REGION Network 50: Step[401] : JOB[4] Condition
   RUNG wire#powerrail
      { S7_Templates := "SrcType := DInt" } EQ_Contact(in1 := "Unit1.Em4.ControlNodes".sideTapeAttachment.sequence.status.currentStep, in2 := #JOB_4_STEP_1)
      Contact( "Unit1.Em4.ControlNodes".sideTapeAttachment.sequence.status.seqActive )
      wire#w1
      Coil( "Unit1.Em4.ControlNodes".sideTapeAttachment."step".action1[401] )
   END_RUNG
   RUNG wire#w1
      Coil( "Unit1.Em4.ControlNodes".sideTapeAttachment."step".transition1[401] )
   END_RUNG
   RUNG wire#w1
      Contact( "Unit1.Em4.ControlNodes".sideTapeAttachment."step".transition1[401] )
      { S7_Templates := "time_type := Time" } #statTonTime[401].TON(pt := T#100ms, et =>)
      wire#w2
      I_Contact( #unitStatus.specialFunctions."sideTapeLeft1 Unuse" )
      I_Contact( #unitStatus.specialFunctions."sideTapeRight1 Unuse" )
      wire#w3
      Contact( "Unit1.Em4.ControlNodes".sideTapeAttachment.homeCheck.waitPosTapeAllGet )
      wire#w4
      Move(in := #JOB_4_STEP_10, out1 => "Unit1.Em4.ControlNodes".sideTapeAttachment.sequence.status.nextStep)
   END_RUNG
   RUNG wire#w3
      Contact( "Unit1.Em4.ControlNodes".sideTapeAttachment.homeCheck.putPosTapeAllGet )
   END_RUNG wire#w4
   RUNG wire#w2
      Contact( #unitStatus.specialFunctions."sideTapeLeft1 Unuse" )
      Contact( "Unit1.Em4.ControlNodes".sideTapeAttachment.homeCheck.waitPosTapeRightGet )
   END_RUNG wire#w4
   RUNG wire#w2
      Contact( #unitStatus.specialFunctions."sideTapeRight1 Unuse" )
      Contact( "Unit1.Em4.ControlNodes".sideTapeAttachment.homeCheck.waitPosTapeLeftGet )
   END_RUNG wire#w4
   RUNG wire#w2
      Contact( #unitStatus.specialFunctions."sideTapeLeft1 Unuse" )
      Contact( #unitStatus.specialFunctions."sideTapeRight1 Unuse" )
      Move(in := #JOB_4_STEP_90, out1 => "Unit1.Em4.ControlNodes".sideTapeAttachment.sequence.status.nextStep)
   END_RUNG
   // the same network as SCL:
   "Unit1.Em4.ControlNodes".sideTapeAttachment."step".action1[401] := ("Unit1.Em4.ControlNodes".sideTapeAttachment.sequence.status.currentStep = #JOB_4_STEP_1) AND "Unit1.Em4.ControlNodes".sideTapeAttachment.sequence.status.seqActive;
   "Unit1.Em4.ControlNodes".sideTapeAttachment."step".transition1[401] := ("Unit1.Em4.ControlNodes".sideTapeAttachment.sequence.status.currentStep = #JOB_4_STEP_1) AND "Unit1.Em4.ControlNodes".sideTapeAttachment.sequence.status.seqActive;
   #statTonTime[401].TON(IN := ("Unit1.Em4.ControlNodes".sideTapeAttachment.sequence.status.currentStep = #JOB_4_STEP_1) AND "Unit1.Em4.ControlNodes".sideTapeAttachment.sequence.status.seqActive AND "Unit1.Em4.ControlNodes".sideTapeAttachment."step".transition1[401],
                         PT := T#100ms);
   IF #statTonTime[401].Q AND ((NOT #unitStatus.specialFunctions."sideTapeLeft1 Unuse" AND NOT #unitStatus.specialFunctions."sideTapeRight1 Unuse" AND ("Unit1.Em4.ControlNodes".sideTapeAttachment.homeCheck.waitPosTapeAllGet OR "Unit1.Em4.ControlNodes".sideTapeAttachment.homeCheck.putPosTapeAllGet)) OR (#unitStatus.specialFunctions."sideTapeLeft1 Unuse" AND "Unit1.Em4.ControlNodes".sideTapeAttachment.homeCheck.waitPosTapeRightGet) OR (#unitStatus.specialFunctions."sideTapeRight1 Unuse" AND "Unit1.Em4.ControlNodes".sideTapeAttachment.homeCheck.waitPosTapeLeftGet)) THEN
       "Unit1.Em4.ControlNodes".sideTapeAttachment.sequence.status.nextStep := #JOB_4_STEP_10;
   END_IF;
   IF #statTonTime[401].Q AND #unitStatus.specialFunctions."sideTapeLeft1 Unuse" AND #unitStatus.specialFunctions."sideTapeRight1 Unuse" THEN
       "Unit1.Em4.ControlNodes".sideTapeAttachment.sequence.status.nextStep := #JOB_4_STEP_90;
   END_IF;
END_REGION

REGION Network 51: Step[410] : Side Tape Attachment X-Axis Tape-1 Put Pos
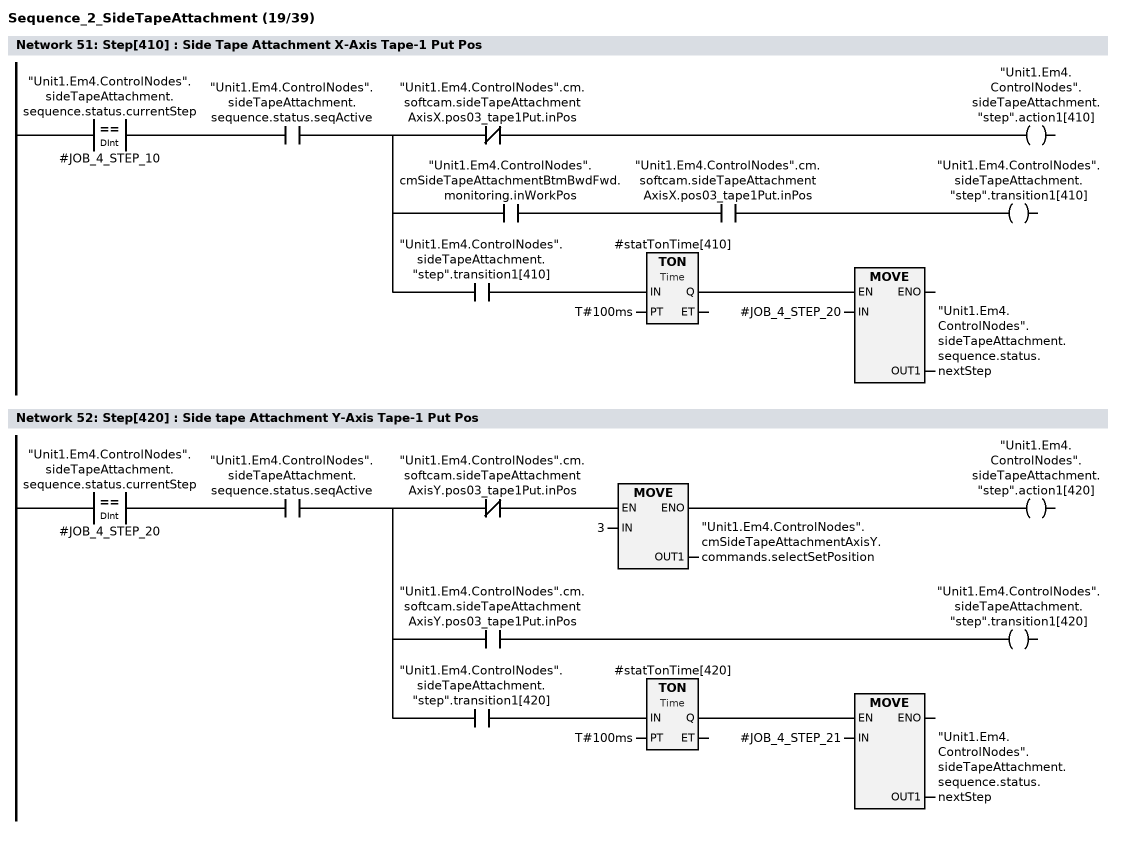
   RUNG wire#powerrail
      { S7_Templates := "SrcType := DInt" } EQ_Contact(in1 := "Unit1.Em4.ControlNodes".sideTapeAttachment.sequence.status.currentStep, in2 := #JOB_4_STEP_10)
      Contact( "Unit1.Em4.ControlNodes".sideTapeAttachment.sequence.status.seqActive )
      wire#w1
      I_Contact( "Unit1.Em4.ControlNodes".cm.softcam.sideTapeAttachmentAxisX.pos03_tape1Put.inPos )
      Coil( "Unit1.Em4.ControlNodes".sideTapeAttachment."step".action1[410] )
   END_RUNG
   RUNG wire#w1
      Contact( "Unit1.Em4.ControlNodes".cmSideTapeAttachmentBtmBwdFwd.monitoring.inWorkPos )
      Contact( "Unit1.Em4.ControlNodes".cm.softcam.sideTapeAttachmentAxisX.pos03_tape1Put.inPos )
      Coil( "Unit1.Em4.ControlNodes".sideTapeAttachment."step".transition1[410] )
   END_RUNG
   RUNG wire#w1
      Contact( "Unit1.Em4.ControlNodes".sideTapeAttachment."step".transition1[410] )
      { S7_Templates := "time_type := Time" } #statTonTime[410].TON(pt := T#100ms, et =>)
      Move(in := #JOB_4_STEP_20, out1 => "Unit1.Em4.ControlNodes".sideTapeAttachment.sequence.status.nextStep)
   END_RUNG
   // the same network as SCL:
   #_w1 := ("Unit1.Em4.ControlNodes".sideTapeAttachment.sequence.status.currentStep = #JOB_4_STEP_10) AND "Unit1.Em4.ControlNodes".sideTapeAttachment.sequence.status.seqActive;
   "Unit1.Em4.ControlNodes".sideTapeAttachment."step".action1[410] := #_w1 AND NOT "Unit1.Em4.ControlNodes".cm.softcam.sideTapeAttachmentAxisX.pos03_tape1Put.inPos;
   "Unit1.Em4.ControlNodes".sideTapeAttachment."step".transition1[410] := #_w1 AND "Unit1.Em4.ControlNodes".cmSideTapeAttachmentBtmBwdFwd.monitoring.inWorkPos AND "Unit1.Em4.ControlNodes".cm.softcam.sideTapeAttachmentAxisX.pos03_tape1Put.inPos;
   #statTonTime[410].TON(IN := #_w1 AND "Unit1.Em4.ControlNodes".sideTapeAttachment."step".transition1[410],
                         PT := T#100ms);
   IF #statTonTime[410].Q THEN
       "Unit1.Em4.ControlNodes".sideTapeAttachment.sequence.status.nextStep := #JOB_4_STEP_20;
   END_IF;
END_REGION

REGION Network 52: Step[420] : Side tape Attachment Y-Axis Tape-1 Put Pos
   RUNG wire#powerrail
      { S7_Templates := "SrcType := DInt" } EQ_Contact(in1 := "Unit1.Em4.ControlNodes".sideTapeAttachment.sequence.status.currentStep, in2 := #JOB_4_STEP_20)
      Contact( "Unit1.Em4.ControlNodes".sideTapeAttachment.sequence.status.seqActive )
      wire#w1
      I_Contact( "Unit1.Em4.ControlNodes".cm.softcam.sideTapeAttachmentAxisY.pos03_tape1Put.inPos )
      Move(in := 3, out1 => "Unit1.Em4.ControlNodes".cmSideTapeAttachmentAxisY.commands.selectSetPosition)
      Coil( "Unit1.Em4.ControlNodes".sideTapeAttachment."step".action1[420] )
   END_RUNG
   RUNG wire#w1
      Contact( "Unit1.Em4.ControlNodes".cm.softcam.sideTapeAttachmentAxisY.pos03_tape1Put.inPos )
      Coil( "Unit1.Em4.ControlNodes".sideTapeAttachment."step".transition1[420] )
   END_RUNG
   RUNG wire#w1
      Contact( "Unit1.Em4.ControlNodes".sideTapeAttachment."step".transition1[420] )
      { S7_Templates := "time_type := Time" } #statTonTime[420].TON(pt := T#100ms, et =>)
      Move(in := #JOB_4_STEP_21, out1 => "Unit1.Em4.ControlNodes".sideTapeAttachment.sequence.status.nextStep)
   END_RUNG
   // the same network as SCL:
   #_w1 := ("Unit1.Em4.ControlNodes".sideTapeAttachment.sequence.status.currentStep = #JOB_4_STEP_20) AND "Unit1.Em4.ControlNodes".sideTapeAttachment.sequence.status.seqActive;
   #_w2 := #_w1 AND NOT "Unit1.Em4.ControlNodes".cm.softcam.sideTapeAttachmentAxisY.pos03_tape1Put.inPos;
   IF #_w2 THEN "Unit1.Em4.ControlNodes".cmSideTapeAttachmentAxisY.commands.selectSetPosition := 3; END_IF;
   "Unit1.Em4.ControlNodes".sideTapeAttachment."step".action1[420] := #_w2;
   "Unit1.Em4.ControlNodes".sideTapeAttachment."step".transition1[420] := #_w1 AND "Unit1.Em4.ControlNodes".cm.softcam.sideTapeAttachmentAxisY.pos03_tape1Put.inPos;
   #statTonTime[420].TON(IN := #_w1 AND "Unit1.Em4.ControlNodes".sideTapeAttachment."step".transition1[420],
                         PT := T#100ms);
   IF #statTonTime[420].Q THEN
       "Unit1.Em4.ControlNodes".sideTapeAttachment.sequence.status.nextStep := #JOB_4_STEP_21;
   END_IF;
END_REGION

REGION Network 53: Step[421] : Side Tape Attachment Left, Right Forward, Vaccum Off
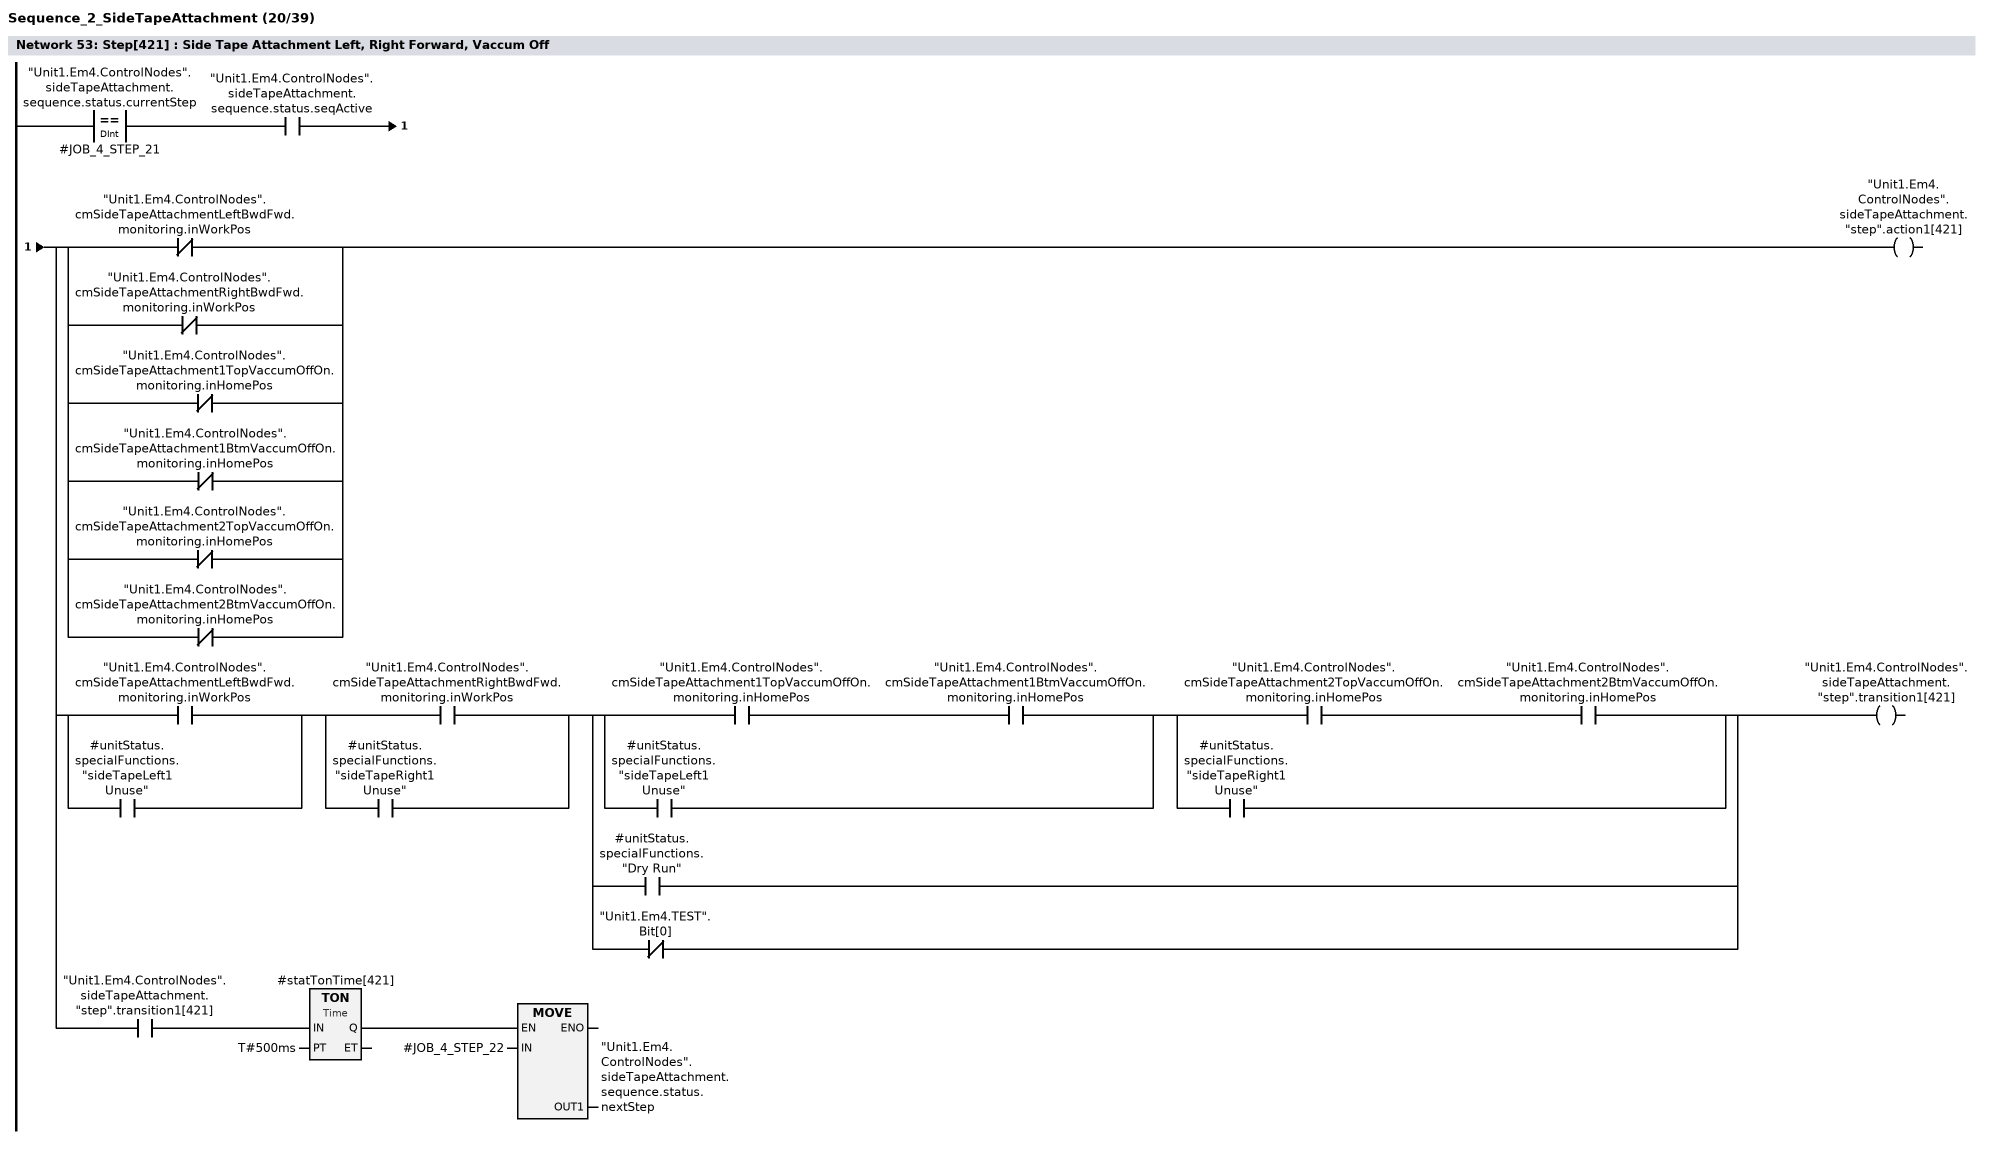
   RUNG wire#powerrail
      { S7_Templates := "SrcType := DInt" } EQ_Contact(in1 := "Unit1.Em4.ControlNodes".sideTapeAttachment.sequence.status.currentStep, in2 := #JOB_4_STEP_21)
      Contact( "Unit1.Em4.ControlNodes".sideTapeAttachment.sequence.status.seqActive )
      wire#w1
      I_Contact( "Unit1.Em4.ControlNodes".cmSideTapeAttachmentLeftBwdFwd.monitoring.inWorkPos )
      wire#w2
      Coil( "Unit1.Em4.ControlNodes".sideTapeAttachment."step".action1[421] )
   END_RUNG
   RUNG wire#w1
      I_Contact( "Unit1.Em4.ControlNodes".cmSideTapeAttachmentRightBwdFwd.monitoring.inWorkPos )
   END_RUNG wire#w2
   RUNG wire#w1
      I_Contact( "Unit1.Em4.ControlNodes".cmSideTapeAttachment1TopVaccumOffOn.monitoring.inHomePos )
   END_RUNG wire#w2
   RUNG wire#w1
      I_Contact( "Unit1.Em4.ControlNodes".cmSideTapeAttachment1BtmVaccumOffOn.monitoring.inHomePos )
   END_RUNG wire#w2
   RUNG wire#w1
      I_Contact( "Unit1.Em4.ControlNodes".cmSideTapeAttachment2TopVaccumOffOn.monitoring.inHomePos )
   END_RUNG wire#w2
   RUNG wire#w1
      I_Contact( "Unit1.Em4.ControlNodes".cmSideTapeAttachment2BtmVaccumOffOn.monitoring.inHomePos )
   END_RUNG wire#w2
   RUNG wire#w1
      Contact( "Unit1.Em4.ControlNodes".cmSideTapeAttachmentLeftBwdFwd.monitoring.inWorkPos )
      wire#w3
      Contact( "Unit1.Em4.ControlNodes".cmSideTapeAttachmentRightBwdFwd.monitoring.inWorkPos )
      wire#w4
      Contact( "Unit1.Em4.ControlNodes".cmSideTapeAttachment1TopVaccumOffOn.monitoring.inHomePos )
      Contact( "Unit1.Em4.ControlNodes".cmSideTapeAttachment1BtmVaccumOffOn.monitoring.inHomePos )
      wire#w5
      Contact( "Unit1.Em4.ControlNodes".cmSideTapeAttachment2TopVaccumOffOn.monitoring.inHomePos )
      Contact( "Unit1.Em4.ControlNodes".cmSideTapeAttachment2BtmVaccumOffOn.monitoring.inHomePos )
      wire#w6
      Coil( "Unit1.Em4.ControlNodes".sideTapeAttachment."step".transition1[421] )
   END_RUNG
   RUNG wire#w1
      Contact( #unitStatus.specialFunctions."sideTapeLeft1 Unuse" )
   END_RUNG wire#w3
   RUNG wire#w3
      Contact( #unitStatus.specialFunctions."sideTapeRight1 Unuse" )
   END_RUNG wire#w4
   RUNG wire#w4
      Contact( #unitStatus.specialFunctions."sideTapeLeft1 Unuse" )
   END_RUNG wire#w5
   RUNG wire#w5
      Contact( #unitStatus.specialFunctions."sideTapeRight1 Unuse" )
   END_RUNG wire#w6
   RUNG wire#w4
      Contact( #unitStatus.specialFunctions."Dry Run" )
   END_RUNG wire#w6
   RUNG wire#w4
      I_Contact( "Unit1.Em4.TEST".Bit[0] )
   END_RUNG wire#w6
   RUNG wire#w1
      Contact( "Unit1.Em4.ControlNodes".sideTapeAttachment."step".transition1[421] )
      { S7_Templates := "time_type := Time" } #statTonTime[421].TON(pt := T#500ms, et =>)
      Move(in := #JOB_4_STEP_22, out1 => "Unit1.Em4.ControlNodes".sideTapeAttachment.sequence.status.nextStep)
   END_RUNG
   // the same network as SCL:
   #_w1 := ("Unit1.Em4.ControlNodes".sideTapeAttachment.sequence.status.currentStep = #JOB_4_STEP_21) AND "Unit1.Em4.ControlNodes".sideTapeAttachment.sequence.status.seqActive;
   "Unit1.Em4.ControlNodes".sideTapeAttachment."step".action1[421] := #_w1 AND (NOT "Unit1.Em4.ControlNodes".cmSideTapeAttachmentLeftBwdFwd.monitoring.inWorkPos OR NOT "Unit1.Em4.ControlNodes".cmSideTapeAttachmentRightBwdFwd.monitoring.inWorkPos OR NOT "Unit1.Em4.ControlNodes".cmSideTapeAttachment1TopVaccumOffOn.monitoring.inHomePos OR NOT "Unit1.Em4.ControlNodes".cmSideTapeAttachment1BtmVaccumOffOn.monitoring.inHomePos OR NOT "Unit1.Em4.ControlNodes".cmSideTapeAttachment2TopVaccumOffOn.monitoring.inHomePos OR NOT "Unit1.Em4.ControlNodes".cmSideTapeAttachment2BtmVaccumOffOn.monitoring.inHomePos);
   "Unit1.Em4.ControlNodes".sideTapeAttachment."step".transition1[421] := #_w1 AND ("Unit1.Em4.ControlNodes".cmSideTapeAttachmentLeftBwdFwd.monitoring.inWorkPos OR #unitStatus.specialFunctions."sideTapeLeft1 Unuse") AND ("Unit1.Em4.ControlNodes".cmSideTapeAttachmentRightBwdFwd.monitoring.inWorkPos OR #unitStatus.specialFunctions."sideTapeRight1 Unuse") AND (((("Unit1.Em4.ControlNodes".cmSideTapeAttachment1TopVaccumOffOn.monitoring.inHomePos AND "Unit1.Em4.ControlNodes".cmSideTapeAttachment1BtmVaccumOffOn.monitoring.inHomePos) OR #unitStatus.specialFunctions."sideTapeLeft1 Unuse") AND (("Unit1.Em4.ControlNodes".cmSideTapeAttachment2TopVaccumOffOn.monitoring.inHomePos AND "Unit1.Em4.ControlNodes".cmSideTapeAttachment2BtmVaccumOffOn.monitoring.inHomePos) OR #unitStatus.specialFunctions."sideTapeRight1 Unuse")) OR #unitStatus.specialFunctions."Dry Run" OR NOT "Unit1.Em4.TEST".Bit[0]);
   #statTonTime[421].TON(IN := #_w1 AND "Unit1.Em4.ControlNodes".sideTapeAttachment."step".transition1[421],
                         PT := T#500ms);
   IF #statTonTime[421].Q THEN
       "Unit1.Em4.ControlNodes".sideTapeAttachment.sequence.status.nextStep := #JOB_4_STEP_22;
   END_IF;
END_REGION

REGION Network 54: Step[422] : Spare
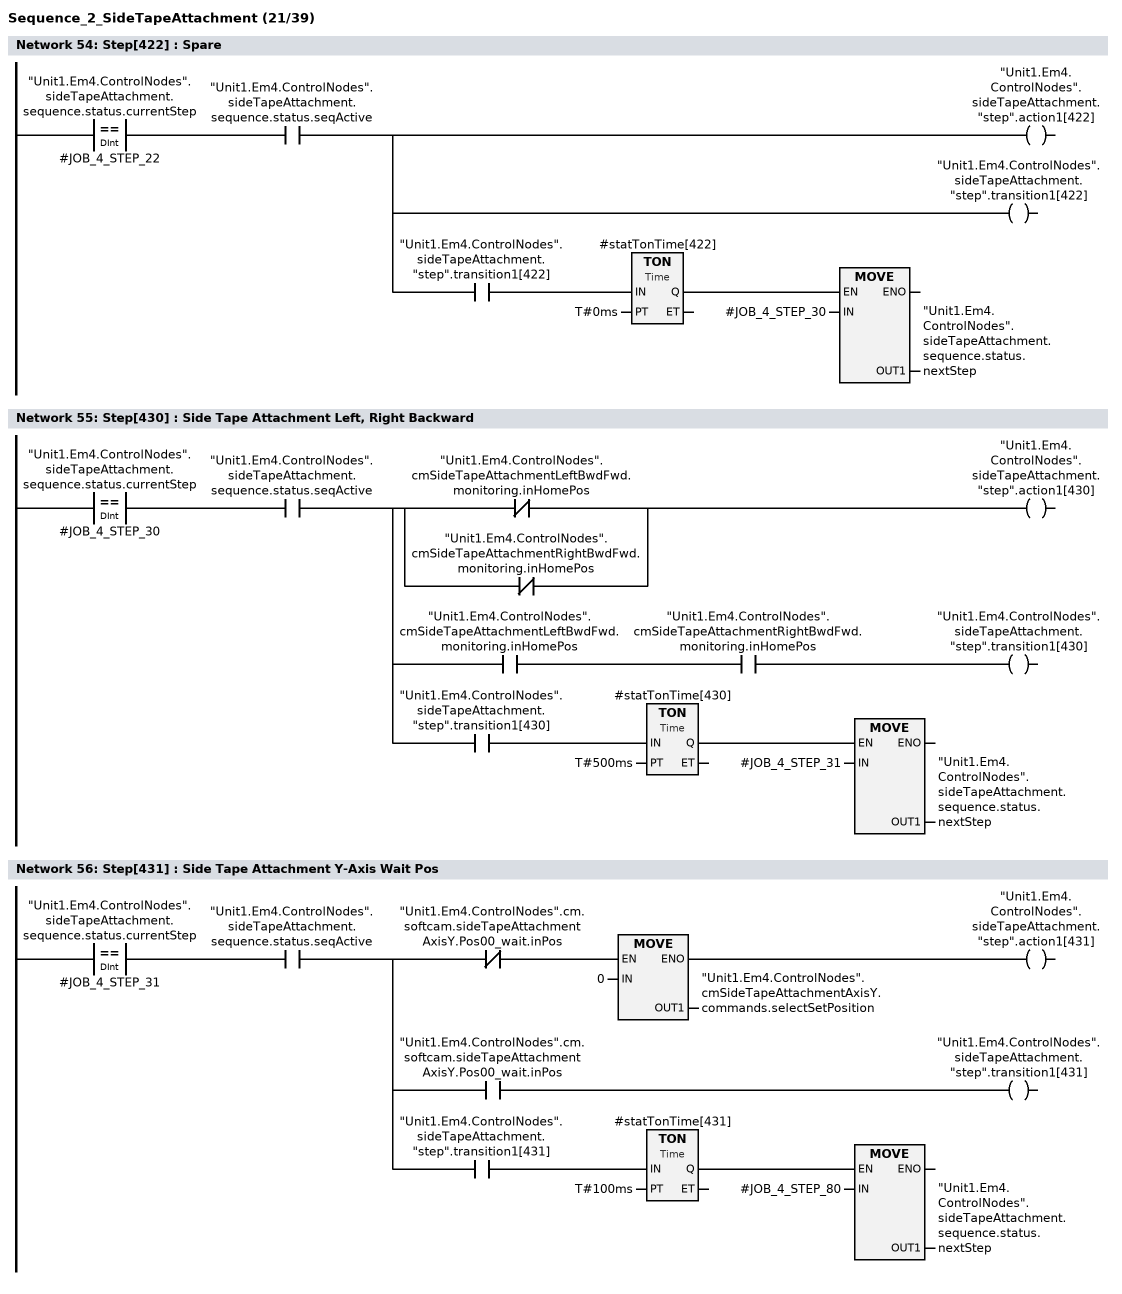
   RUNG wire#powerrail
      { S7_Templates := "SrcType := DInt" } EQ_Contact(in1 := "Unit1.Em4.ControlNodes".sideTapeAttachment.sequence.status.currentStep, in2 := #JOB_4_STEP_22)
      Contact( "Unit1.Em4.ControlNodes".sideTapeAttachment.sequence.status.seqActive )
      wire#w1
      Coil( "Unit1.Em4.ControlNodes".sideTapeAttachment."step".action1[422] )
   END_RUNG
   RUNG wire#w1
      Coil( "Unit1.Em4.ControlNodes".sideTapeAttachment."step".transition1[422] )
   END_RUNG
   RUNG wire#w1
      Contact( "Unit1.Em4.ControlNodes".sideTapeAttachment."step".transition1[422] )
      { S7_Templates := "time_type := Time" } #statTonTime[422].TON(pt := T#0ms, et =>)
      Move(in := #JOB_4_STEP_30, out1 => "Unit1.Em4.ControlNodes".sideTapeAttachment.sequence.status.nextStep)
   END_RUNG
   // the same network as SCL:
   "Unit1.Em4.ControlNodes".sideTapeAttachment."step".action1[422] := ("Unit1.Em4.ControlNodes".sideTapeAttachment.sequence.status.currentStep = #JOB_4_STEP_22) AND "Unit1.Em4.ControlNodes".sideTapeAttachment.sequence.status.seqActive;
   "Unit1.Em4.ControlNodes".sideTapeAttachment."step".transition1[422] := ("Unit1.Em4.ControlNodes".sideTapeAttachment.sequence.status.currentStep = #JOB_4_STEP_22) AND "Unit1.Em4.ControlNodes".sideTapeAttachment.sequence.status.seqActive;
   #statTonTime[422].TON(IN := ("Unit1.Em4.ControlNodes".sideTapeAttachment.sequence.status.currentStep = #JOB_4_STEP_22) AND "Unit1.Em4.ControlNodes".sideTapeAttachment.sequence.status.seqActive AND "Unit1.Em4.ControlNodes".sideTapeAttachment."step".transition1[422],
                         PT := T#0ms);
   IF #statTonTime[422].Q THEN
       "Unit1.Em4.ControlNodes".sideTapeAttachment.sequence.status.nextStep := #JOB_4_STEP_30;
   END_IF;
END_REGION

REGION Network 55: Step[430] : Side Tape Attachment Left, Right Backward
   RUNG wire#powerrail
      { S7_Templates := "SrcType := DInt" } EQ_Contact(in1 := "Unit1.Em4.ControlNodes".sideTapeAttachment.sequence.status.currentStep, in2 := #JOB_4_STEP_30)
      Contact( "Unit1.Em4.ControlNodes".sideTapeAttachment.sequence.status.seqActive )
      wire#w1
      I_Contact( "Unit1.Em4.ControlNodes".cmSideTapeAttachmentLeftBwdFwd.monitoring.inHomePos )
      wire#w2
      Coil( "Unit1.Em4.ControlNodes".sideTapeAttachment."step".action1[430] )
   END_RUNG
   RUNG wire#w1
      I_Contact( "Unit1.Em4.ControlNodes".cmSideTapeAttachmentRightBwdFwd.monitoring.inHomePos )
   END_RUNG wire#w2
   RUNG wire#w1
      Contact( "Unit1.Em4.ControlNodes".cmSideTapeAttachmentLeftBwdFwd.monitoring.inHomePos )
      Contact( "Unit1.Em4.ControlNodes".cmSideTapeAttachmentRightBwdFwd.monitoring.inHomePos )
      Coil( "Unit1.Em4.ControlNodes".sideTapeAttachment."step".transition1[430] )
   END_RUNG
   RUNG wire#w1
      Contact( "Unit1.Em4.ControlNodes".sideTapeAttachment."step".transition1[430] )
      { S7_Templates := "time_type := Time" } #statTonTime[430].TON(pt := T#500ms, et =>)
      Move(in := #JOB_4_STEP_31, out1 => "Unit1.Em4.ControlNodes".sideTapeAttachment.sequence.status.nextStep)
   END_RUNG
   // the same network as SCL:
   #_w1 := ("Unit1.Em4.ControlNodes".sideTapeAttachment.sequence.status.currentStep = #JOB_4_STEP_30) AND "Unit1.Em4.ControlNodes".sideTapeAttachment.sequence.status.seqActive;
   "Unit1.Em4.ControlNodes".sideTapeAttachment."step".action1[430] := #_w1 AND (NOT "Unit1.Em4.ControlNodes".cmSideTapeAttachmentLeftBwdFwd.monitoring.inHomePos OR NOT "Unit1.Em4.ControlNodes".cmSideTapeAttachmentRightBwdFwd.monitoring.inHomePos);
   "Unit1.Em4.ControlNodes".sideTapeAttachment."step".transition1[430] := #_w1 AND "Unit1.Em4.ControlNodes".cmSideTapeAttachmentLeftBwdFwd.monitoring.inHomePos AND "Unit1.Em4.ControlNodes".cmSideTapeAttachmentRightBwdFwd.monitoring.inHomePos;
   #statTonTime[430].TON(IN := #_w1 AND "Unit1.Em4.ControlNodes".sideTapeAttachment."step".transition1[430],
                         PT := T#500ms);
   IF #statTonTime[430].Q THEN
       "Unit1.Em4.ControlNodes".sideTapeAttachment.sequence.status.nextStep := #JOB_4_STEP_31;
   END_IF;
END_REGION

REGION Network 56: Step[431] : Side Tape Attachment Y-Axis Wait Pos
   RUNG wire#powerrail
      { S7_Templates := "SrcType := DInt" } EQ_Contact(in1 := "Unit1.Em4.ControlNodes".sideTapeAttachment.sequence.status.currentStep, in2 := #JOB_4_STEP_31)
      Contact( "Unit1.Em4.ControlNodes".sideTapeAttachment.sequence.status.seqActive )
      wire#w1
      I_Contact( "Unit1.Em4.ControlNodes".cm.softcam.sideTapeAttachmentAxisY.Pos00_wait.inPos )
      Move(in := 0, out1 => "Unit1.Em4.ControlNodes".cmSideTapeAttachmentAxisY.commands.selectSetPosition)
      Coil( "Unit1.Em4.ControlNodes".sideTapeAttachment."step".action1[431] )
   END_RUNG
   RUNG wire#w1
      Contact( "Unit1.Em4.ControlNodes".cm.softcam.sideTapeAttachmentAxisY.Pos00_wait.inPos )
      Coil( "Unit1.Em4.ControlNodes".sideTapeAttachment."step".transition1[431] )
   END_RUNG
   RUNG wire#w1
      Contact( "Unit1.Em4.ControlNodes".sideTapeAttachment."step".transition1[431] )
      { S7_Templates := "time_type := Time" } #statTonTime[431].TON(pt := T#100ms, et =>)
      Move(in := #JOB_4_STEP_80, out1 => "Unit1.Em4.ControlNodes".sideTapeAttachment.sequence.status.nextStep)
   END_RUNG
   // the same network as SCL:
   #_w1 := ("Unit1.Em4.ControlNodes".sideTapeAttachment.sequence.status.currentStep = #JOB_4_STEP_31) AND "Unit1.Em4.ControlNodes".sideTapeAttachment.sequence.status.seqActive;
   #_w2 := #_w1 AND NOT "Unit1.Em4.ControlNodes".cm.softcam.sideTapeAttachmentAxisY.Pos00_wait.inPos;
   IF #_w2 THEN "Unit1.Em4.ControlNodes".cmSideTapeAttachmentAxisY.commands.selectSetPosition := 0; END_IF;
   "Unit1.Em4.ControlNodes".sideTapeAttachment."step".action1[431] := #_w2;
   "Unit1.Em4.ControlNodes".sideTapeAttachment."step".transition1[431] := #_w1 AND "Unit1.Em4.ControlNodes".cm.softcam.sideTapeAttachmentAxisY.Pos00_wait.inPos;
   #statTonTime[431].TON(IN := #_w1 AND "Unit1.Em4.ControlNodes".sideTapeAttachment."step".transition1[431],
                         PT := T#100ms);
   IF #statTonTime[431].Q THEN
       "Unit1.Em4.ControlNodes".sideTapeAttachment.sequence.status.nextStep := #JOB_4_STEP_80;
   END_IF;
END_REGION

REGION Network 57: Step[480] : Side Tape Attachment X-Axis Wait Pos
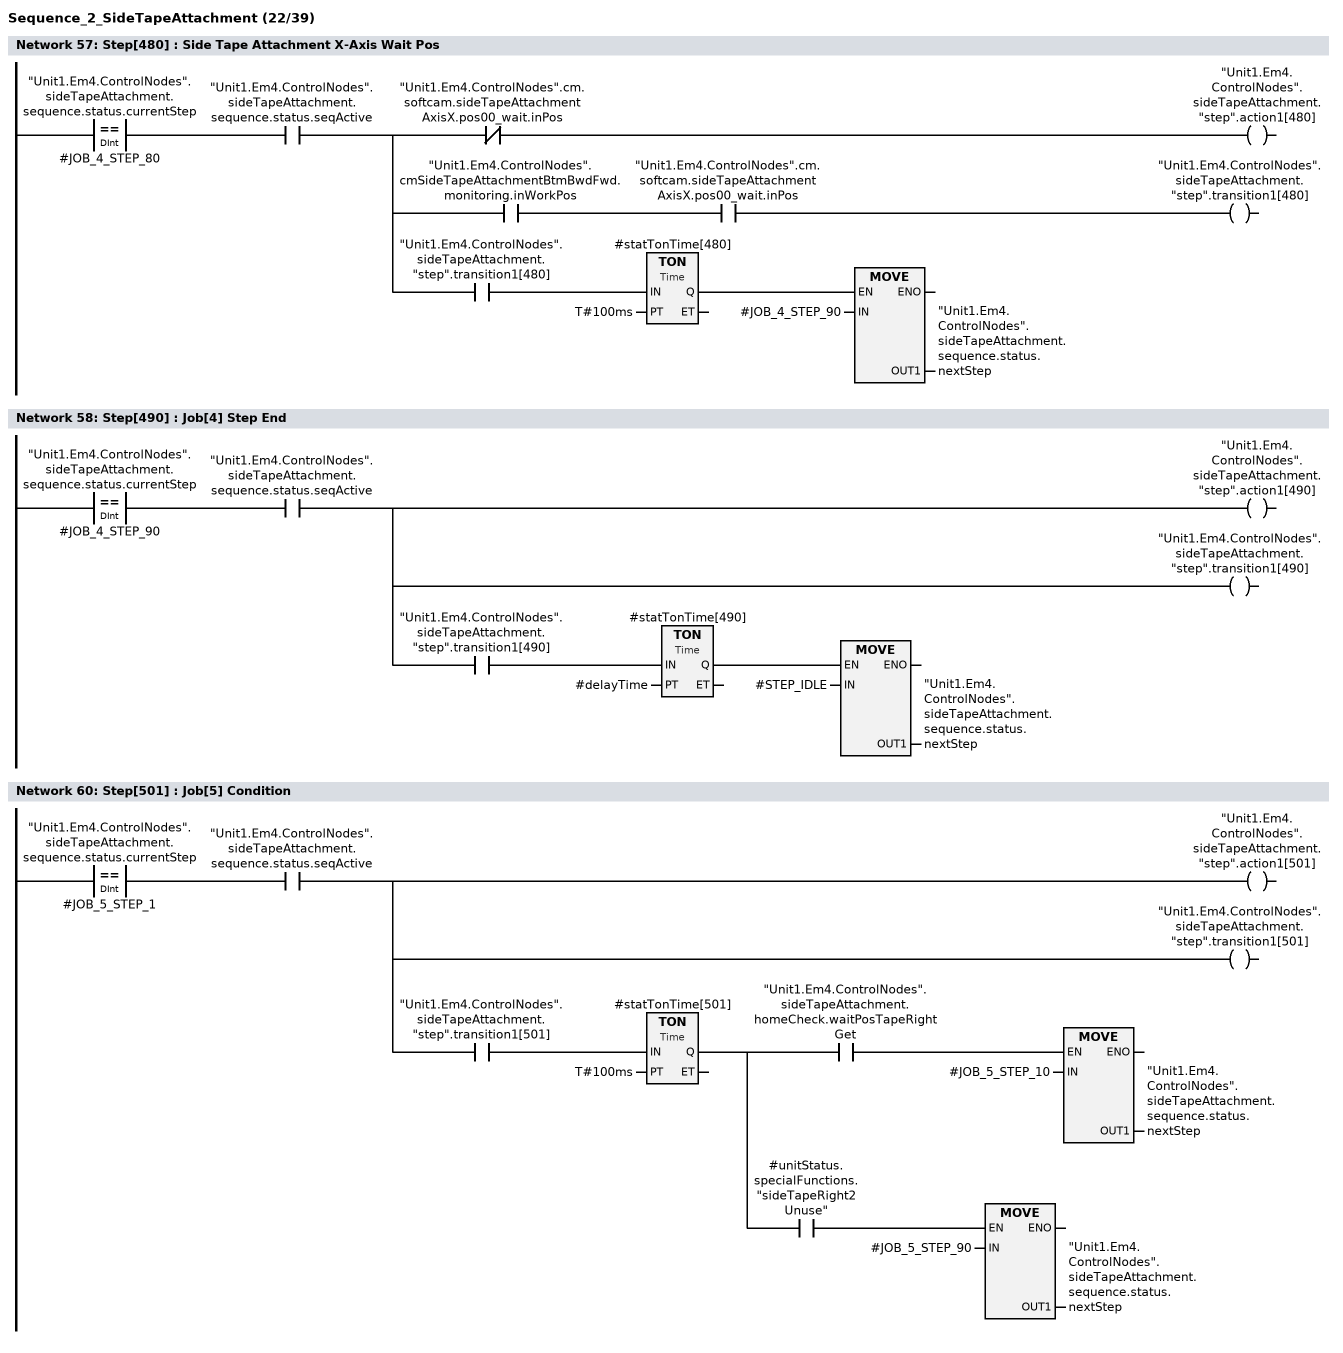
   RUNG wire#powerrail
      { S7_Templates := "SrcType := DInt" } EQ_Contact(in1 := "Unit1.Em4.ControlNodes".sideTapeAttachment.sequence.status.currentStep, in2 := #JOB_4_STEP_80)
      Contact( "Unit1.Em4.ControlNodes".sideTapeAttachment.sequence.status.seqActive )
      wire#w1
      I_Contact( "Unit1.Em4.ControlNodes".cm.softcam.sideTapeAttachmentAxisX.pos00_wait.inPos )
      Coil( "Unit1.Em4.ControlNodes".sideTapeAttachment."step".action1[480] )
   END_RUNG
   RUNG wire#w1
      Contact( "Unit1.Em4.ControlNodes".cmSideTapeAttachmentBtmBwdFwd.monitoring.inWorkPos )
      Contact( "Unit1.Em4.ControlNodes".cm.softcam.sideTapeAttachmentAxisX.pos00_wait.inPos )
      Coil( "Unit1.Em4.ControlNodes".sideTapeAttachment."step".transition1[480] )
   END_RUNG
   RUNG wire#w1
      Contact( "Unit1.Em4.ControlNodes".sideTapeAttachment."step".transition1[480] )
      { S7_Templates := "time_type := Time" } #statTonTime[480].TON(pt := T#100ms, et =>)
      Move(in := #JOB_4_STEP_90, out1 => "Unit1.Em4.ControlNodes".sideTapeAttachment.sequence.status.nextStep)
   END_RUNG
   // the same network as SCL:
   #_w1 := ("Unit1.Em4.ControlNodes".sideTapeAttachment.sequence.status.currentStep = #JOB_4_STEP_80) AND "Unit1.Em4.ControlNodes".sideTapeAttachment.sequence.status.seqActive;
   "Unit1.Em4.ControlNodes".sideTapeAttachment."step".action1[480] := #_w1 AND NOT "Unit1.Em4.ControlNodes".cm.softcam.sideTapeAttachmentAxisX.pos00_wait.inPos;
   "Unit1.Em4.ControlNodes".sideTapeAttachment."step".transition1[480] := #_w1 AND "Unit1.Em4.ControlNodes".cmSideTapeAttachmentBtmBwdFwd.monitoring.inWorkPos AND "Unit1.Em4.ControlNodes".cm.softcam.sideTapeAttachmentAxisX.pos00_wait.inPos;
   #statTonTime[480].TON(IN := #_w1 AND "Unit1.Em4.ControlNodes".sideTapeAttachment."step".transition1[480],
                         PT := T#100ms);
   IF #statTonTime[480].Q THEN
       "Unit1.Em4.ControlNodes".sideTapeAttachment.sequence.status.nextStep := #JOB_4_STEP_90;
   END_IF;
END_REGION

REGION Network 58: Step[490] : Job[4] Step End
   RUNG wire#powerrail
      { S7_Templates := "SrcType := DInt" } EQ_Contact(in1 := "Unit1.Em4.ControlNodes".sideTapeAttachment.sequence.status.currentStep, in2 := #JOB_4_STEP_90)
      Contact( "Unit1.Em4.ControlNodes".sideTapeAttachment.sequence.status.seqActive )
      wire#w1
      Coil( "Unit1.Em4.ControlNodes".sideTapeAttachment."step".action1[490] )
   END_RUNG
   RUNG wire#w1
      Coil( "Unit1.Em4.ControlNodes".sideTapeAttachment."step".transition1[490] )
   END_RUNG
   RUNG wire#w1
      Contact( "Unit1.Em4.ControlNodes".sideTapeAttachment."step".transition1[490] )
      { S7_Templates := "time_type := Time" } #statTonTime[490].TON(pt := #delayTime, et =>)
      Move(in := #STEP_IDLE, out1 => "Unit1.Em4.ControlNodes".sideTapeAttachment.sequence.status.nextStep)
   END_RUNG
   // the same network as SCL:
   "Unit1.Em4.ControlNodes".sideTapeAttachment."step".action1[490] := ("Unit1.Em4.ControlNodes".sideTapeAttachment.sequence.status.currentStep = #JOB_4_STEP_90) AND "Unit1.Em4.ControlNodes".sideTapeAttachment.sequence.status.seqActive;
   "Unit1.Em4.ControlNodes".sideTapeAttachment."step".transition1[490] := ("Unit1.Em4.ControlNodes".sideTapeAttachment.sequence.status.currentStep = #JOB_4_STEP_90) AND "Unit1.Em4.ControlNodes".sideTapeAttachment.sequence.status.seqActive;
   #statTonTime[490].TON(IN := ("Unit1.Em4.ControlNodes".sideTapeAttachment.sequence.status.currentStep = #JOB_4_STEP_90) AND "Unit1.Em4.ControlNodes".sideTapeAttachment.sequence.status.seqActive AND "Unit1.Em4.ControlNodes".sideTapeAttachment."step".transition1[490],
                         PT := #delayTime);
   IF #statTonTime[490].Q THEN
       "Unit1.Em4.ControlNodes".sideTapeAttachment.sequence.status.nextStep := #STEP_IDLE;
   END_IF;
END_REGION

REGION Network 59: *************** JOB[5] SIDE TAPE PUT-2=AUTO *************************
END_REGION

REGION Network 60: Step[501] : Job[5] Condition
   RUNG wire#powerrail
      { S7_Templates := "SrcType := DInt" } EQ_Contact(in1 := "Unit1.Em4.ControlNodes".sideTapeAttachment.sequence.status.currentStep, in2 := #JOB_5_STEP_1)
      Contact( "Unit1.Em4.ControlNodes".sideTapeAttachment.sequence.status.seqActive )
      wire#w1
      Coil( "Unit1.Em4.ControlNodes".sideTapeAttachment."step".action1[501] )
   END_RUNG
   RUNG wire#w1
      Coil( "Unit1.Em4.ControlNodes".sideTapeAttachment."step".transition1[501] )
   END_RUNG
   RUNG wire#w1
      Contact( "Unit1.Em4.ControlNodes".sideTapeAttachment."step".transition1[501] )
      { S7_Templates := "time_type := Time" } #statTonTime[501].TON(pt := T#100ms, et =>)
      wire#w2
      Contact( "Unit1.Em4.ControlNodes".sideTapeAttachment.homeCheck.waitPosTapeRightGet )
      Move(in := #JOB_5_STEP_10, out1 => "Unit1.Em4.ControlNodes".sideTapeAttachment.sequence.status.nextStep)
   END_RUNG
   RUNG wire#w2
      Contact( #unitStatus.specialFunctions."sideTapeRight2 Unuse" )
      Move(in := #JOB_5_STEP_90, out1 => "Unit1.Em4.ControlNodes".sideTapeAttachment.sequence.status.nextStep)
   END_RUNG
   // the same network as SCL:
   "Unit1.Em4.ControlNodes".sideTapeAttachment."step".action1[501] := ("Unit1.Em4.ControlNodes".sideTapeAttachment.sequence.status.currentStep = #JOB_5_STEP_1) AND "Unit1.Em4.ControlNodes".sideTapeAttachment.sequence.status.seqActive;
   "Unit1.Em4.ControlNodes".sideTapeAttachment."step".transition1[501] := ("Unit1.Em4.ControlNodes".sideTapeAttachment.sequence.status.currentStep = #JOB_5_STEP_1) AND "Unit1.Em4.ControlNodes".sideTapeAttachment.sequence.status.seqActive;
   #statTonTime[501].TON(IN := ("Unit1.Em4.ControlNodes".sideTapeAttachment.sequence.status.currentStep = #JOB_5_STEP_1) AND "Unit1.Em4.ControlNodes".sideTapeAttachment.sequence.status.seqActive AND "Unit1.Em4.ControlNodes".sideTapeAttachment."step".transition1[501],
                         PT := T#100ms);
   IF #statTonTime[501].Q AND "Unit1.Em4.ControlNodes".sideTapeAttachment.homeCheck.waitPosTapeRightGet THEN
       "Unit1.Em4.ControlNodes".sideTapeAttachment.sequence.status.nextStep := #JOB_5_STEP_10;
   END_IF;
   IF #statTonTime[501].Q AND #unitStatus.specialFunctions."sideTapeRight2 Unuse" THEN
       "Unit1.Em4.ControlNodes".sideTapeAttachment.sequence.status.nextStep := #JOB_5_STEP_90;
   END_IF;
END_REGION

REGION Network 61: Step[510] : Side Tape Attachment X-Axis Tape-2 Put Pos
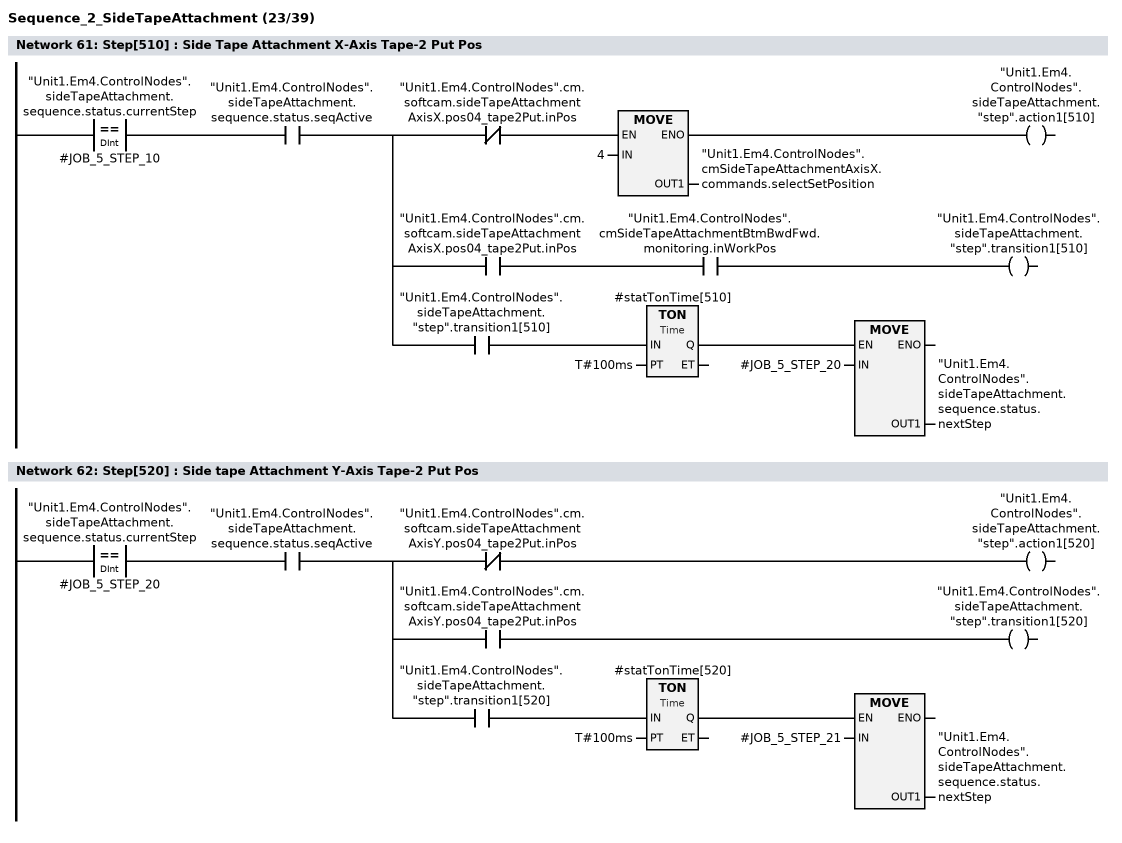
   RUNG wire#powerrail
      { S7_Templates := "SrcType := DInt" } EQ_Contact(in1 := "Unit1.Em4.ControlNodes".sideTapeAttachment.sequence.status.currentStep, in2 := #JOB_5_STEP_10)
      Contact( "Unit1.Em4.ControlNodes".sideTapeAttachment.sequence.status.seqActive )
      wire#w1
      I_Contact( "Unit1.Em4.ControlNodes".cm.softcam.sideTapeAttachmentAxisX.pos04_tape2Put.inPos )
      Move(in := 4, out1 => "Unit1.Em4.ControlNodes".cmSideTapeAttachmentAxisX.commands.selectSetPosition)
      Coil( "Unit1.Em4.ControlNodes".sideTapeAttachment."step".action1[510] )
   END_RUNG
   RUNG wire#w1
      Contact( "Unit1.Em4.ControlNodes".cm.softcam.sideTapeAttachmentAxisX.pos04_tape2Put.inPos )
      Contact( "Unit1.Em4.ControlNodes".cmSideTapeAttachmentBtmBwdFwd.monitoring.inWorkPos )
      Coil( "Unit1.Em4.ControlNodes".sideTapeAttachment."step".transition1[510] )
   END_RUNG
   RUNG wire#w1
      Contact( "Unit1.Em4.ControlNodes".sideTapeAttachment."step".transition1[510] )
      { S7_Templates := "time_type := Time" } #statTonTime[510].TON(pt := T#100ms, et =>)
      Move(in := #JOB_5_STEP_20, out1 => "Unit1.Em4.ControlNodes".sideTapeAttachment.sequence.status.nextStep)
   END_RUNG
   // the same network as SCL:
   #_w1 := ("Unit1.Em4.ControlNodes".sideTapeAttachment.sequence.status.currentStep = #JOB_5_STEP_10) AND "Unit1.Em4.ControlNodes".sideTapeAttachment.sequence.status.seqActive;
   #_w2 := #_w1 AND NOT "Unit1.Em4.ControlNodes".cm.softcam.sideTapeAttachmentAxisX.pos04_tape2Put.inPos;
   IF #_w2 THEN "Unit1.Em4.ControlNodes".cmSideTapeAttachmentAxisX.commands.selectSetPosition := 4; END_IF;
   "Unit1.Em4.ControlNodes".sideTapeAttachment."step".action1[510] := #_w2;
   "Unit1.Em4.ControlNodes".sideTapeAttachment."step".transition1[510] := #_w1 AND "Unit1.Em4.ControlNodes".cm.softcam.sideTapeAttachmentAxisX.pos04_tape2Put.inPos AND "Unit1.Em4.ControlNodes".cmSideTapeAttachmentBtmBwdFwd.monitoring.inWorkPos;
   #statTonTime[510].TON(IN := #_w1 AND "Unit1.Em4.ControlNodes".sideTapeAttachment."step".transition1[510],
                         PT := T#100ms);
   IF #statTonTime[510].Q THEN
       "Unit1.Em4.ControlNodes".sideTapeAttachment.sequence.status.nextStep := #JOB_5_STEP_20;
   END_IF;
END_REGION

REGION Network 62: Step[520] : Side tape Attachment Y-Axis Tape-2 Put Pos
   RUNG wire#powerrail
      { S7_Templates := "SrcType := DInt" } EQ_Contact(in1 := "Unit1.Em4.ControlNodes".sideTapeAttachment.sequence.status.currentStep, in2 := #JOB_5_STEP_20)
      Contact( "Unit1.Em4.ControlNodes".sideTapeAttachment.sequence.status.seqActive )
      wire#w1
      I_Contact( "Unit1.Em4.ControlNodes".cm.softcam.sideTapeAttachmentAxisY.pos04_tape2Put.inPos )
      Coil( "Unit1.Em4.ControlNodes".sideTapeAttachment."step".action1[520] )
   END_RUNG
   RUNG wire#w1
      Contact( "Unit1.Em4.ControlNodes".cm.softcam.sideTapeAttachmentAxisY.pos04_tape2Put.inPos )
      Coil( "Unit1.Em4.ControlNodes".sideTapeAttachment."step".transition1[520] )
   END_RUNG
   RUNG wire#w1
      Contact( "Unit1.Em4.ControlNodes".sideTapeAttachment."step".transition1[520] )
      { S7_Templates := "time_type := Time" } #statTonTime[520].TON(pt := T#100ms, et =>)
      Move(in := #JOB_5_STEP_21, out1 => "Unit1.Em4.ControlNodes".sideTapeAttachment.sequence.status.nextStep)
   END_RUNG
   // the same network as SCL:
   #_w1 := ("Unit1.Em4.ControlNodes".sideTapeAttachment.sequence.status.currentStep = #JOB_5_STEP_20) AND "Unit1.Em4.ControlNodes".sideTapeAttachment.sequence.status.seqActive;
   "Unit1.Em4.ControlNodes".sideTapeAttachment."step".action1[520] := #_w1 AND NOT "Unit1.Em4.ControlNodes".cm.softcam.sideTapeAttachmentAxisY.pos04_tape2Put.inPos;
   "Unit1.Em4.ControlNodes".sideTapeAttachment."step".transition1[520] := #_w1 AND "Unit1.Em4.ControlNodes".cm.softcam.sideTapeAttachmentAxisY.pos04_tape2Put.inPos;
   #statTonTime[520].TON(IN := #_w1 AND "Unit1.Em4.ControlNodes".sideTapeAttachment."step".transition1[520],
                         PT := T#100ms);
   IF #statTonTime[520].Q THEN
       "Unit1.Em4.ControlNodes".sideTapeAttachment.sequence.status.nextStep := #JOB_5_STEP_21;
   END_IF;
END_REGION

REGION Network 63: Step[521] : Side Tape Attachment Right Forward, Vaccum Off
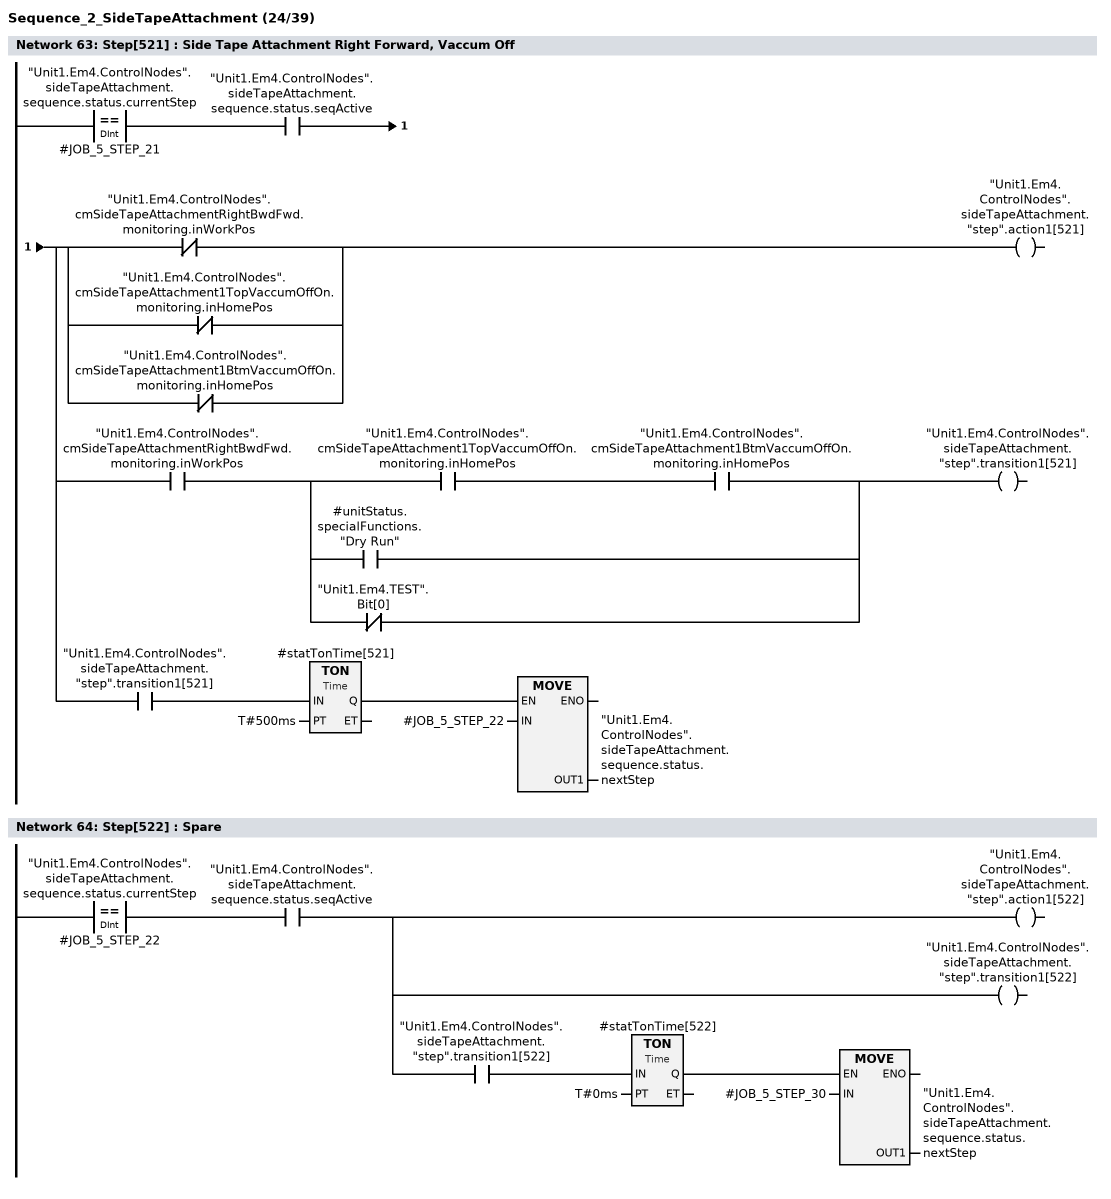
   RUNG wire#powerrail
      { S7_Templates := "SrcType := DInt" } EQ_Contact(in1 := "Unit1.Em4.ControlNodes".sideTapeAttachment.sequence.status.currentStep, in2 := #JOB_5_STEP_21)
      Contact( "Unit1.Em4.ControlNodes".sideTapeAttachment.sequence.status.seqActive )
      wire#w1
      I_Contact( "Unit1.Em4.ControlNodes".cmSideTapeAttachmentRightBwdFwd.monitoring.inWorkPos )
      wire#w2
      Coil( "Unit1.Em4.ControlNodes".sideTapeAttachment."step".action1[521] )
   END_RUNG
   RUNG wire#w1
      I_Contact( "Unit1.Em4.ControlNodes".cmSideTapeAttachment1TopVaccumOffOn.monitoring.inHomePos )
   END_RUNG wire#w2
   RUNG wire#w1
      I_Contact( "Unit1.Em4.ControlNodes".cmSideTapeAttachment1BtmVaccumOffOn.monitoring.inHomePos )
   END_RUNG wire#w2
   RUNG wire#w1
      Contact( "Unit1.Em4.ControlNodes".cmSideTapeAttachmentRightBwdFwd.monitoring.inWorkPos )
      wire#w3
      Contact( "Unit1.Em4.ControlNodes".cmSideTapeAttachment1TopVaccumOffOn.monitoring.inHomePos )
      Contact( "Unit1.Em4.ControlNodes".cmSideTapeAttachment1BtmVaccumOffOn.monitoring.inHomePos )
      wire#w4
      Coil( "Unit1.Em4.ControlNodes".sideTapeAttachment."step".transition1[521] )
   END_RUNG
   RUNG wire#w3
      Contact( #unitStatus.specialFunctions."Dry Run" )
   END_RUNG wire#w4
   RUNG wire#w3
      I_Contact( "Unit1.Em4.TEST".Bit[0] )
   END_RUNG wire#w4
   RUNG wire#w1
      Contact( "Unit1.Em4.ControlNodes".sideTapeAttachment."step".transition1[521] )
      { S7_Templates := "time_type := Time" } #statTonTime[521].TON(pt := T#500ms, et =>)
      Move(in := #JOB_5_STEP_22, out1 => "Unit1.Em4.ControlNodes".sideTapeAttachment.sequence.status.nextStep)
   END_RUNG
   // the same network as SCL:
   #_w1 := ("Unit1.Em4.ControlNodes".sideTapeAttachment.sequence.status.currentStep = #JOB_5_STEP_21) AND "Unit1.Em4.ControlNodes".sideTapeAttachment.sequence.status.seqActive;
   "Unit1.Em4.ControlNodes".sideTapeAttachment."step".action1[521] := #_w1 AND (NOT "Unit1.Em4.ControlNodes".cmSideTapeAttachmentRightBwdFwd.monitoring.inWorkPos OR NOT "Unit1.Em4.ControlNodes".cmSideTapeAttachment1TopVaccumOffOn.monitoring.inHomePos OR NOT "Unit1.Em4.ControlNodes".cmSideTapeAttachment1BtmVaccumOffOn.monitoring.inHomePos);
   "Unit1.Em4.ControlNodes".sideTapeAttachment."step".transition1[521] := #_w1 AND "Unit1.Em4.ControlNodes".cmSideTapeAttachmentRightBwdFwd.monitoring.inWorkPos AND (("Unit1.Em4.ControlNodes".cmSideTapeAttachment1TopVaccumOffOn.monitoring.inHomePos AND "Unit1.Em4.ControlNodes".cmSideTapeAttachment1BtmVaccumOffOn.monitoring.inHomePos) OR #unitStatus.specialFunctions."Dry Run" OR NOT "Unit1.Em4.TEST".Bit[0]);
   #statTonTime[521].TON(IN := #_w1 AND "Unit1.Em4.ControlNodes".sideTapeAttachment."step".transition1[521],
                         PT := T#500ms);
   IF #statTonTime[521].Q THEN
       "Unit1.Em4.ControlNodes".sideTapeAttachment.sequence.status.nextStep := #JOB_5_STEP_22;
   END_IF;
END_REGION

REGION Network 64: Step[522] : Spare
   RUNG wire#powerrail
      { S7_Templates := "SrcType := DInt" } EQ_Contact(in1 := "Unit1.Em4.ControlNodes".sideTapeAttachment.sequence.status.currentStep, in2 := #JOB_5_STEP_22)
      Contact( "Unit1.Em4.ControlNodes".sideTapeAttachment.sequence.status.seqActive )
      wire#w1
      Coil( "Unit1.Em4.ControlNodes".sideTapeAttachment."step".action1[522] )
   END_RUNG
   RUNG wire#w1
      Coil( "Unit1.Em4.ControlNodes".sideTapeAttachment."step".transition1[522] )
   END_RUNG
   RUNG wire#w1
      Contact( "Unit1.Em4.ControlNodes".sideTapeAttachment."step".transition1[522] )
      { S7_Templates := "time_type := Time" } #statTonTime[522].TON(pt := T#0ms, et =>)
      Move(in := #JOB_5_STEP_30, out1 => "Unit1.Em4.ControlNodes".sideTapeAttachment.sequence.status.nextStep)
   END_RUNG
   // the same network as SCL:
   "Unit1.Em4.ControlNodes".sideTapeAttachment."step".action1[522] := ("Unit1.Em4.ControlNodes".sideTapeAttachment.sequence.status.currentStep = #JOB_5_STEP_22) AND "Unit1.Em4.ControlNodes".sideTapeAttachment.sequence.status.seqActive;
   "Unit1.Em4.ControlNodes".sideTapeAttachment."step".transition1[522] := ("Unit1.Em4.ControlNodes".sideTapeAttachment.sequence.status.currentStep = #JOB_5_STEP_22) AND "Unit1.Em4.ControlNodes".sideTapeAttachment.sequence.status.seqActive;
   #statTonTime[522].TON(IN := ("Unit1.Em4.ControlNodes".sideTapeAttachment.sequence.status.currentStep = #JOB_5_STEP_22) AND "Unit1.Em4.ControlNodes".sideTapeAttachment.sequence.status.seqActive AND "Unit1.Em4.ControlNodes".sideTapeAttachment."step".transition1[522],
                         PT := T#0ms);
   IF #statTonTime[522].Q THEN
       "Unit1.Em4.ControlNodes".sideTapeAttachment.sequence.status.nextStep := #JOB_5_STEP_30;
   END_IF;
END_REGION

REGION Network 65: Step[530] : Side Tape Attachment Right Backward
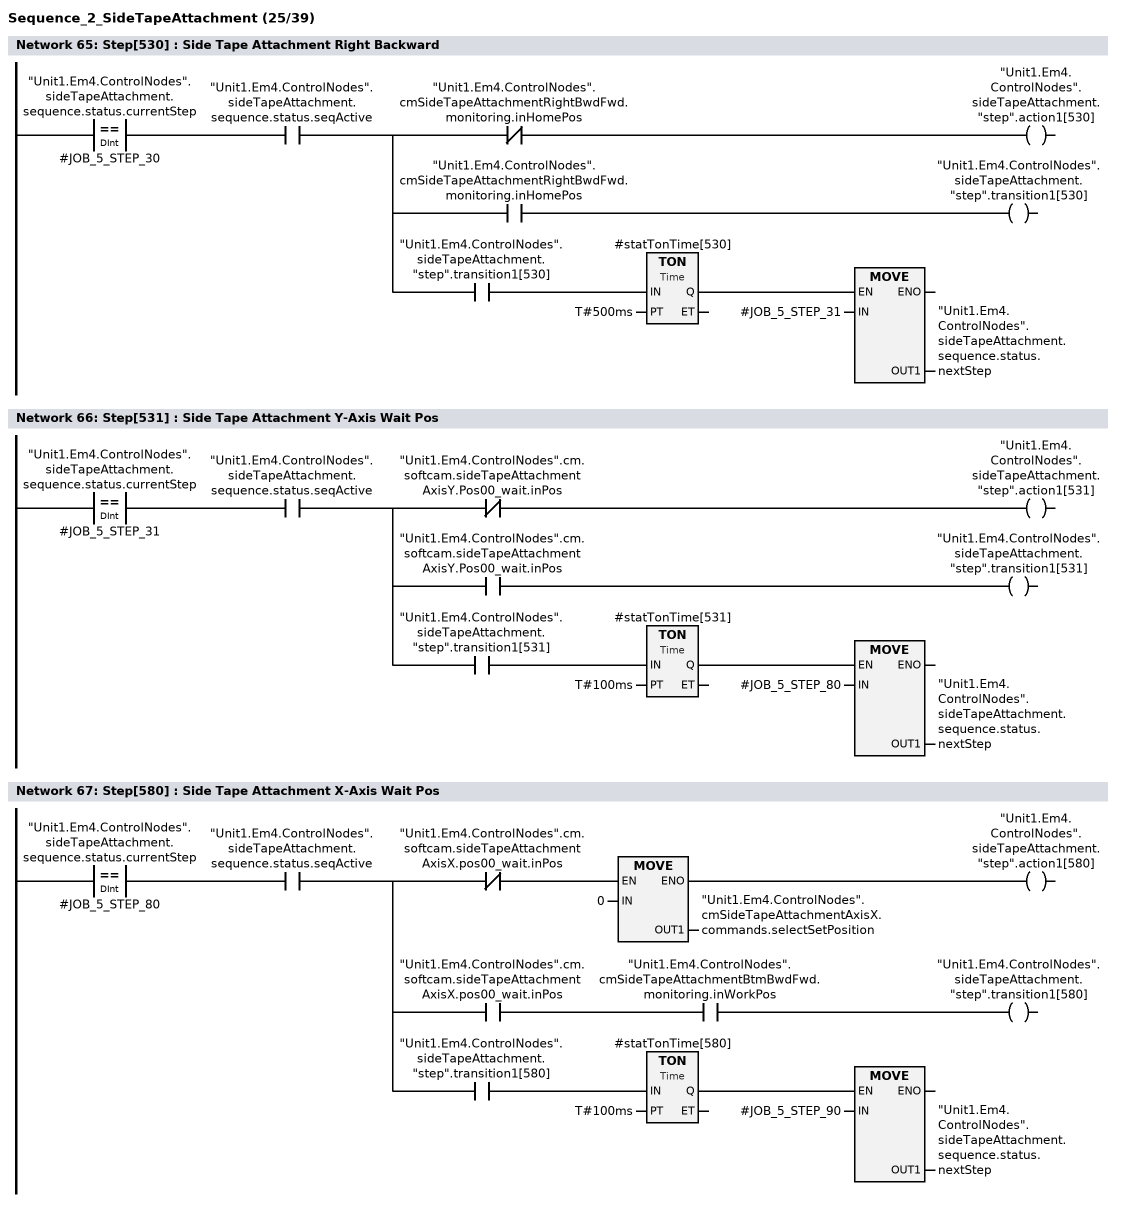
   RUNG wire#powerrail
      { S7_Templates := "SrcType := DInt" } EQ_Contact(in1 := "Unit1.Em4.ControlNodes".sideTapeAttachment.sequence.status.currentStep, in2 := #JOB_5_STEP_30)
      Contact( "Unit1.Em4.ControlNodes".sideTapeAttachment.sequence.status.seqActive )
      wire#w1
      I_Contact( "Unit1.Em4.ControlNodes".cmSideTapeAttachmentRightBwdFwd.monitoring.inHomePos )
      Coil( "Unit1.Em4.ControlNodes".sideTapeAttachment."step".action1[530] )
   END_RUNG
   RUNG wire#w1
      Contact( "Unit1.Em4.ControlNodes".cmSideTapeAttachmentRightBwdFwd.monitoring.inHomePos )
      Coil( "Unit1.Em4.ControlNodes".sideTapeAttachment."step".transition1[530] )
   END_RUNG
   RUNG wire#w1
      Contact( "Unit1.Em4.ControlNodes".sideTapeAttachment."step".transition1[530] )
      { S7_Templates := "time_type := Time" } #statTonTime[530].TON(pt := T#500ms, et =>)
      Move(in := #JOB_5_STEP_31, out1 => "Unit1.Em4.ControlNodes".sideTapeAttachment.sequence.status.nextStep)
   END_RUNG
   // the same network as SCL:
   #_w1 := ("Unit1.Em4.ControlNodes".sideTapeAttachment.sequence.status.currentStep = #JOB_5_STEP_30) AND "Unit1.Em4.ControlNodes".sideTapeAttachment.sequence.status.seqActive;
   "Unit1.Em4.ControlNodes".sideTapeAttachment."step".action1[530] := #_w1 AND NOT "Unit1.Em4.ControlNodes".cmSideTapeAttachmentRightBwdFwd.monitoring.inHomePos;
   "Unit1.Em4.ControlNodes".sideTapeAttachment."step".transition1[530] := #_w1 AND "Unit1.Em4.ControlNodes".cmSideTapeAttachmentRightBwdFwd.monitoring.inHomePos;
   #statTonTime[530].TON(IN := #_w1 AND "Unit1.Em4.ControlNodes".sideTapeAttachment."step".transition1[530],
                         PT := T#500ms);
   IF #statTonTime[530].Q THEN
       "Unit1.Em4.ControlNodes".sideTapeAttachment.sequence.status.nextStep := #JOB_5_STEP_31;
   END_IF;
END_REGION

REGION Network 66: Step[531] : Side Tape Attachment Y-Axis Wait Pos
   RUNG wire#powerrail
      { S7_Templates := "SrcType := DInt" } EQ_Contact(in1 := "Unit1.Em4.ControlNodes".sideTapeAttachment.sequence.status.currentStep, in2 := #JOB_5_STEP_31)
      Contact( "Unit1.Em4.ControlNodes".sideTapeAttachment.sequence.status.seqActive )
      wire#w1
      I_Contact( "Unit1.Em4.ControlNodes".cm.softcam.sideTapeAttachmentAxisY.Pos00_wait.inPos )
      Coil( "Unit1.Em4.ControlNodes".sideTapeAttachment."step".action1[531] )
   END_RUNG
   RUNG wire#w1
      Contact( "Unit1.Em4.ControlNodes".cm.softcam.sideTapeAttachmentAxisY.Pos00_wait.inPos )
      Coil( "Unit1.Em4.ControlNodes".sideTapeAttachment."step".transition1[531] )
   END_RUNG
   RUNG wire#w1
      Contact( "Unit1.Em4.ControlNodes".sideTapeAttachment."step".transition1[531] )
      { S7_Templates := "time_type := Time" } #statTonTime[531].TON(pt := T#100ms, et =>)
      Move(in := #JOB_5_STEP_80, out1 => "Unit1.Em4.ControlNodes".sideTapeAttachment.sequence.status.nextStep)
   END_RUNG
   // the same network as SCL:
   #_w1 := ("Unit1.Em4.ControlNodes".sideTapeAttachment.sequence.status.currentStep = #JOB_5_STEP_31) AND "Unit1.Em4.ControlNodes".sideTapeAttachment.sequence.status.seqActive;
   "Unit1.Em4.ControlNodes".sideTapeAttachment."step".action1[531] := #_w1 AND NOT "Unit1.Em4.ControlNodes".cm.softcam.sideTapeAttachmentAxisY.Pos00_wait.inPos;
   "Unit1.Em4.ControlNodes".sideTapeAttachment."step".transition1[531] := #_w1 AND "Unit1.Em4.ControlNodes".cm.softcam.sideTapeAttachmentAxisY.Pos00_wait.inPos;
   #statTonTime[531].TON(IN := #_w1 AND "Unit1.Em4.ControlNodes".sideTapeAttachment."step".transition1[531],
                         PT := T#100ms);
   IF #statTonTime[531].Q THEN
       "Unit1.Em4.ControlNodes".sideTapeAttachment.sequence.status.nextStep := #JOB_5_STEP_80;
   END_IF;
END_REGION

REGION Network 67: Step[580] : Side Tape Attachment X-Axis Wait Pos
   RUNG wire#powerrail
      { S7_Templates := "SrcType := DInt" } EQ_Contact(in1 := "Unit1.Em4.ControlNodes".sideTapeAttachment.sequence.status.currentStep, in2 := #JOB_5_STEP_80)
      Contact( "Unit1.Em4.ControlNodes".sideTapeAttachment.sequence.status.seqActive )
      wire#w1
      I_Contact( "Unit1.Em4.ControlNodes".cm.softcam.sideTapeAttachmentAxisX.pos00_wait.inPos )
      Move(in := 0, out1 => "Unit1.Em4.ControlNodes".cmSideTapeAttachmentAxisX.commands.selectSetPosition)
      Coil( "Unit1.Em4.ControlNodes".sideTapeAttachment."step".action1[580] )
   END_RUNG
   RUNG wire#w1
      Contact( "Unit1.Em4.ControlNodes".cm.softcam.sideTapeAttachmentAxisX.pos00_wait.inPos )
      Contact( "Unit1.Em4.ControlNodes".cmSideTapeAttachmentBtmBwdFwd.monitoring.inWorkPos )
      Coil( "Unit1.Em4.ControlNodes".sideTapeAttachment."step".transition1[580] )
   END_RUNG
   RUNG wire#w1
      Contact( "Unit1.Em4.ControlNodes".sideTapeAttachment."step".transition1[580] )
      { S7_Templates := "time_type := Time" } #statTonTime[580].TON(pt := T#100ms, et =>)
      Move(in := #JOB_5_STEP_90, out1 => "Unit1.Em4.ControlNodes".sideTapeAttachment.sequence.status.nextStep)
   END_RUNG
   // the same network as SCL:
   #_w1 := ("Unit1.Em4.ControlNodes".sideTapeAttachment.sequence.status.currentStep = #JOB_5_STEP_80) AND "Unit1.Em4.ControlNodes".sideTapeAttachment.sequence.status.seqActive;
   #_w2 := #_w1 AND NOT "Unit1.Em4.ControlNodes".cm.softcam.sideTapeAttachmentAxisX.pos00_wait.inPos;
   IF #_w2 THEN "Unit1.Em4.ControlNodes".cmSideTapeAttachmentAxisX.commands.selectSetPosition := 0; END_IF;
   "Unit1.Em4.ControlNodes".sideTapeAttachment."step".action1[580] := #_w2;
   "Unit1.Em4.ControlNodes".sideTapeAttachment."step".transition1[580] := #_w1 AND "Unit1.Em4.ControlNodes".cm.softcam.sideTapeAttachmentAxisX.pos00_wait.inPos AND "Unit1.Em4.ControlNodes".cmSideTapeAttachmentBtmBwdFwd.monitoring.inWorkPos;
   #statTonTime[580].TON(IN := #_w1 AND "Unit1.Em4.ControlNodes".sideTapeAttachment."step".transition1[580],
                         PT := T#100ms);
   IF #statTonTime[580].Q THEN
       "Unit1.Em4.ControlNodes".sideTapeAttachment.sequence.status.nextStep := #JOB_5_STEP_90;
   END_IF;
END_REGION

REGION Network 68: Step[590] : Job[5] Step End
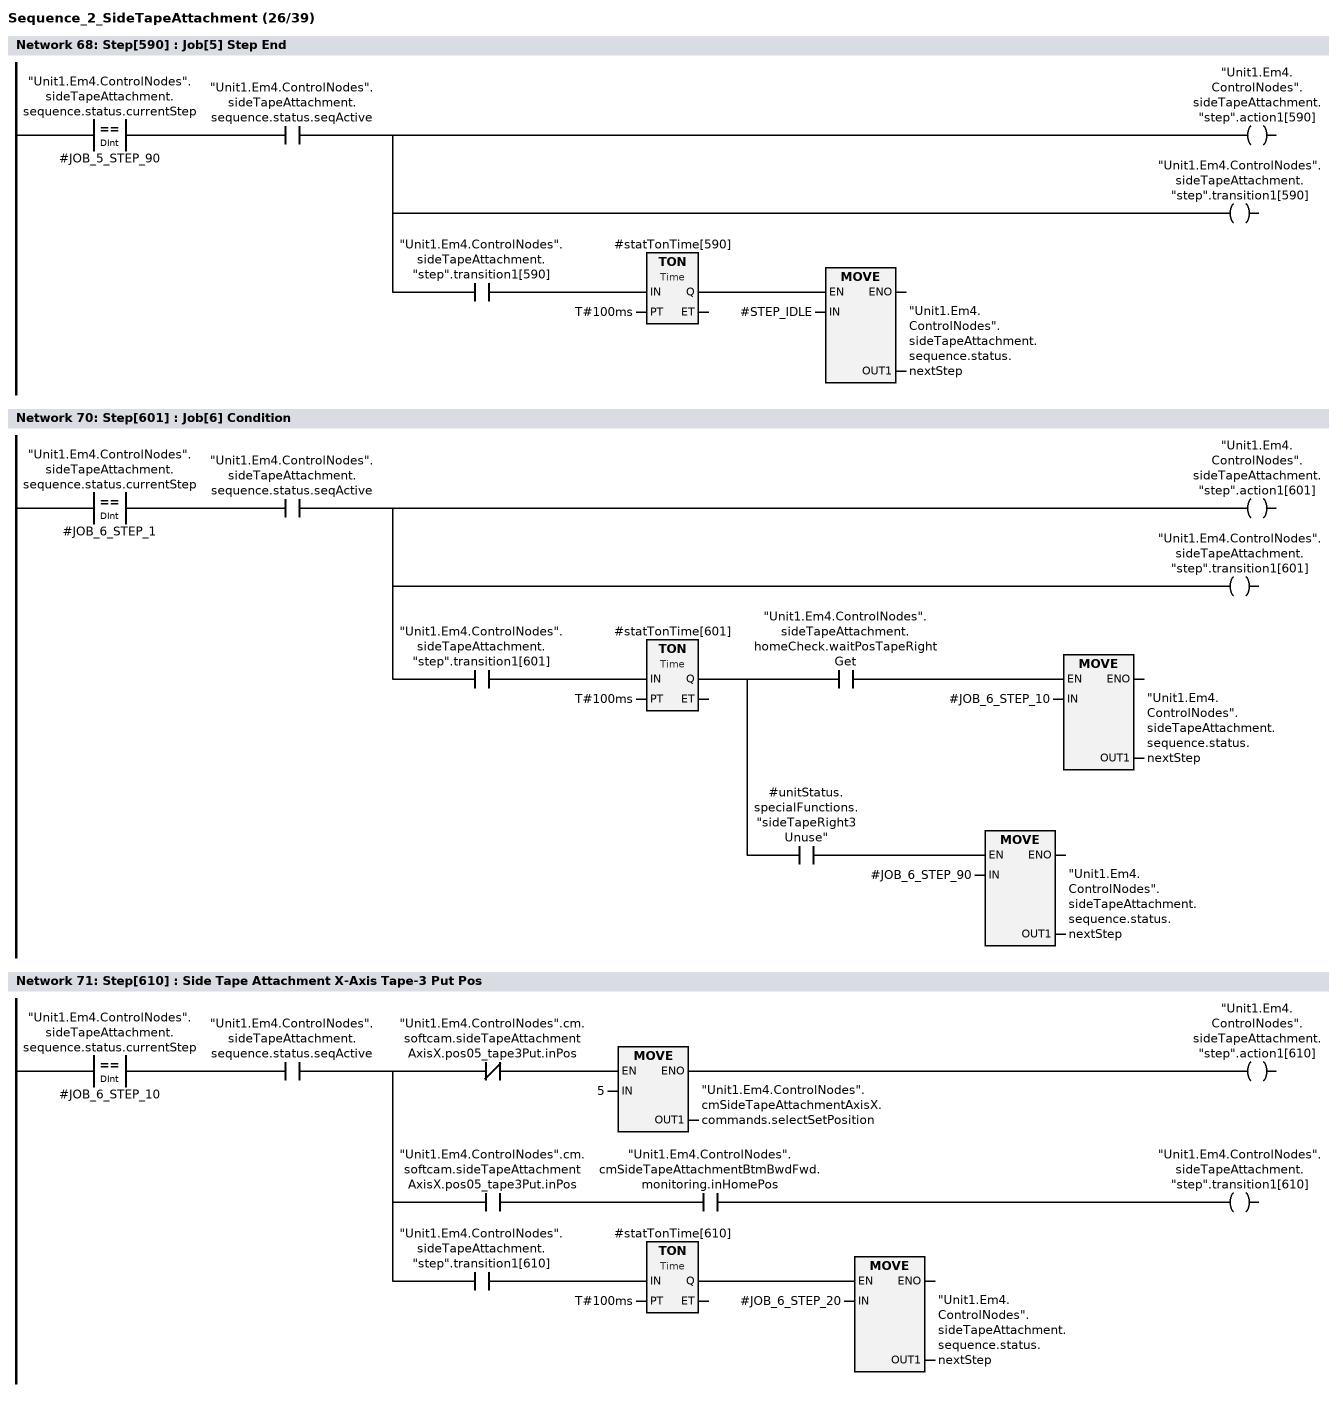
   RUNG wire#powerrail
      { S7_Templates := "SrcType := DInt" } EQ_Contact(in1 := "Unit1.Em4.ControlNodes".sideTapeAttachment.sequence.status.currentStep, in2 := #JOB_5_STEP_90)
      Contact( "Unit1.Em4.ControlNodes".sideTapeAttachment.sequence.status.seqActive )
      wire#w1
      Coil( "Unit1.Em4.ControlNodes".sideTapeAttachment."step".action1[590] )
   END_RUNG
   RUNG wire#w1
      Coil( "Unit1.Em4.ControlNodes".sideTapeAttachment."step".transition1[590] )
   END_RUNG
   RUNG wire#w1
      Contact( "Unit1.Em4.ControlNodes".sideTapeAttachment."step".transition1[590] )
      { S7_Templates := "time_type := Time" } #statTonTime[590].TON(pt := T#100ms, et =>)
      Move(in := #STEP_IDLE, out1 => "Unit1.Em4.ControlNodes".sideTapeAttachment.sequence.status.nextStep)
   END_RUNG
   // the same network as SCL:
   "Unit1.Em4.ControlNodes".sideTapeAttachment."step".action1[590] := ("Unit1.Em4.ControlNodes".sideTapeAttachment.sequence.status.currentStep = #JOB_5_STEP_90) AND "Unit1.Em4.ControlNodes".sideTapeAttachment.sequence.status.seqActive;
   "Unit1.Em4.ControlNodes".sideTapeAttachment."step".transition1[590] := ("Unit1.Em4.ControlNodes".sideTapeAttachment.sequence.status.currentStep = #JOB_5_STEP_90) AND "Unit1.Em4.ControlNodes".sideTapeAttachment.sequence.status.seqActive;
   #statTonTime[590].TON(IN := ("Unit1.Em4.ControlNodes".sideTapeAttachment.sequence.status.currentStep = #JOB_5_STEP_90) AND "Unit1.Em4.ControlNodes".sideTapeAttachment.sequence.status.seqActive AND "Unit1.Em4.ControlNodes".sideTapeAttachment."step".transition1[590],
                         PT := T#100ms);
   IF #statTonTime[590].Q THEN
       "Unit1.Em4.ControlNodes".sideTapeAttachment.sequence.status.nextStep := #STEP_IDLE;
   END_IF;
END_REGION

REGION Network 69: *************** JOB[6] SIDE TAPE PUT-3=AUTO *************************
END_REGION

REGION Network 70: Step[601] : Job[6] Condition
   RUNG wire#powerrail
      { S7_Templates := "SrcType := DInt" } EQ_Contact(in1 := "Unit1.Em4.ControlNodes".sideTapeAttachment.sequence.status.currentStep, in2 := #JOB_6_STEP_1)
      Contact( "Unit1.Em4.ControlNodes".sideTapeAttachment.sequence.status.seqActive )
      wire#w1
      Coil( "Unit1.Em4.ControlNodes".sideTapeAttachment."step".action1[601] )
   END_RUNG
   RUNG wire#w1
      Coil( "Unit1.Em4.ControlNodes".sideTapeAttachment."step".transition1[601] )
   END_RUNG
   RUNG wire#w1
      Contact( "Unit1.Em4.ControlNodes".sideTapeAttachment."step".transition1[601] )
      { S7_Templates := "time_type := Time" } #statTonTime[601].TON(pt := T#100ms, et =>)
      wire#w2
      Contact( "Unit1.Em4.ControlNodes".sideTapeAttachment.homeCheck.waitPosTapeRightGet )
      Move(in := #JOB_6_STEP_10, out1 => "Unit1.Em4.ControlNodes".sideTapeAttachment.sequence.status.nextStep)
   END_RUNG
   RUNG wire#w2
      Contact( #unitStatus.specialFunctions."sideTapeRight3 Unuse" )
      Move(in := #JOB_6_STEP_90, out1 => "Unit1.Em4.ControlNodes".sideTapeAttachment.sequence.status.nextStep)
   END_RUNG
   // the same network as SCL:
   "Unit1.Em4.ControlNodes".sideTapeAttachment."step".action1[601] := ("Unit1.Em4.ControlNodes".sideTapeAttachment.sequence.status.currentStep = #JOB_6_STEP_1) AND "Unit1.Em4.ControlNodes".sideTapeAttachment.sequence.status.seqActive;
   "Unit1.Em4.ControlNodes".sideTapeAttachment."step".transition1[601] := ("Unit1.Em4.ControlNodes".sideTapeAttachment.sequence.status.currentStep = #JOB_6_STEP_1) AND "Unit1.Em4.ControlNodes".sideTapeAttachment.sequence.status.seqActive;
   #statTonTime[601].TON(IN := ("Unit1.Em4.ControlNodes".sideTapeAttachment.sequence.status.currentStep = #JOB_6_STEP_1) AND "Unit1.Em4.ControlNodes".sideTapeAttachment.sequence.status.seqActive AND "Unit1.Em4.ControlNodes".sideTapeAttachment."step".transition1[601],
                         PT := T#100ms);
   IF #statTonTime[601].Q AND "Unit1.Em4.ControlNodes".sideTapeAttachment.homeCheck.waitPosTapeRightGet THEN
       "Unit1.Em4.ControlNodes".sideTapeAttachment.sequence.status.nextStep := #JOB_6_STEP_10;
   END_IF;
   IF #statTonTime[601].Q AND #unitStatus.specialFunctions."sideTapeRight3 Unuse" THEN
       "Unit1.Em4.ControlNodes".sideTapeAttachment.sequence.status.nextStep := #JOB_6_STEP_90;
   END_IF;
END_REGION

REGION Network 71: Step[610] : Side Tape Attachment X-Axis Tape-3 Put Pos
   RUNG wire#powerrail
      { S7_Templates := "SrcType := DInt" } EQ_Contact(in1 := "Unit1.Em4.ControlNodes".sideTapeAttachment.sequence.status.currentStep, in2 := #JOB_6_STEP_10)
      Contact( "Unit1.Em4.ControlNodes".sideTapeAttachment.sequence.status.seqActive )
      wire#w1
      I_Contact( "Unit1.Em4.ControlNodes".cm.softcam.sideTapeAttachmentAxisX.pos05_tape3Put.inPos )
      Move(in := 5, out1 => "Unit1.Em4.ControlNodes".cmSideTapeAttachmentAxisX.commands.selectSetPosition)
      Coil( "Unit1.Em4.ControlNodes".sideTapeAttachment."step".action1[610] )
   END_RUNG
   RUNG wire#w1
      Contact( "Unit1.Em4.ControlNodes".cm.softcam.sideTapeAttachmentAxisX.pos05_tape3Put.inPos )
      Contact( "Unit1.Em4.ControlNodes".cmSideTapeAttachmentBtmBwdFwd.monitoring.inHomePos )
      Coil( "Unit1.Em4.ControlNodes".sideTapeAttachment."step".transition1[610] )
   END_RUNG
   RUNG wire#w1
      Contact( "Unit1.Em4.ControlNodes".sideTapeAttachment."step".transition1[610] )
      { S7_Templates := "time_type := Time" } #statTonTime[610].TON(pt := T#100ms, et =>)
      Move(in := #JOB_6_STEP_20, out1 => "Unit1.Em4.ControlNodes".sideTapeAttachment.sequence.status.nextStep)
   END_RUNG
   // the same network as SCL:
   #_w1 := ("Unit1.Em4.ControlNodes".sideTapeAttachment.sequence.status.currentStep = #JOB_6_STEP_10) AND "Unit1.Em4.ControlNodes".sideTapeAttachment.sequence.status.seqActive;
   #_w2 := #_w1 AND NOT "Unit1.Em4.ControlNodes".cm.softcam.sideTapeAttachmentAxisX.pos05_tape3Put.inPos;
   IF #_w2 THEN "Unit1.Em4.ControlNodes".cmSideTapeAttachmentAxisX.commands.selectSetPosition := 5; END_IF;
   "Unit1.Em4.ControlNodes".sideTapeAttachment."step".action1[610] := #_w2;
   "Unit1.Em4.ControlNodes".sideTapeAttachment."step".transition1[610] := #_w1 AND "Unit1.Em4.ControlNodes".cm.softcam.sideTapeAttachmentAxisX.pos05_tape3Put.inPos AND "Unit1.Em4.ControlNodes".cmSideTapeAttachmentBtmBwdFwd.monitoring.inHomePos;
   #statTonTime[610].TON(IN := #_w1 AND "Unit1.Em4.ControlNodes".sideTapeAttachment."step".transition1[610],
                         PT := T#100ms);
   IF #statTonTime[610].Q THEN
       "Unit1.Em4.ControlNodes".sideTapeAttachment.sequence.status.nextStep := #JOB_6_STEP_20;
   END_IF;
END_REGION

REGION Network 72: Step[620] : Side tape Attachment Y-Axis Tape-3 Put Pos
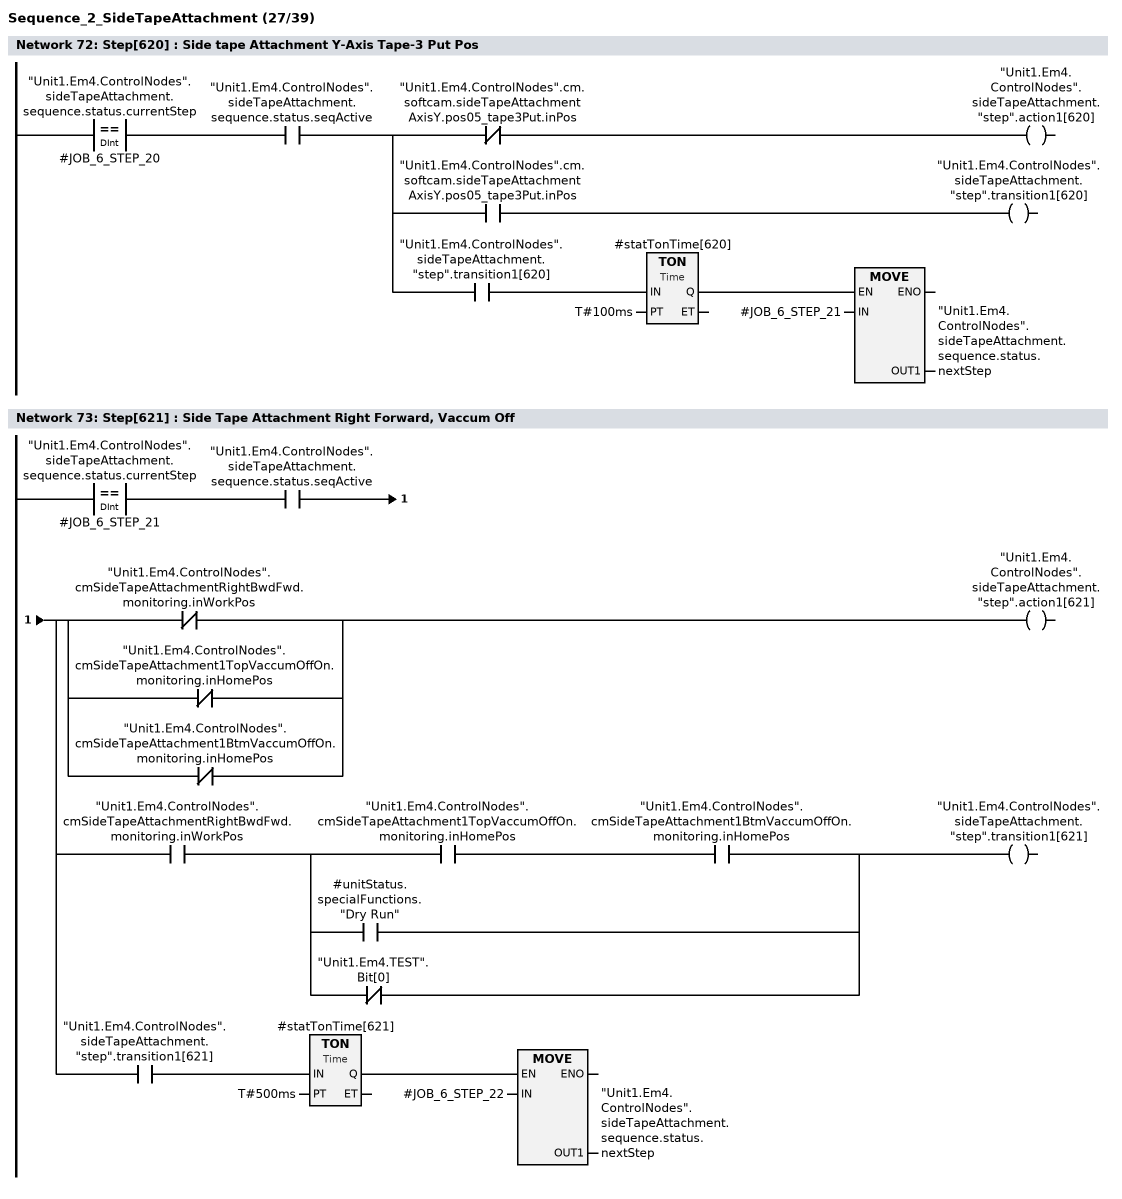
   RUNG wire#powerrail
      { S7_Templates := "SrcType := DInt" } EQ_Contact(in1 := "Unit1.Em4.ControlNodes".sideTapeAttachment.sequence.status.currentStep, in2 := #JOB_6_STEP_20)
      Contact( "Unit1.Em4.ControlNodes".sideTapeAttachment.sequence.status.seqActive )
      wire#w1
      I_Contact( "Unit1.Em4.ControlNodes".cm.softcam.sideTapeAttachmentAxisY.pos05_tape3Put.inPos )
      Coil( "Unit1.Em4.ControlNodes".sideTapeAttachment."step".action1[620] )
   END_RUNG
   RUNG wire#w1
      Contact( "Unit1.Em4.ControlNodes".cm.softcam.sideTapeAttachmentAxisY.pos05_tape3Put.inPos )
      Coil( "Unit1.Em4.ControlNodes".sideTapeAttachment."step".transition1[620] )
   END_RUNG
   RUNG wire#w1
      Contact( "Unit1.Em4.ControlNodes".sideTapeAttachment."step".transition1[620] )
      { S7_Templates := "time_type := Time" } #statTonTime[620].TON(pt := T#100ms, et =>)
      Move(in := #JOB_6_STEP_21, out1 => "Unit1.Em4.ControlNodes".sideTapeAttachment.sequence.status.nextStep)
   END_RUNG
   // the same network as SCL:
   #_w1 := ("Unit1.Em4.ControlNodes".sideTapeAttachment.sequence.status.currentStep = #JOB_6_STEP_20) AND "Unit1.Em4.ControlNodes".sideTapeAttachment.sequence.status.seqActive;
   "Unit1.Em4.ControlNodes".sideTapeAttachment."step".action1[620] := #_w1 AND NOT "Unit1.Em4.ControlNodes".cm.softcam.sideTapeAttachmentAxisY.pos05_tape3Put.inPos;
   "Unit1.Em4.ControlNodes".sideTapeAttachment."step".transition1[620] := #_w1 AND "Unit1.Em4.ControlNodes".cm.softcam.sideTapeAttachmentAxisY.pos05_tape3Put.inPos;
   #statTonTime[620].TON(IN := #_w1 AND "Unit1.Em4.ControlNodes".sideTapeAttachment."step".transition1[620],
                         PT := T#100ms);
   IF #statTonTime[620].Q THEN
       "Unit1.Em4.ControlNodes".sideTapeAttachment.sequence.status.nextStep := #JOB_6_STEP_21;
   END_IF;
END_REGION

REGION Network 73: Step[621] : Side Tape Attachment Right Forward, Vaccum Off
   RUNG wire#powerrail
      { S7_Templates := "SrcType := DInt" } EQ_Contact(in1 := "Unit1.Em4.ControlNodes".sideTapeAttachment.sequence.status.currentStep, in2 := #JOB_6_STEP_21)
      Contact( "Unit1.Em4.ControlNodes".sideTapeAttachment.sequence.status.seqActive )
      wire#w1
      I_Contact( "Unit1.Em4.ControlNodes".cmSideTapeAttachmentRightBwdFwd.monitoring.inWorkPos )
      wire#w2
      Coil( "Unit1.Em4.ControlNodes".sideTapeAttachment."step".action1[621] )
   END_RUNG
   RUNG wire#w1
      I_Contact( "Unit1.Em4.ControlNodes".cmSideTapeAttachment1TopVaccumOffOn.monitoring.inHomePos )
   END_RUNG wire#w2
   RUNG wire#w1
      I_Contact( "Unit1.Em4.ControlNodes".cmSideTapeAttachment1BtmVaccumOffOn.monitoring.inHomePos )
   END_RUNG wire#w2
   RUNG wire#w1
      Contact( "Unit1.Em4.ControlNodes".cmSideTapeAttachmentRightBwdFwd.monitoring.inWorkPos )
      wire#w3
      Contact( "Unit1.Em4.ControlNodes".cmSideTapeAttachment1TopVaccumOffOn.monitoring.inHomePos )
      Contact( "Unit1.Em4.ControlNodes".cmSideTapeAttachment1BtmVaccumOffOn.monitoring.inHomePos )
      wire#w4
      Coil( "Unit1.Em4.ControlNodes".sideTapeAttachment."step".transition1[621] )
   END_RUNG
   RUNG wire#w3
      Contact( #unitStatus.specialFunctions."Dry Run" )
   END_RUNG wire#w4
   RUNG wire#w3
      I_Contact( "Unit1.Em4.TEST".Bit[0] )
   END_RUNG wire#w4
   RUNG wire#w1
      Contact( "Unit1.Em4.ControlNodes".sideTapeAttachment."step".transition1[621] )
      { S7_Templates := "time_type := Time" } #statTonTime[621].TON(pt := T#500ms, et =>)
      Move(in := #JOB_6_STEP_22, out1 => "Unit1.Em4.ControlNodes".sideTapeAttachment.sequence.status.nextStep)
   END_RUNG
   // the same network as SCL:
   #_w1 := ("Unit1.Em4.ControlNodes".sideTapeAttachment.sequence.status.currentStep = #JOB_6_STEP_21) AND "Unit1.Em4.ControlNodes".sideTapeAttachment.sequence.status.seqActive;
   "Unit1.Em4.ControlNodes".sideTapeAttachment."step".action1[621] := #_w1 AND (NOT "Unit1.Em4.ControlNodes".cmSideTapeAttachmentRightBwdFwd.monitoring.inWorkPos OR NOT "Unit1.Em4.ControlNodes".cmSideTapeAttachment1TopVaccumOffOn.monitoring.inHomePos OR NOT "Unit1.Em4.ControlNodes".cmSideTapeAttachment1BtmVaccumOffOn.monitoring.inHomePos);
   "Unit1.Em4.ControlNodes".sideTapeAttachment."step".transition1[621] := #_w1 AND "Unit1.Em4.ControlNodes".cmSideTapeAttachmentRightBwdFwd.monitoring.inWorkPos AND (("Unit1.Em4.ControlNodes".cmSideTapeAttachment1TopVaccumOffOn.monitoring.inHomePos AND "Unit1.Em4.ControlNodes".cmSideTapeAttachment1BtmVaccumOffOn.monitoring.inHomePos) OR #unitStatus.specialFunctions."Dry Run" OR NOT "Unit1.Em4.TEST".Bit[0]);
   #statTonTime[621].TON(IN := #_w1 AND "Unit1.Em4.ControlNodes".sideTapeAttachment."step".transition1[621],
                         PT := T#500ms);
   IF #statTonTime[621].Q THEN
       "Unit1.Em4.ControlNodes".sideTapeAttachment.sequence.status.nextStep := #JOB_6_STEP_22;
   END_IF;
END_REGION

REGION Network 74: Step[622] : Spare
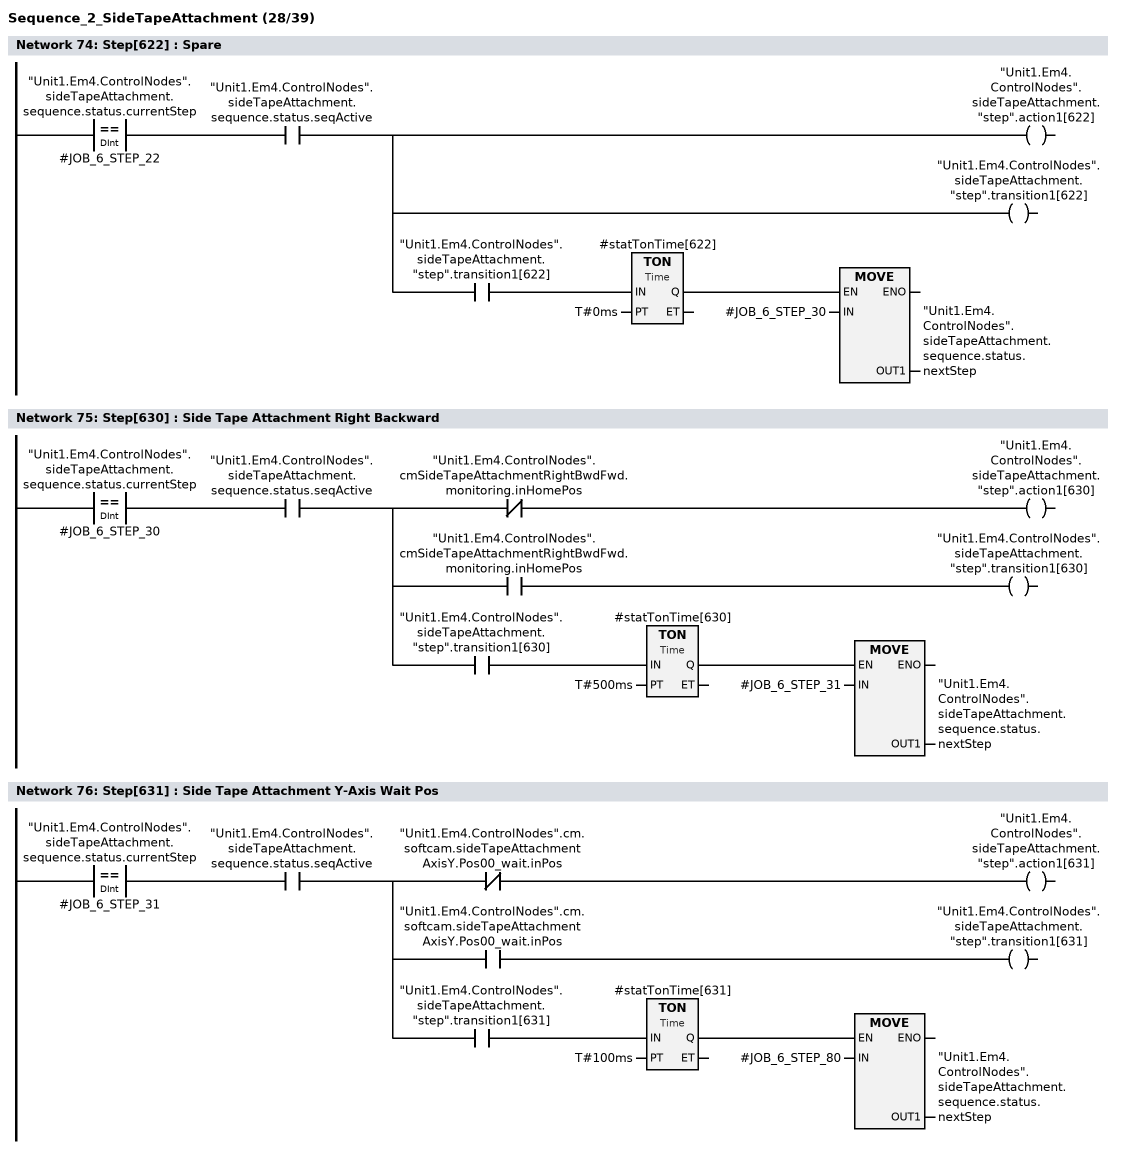
   RUNG wire#powerrail
      { S7_Templates := "SrcType := DInt" } EQ_Contact(in1 := "Unit1.Em4.ControlNodes".sideTapeAttachment.sequence.status.currentStep, in2 := #JOB_6_STEP_22)
      Contact( "Unit1.Em4.ControlNodes".sideTapeAttachment.sequence.status.seqActive )
      wire#w1
      Coil( "Unit1.Em4.ControlNodes".sideTapeAttachment."step".action1[622] )
   END_RUNG
   RUNG wire#w1
      Coil( "Unit1.Em4.ControlNodes".sideTapeAttachment."step".transition1[622] )
   END_RUNG
   RUNG wire#w1
      Contact( "Unit1.Em4.ControlNodes".sideTapeAttachment."step".transition1[622] )
      { S7_Templates := "time_type := Time" } #statTonTime[622].TON(pt := T#0ms, et =>)
      Move(in := #JOB_6_STEP_30, out1 => "Unit1.Em4.ControlNodes".sideTapeAttachment.sequence.status.nextStep)
   END_RUNG
   // the same network as SCL:
   "Unit1.Em4.ControlNodes".sideTapeAttachment."step".action1[622] := ("Unit1.Em4.ControlNodes".sideTapeAttachment.sequence.status.currentStep = #JOB_6_STEP_22) AND "Unit1.Em4.ControlNodes".sideTapeAttachment.sequence.status.seqActive;
   "Unit1.Em4.ControlNodes".sideTapeAttachment."step".transition1[622] := ("Unit1.Em4.ControlNodes".sideTapeAttachment.sequence.status.currentStep = #JOB_6_STEP_22) AND "Unit1.Em4.ControlNodes".sideTapeAttachment.sequence.status.seqActive;
   #statTonTime[622].TON(IN := ("Unit1.Em4.ControlNodes".sideTapeAttachment.sequence.status.currentStep = #JOB_6_STEP_22) AND "Unit1.Em4.ControlNodes".sideTapeAttachment.sequence.status.seqActive AND "Unit1.Em4.ControlNodes".sideTapeAttachment."step".transition1[622],
                         PT := T#0ms);
   IF #statTonTime[622].Q THEN
       "Unit1.Em4.ControlNodes".sideTapeAttachment.sequence.status.nextStep := #JOB_6_STEP_30;
   END_IF;
END_REGION

REGION Network 75: Step[630] : Side Tape Attachment Right Backward
   RUNG wire#powerrail
      { S7_Templates := "SrcType := DInt" } EQ_Contact(in1 := "Unit1.Em4.ControlNodes".sideTapeAttachment.sequence.status.currentStep, in2 := #JOB_6_STEP_30)
      Contact( "Unit1.Em4.ControlNodes".sideTapeAttachment.sequence.status.seqActive )
      wire#w1
      I_Contact( "Unit1.Em4.ControlNodes".cmSideTapeAttachmentRightBwdFwd.monitoring.inHomePos )
      Coil( "Unit1.Em4.ControlNodes".sideTapeAttachment."step".action1[630] )
   END_RUNG
   RUNG wire#w1
      Contact( "Unit1.Em4.ControlNodes".cmSideTapeAttachmentRightBwdFwd.monitoring.inHomePos )
      Coil( "Unit1.Em4.ControlNodes".sideTapeAttachment."step".transition1[630] )
   END_RUNG
   RUNG wire#w1
      Contact( "Unit1.Em4.ControlNodes".sideTapeAttachment."step".transition1[630] )
      { S7_Templates := "time_type := Time" } #statTonTime[630].TON(pt := T#500ms, et =>)
      Move(in := #JOB_6_STEP_31, out1 => "Unit1.Em4.ControlNodes".sideTapeAttachment.sequence.status.nextStep)
   END_RUNG
   // the same network as SCL:
   #_w1 := ("Unit1.Em4.ControlNodes".sideTapeAttachment.sequence.status.currentStep = #JOB_6_STEP_30) AND "Unit1.Em4.ControlNodes".sideTapeAttachment.sequence.status.seqActive;
   "Unit1.Em4.ControlNodes".sideTapeAttachment."step".action1[630] := #_w1 AND NOT "Unit1.Em4.ControlNodes".cmSideTapeAttachmentRightBwdFwd.monitoring.inHomePos;
   "Unit1.Em4.ControlNodes".sideTapeAttachment."step".transition1[630] := #_w1 AND "Unit1.Em4.ControlNodes".cmSideTapeAttachmentRightBwdFwd.monitoring.inHomePos;
   #statTonTime[630].TON(IN := #_w1 AND "Unit1.Em4.ControlNodes".sideTapeAttachment."step".transition1[630],
                         PT := T#500ms);
   IF #statTonTime[630].Q THEN
       "Unit1.Em4.ControlNodes".sideTapeAttachment.sequence.status.nextStep := #JOB_6_STEP_31;
   END_IF;
END_REGION

REGION Network 76: Step[631] : Side Tape Attachment Y-Axis Wait Pos
   RUNG wire#powerrail
      { S7_Templates := "SrcType := DInt" } EQ_Contact(in1 := "Unit1.Em4.ControlNodes".sideTapeAttachment.sequence.status.currentStep, in2 := #JOB_6_STEP_31)
      Contact( "Unit1.Em4.ControlNodes".sideTapeAttachment.sequence.status.seqActive )
      wire#w1
      I_Contact( "Unit1.Em4.ControlNodes".cm.softcam.sideTapeAttachmentAxisY.Pos00_wait.inPos )
      Coil( "Unit1.Em4.ControlNodes".sideTapeAttachment."step".action1[631] )
   END_RUNG
   RUNG wire#w1
      Contact( "Unit1.Em4.ControlNodes".cm.softcam.sideTapeAttachmentAxisY.Pos00_wait.inPos )
      Coil( "Unit1.Em4.ControlNodes".sideTapeAttachment."step".transition1[631] )
   END_RUNG
   RUNG wire#w1
      Contact( "Unit1.Em4.ControlNodes".sideTapeAttachment."step".transition1[631] )
      { S7_Templates := "time_type := Time" } #statTonTime[631].TON(pt := T#100ms, et =>)
      Move(in := #JOB_6_STEP_80, out1 => "Unit1.Em4.ControlNodes".sideTapeAttachment.sequence.status.nextStep)
   END_RUNG
   // the same network as SCL:
   #_w1 := ("Unit1.Em4.ControlNodes".sideTapeAttachment.sequence.status.currentStep = #JOB_6_STEP_31) AND "Unit1.Em4.ControlNodes".sideTapeAttachment.sequence.status.seqActive;
   "Unit1.Em4.ControlNodes".sideTapeAttachment."step".action1[631] := #_w1 AND NOT "Unit1.Em4.ControlNodes".cm.softcam.sideTapeAttachmentAxisY.Pos00_wait.inPos;
   "Unit1.Em4.ControlNodes".sideTapeAttachment."step".transition1[631] := #_w1 AND "Unit1.Em4.ControlNodes".cm.softcam.sideTapeAttachmentAxisY.Pos00_wait.inPos;
   #statTonTime[631].TON(IN := #_w1 AND "Unit1.Em4.ControlNodes".sideTapeAttachment."step".transition1[631],
                         PT := T#100ms);
   IF #statTonTime[631].Q THEN
       "Unit1.Em4.ControlNodes".sideTapeAttachment.sequence.status.nextStep := #JOB_6_STEP_80;
   END_IF;
END_REGION

REGION Network 77: Step[680] : Side Tape Attachment X-Axis Wait Pos
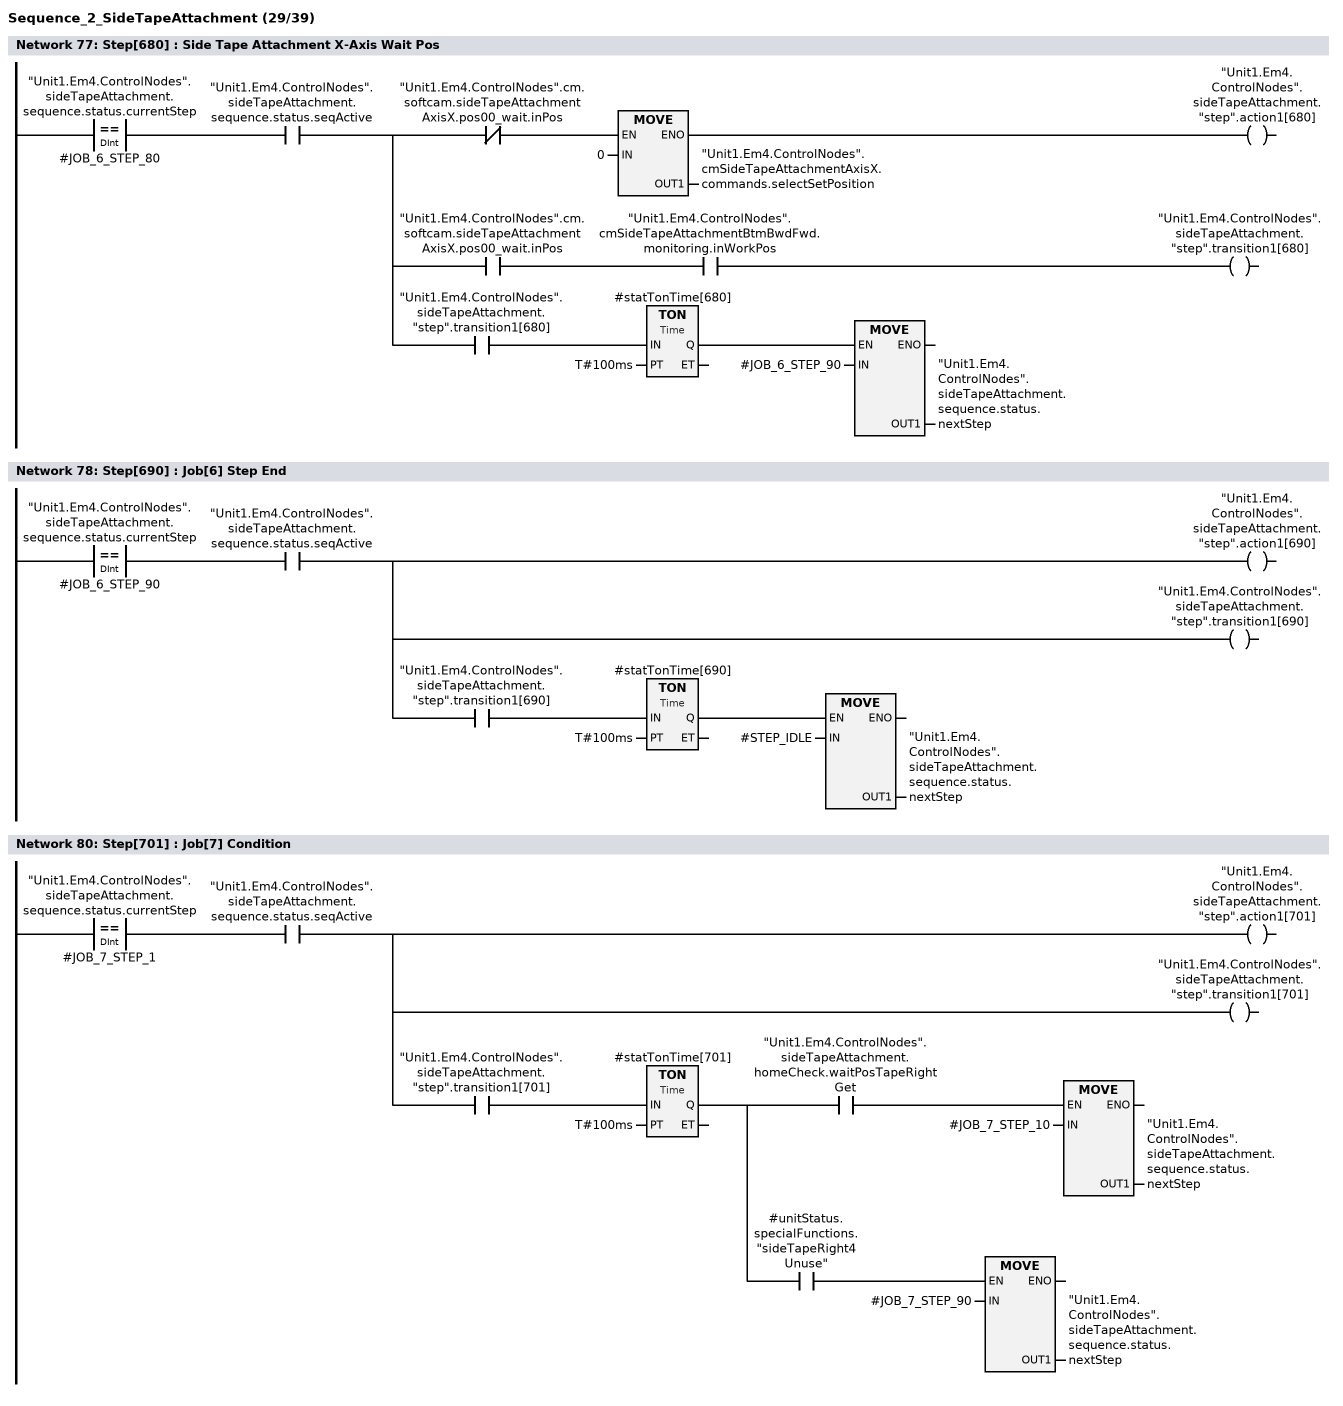
   RUNG wire#powerrail
      { S7_Templates := "SrcType := DInt" } EQ_Contact(in1 := "Unit1.Em4.ControlNodes".sideTapeAttachment.sequence.status.currentStep, in2 := #JOB_6_STEP_80)
      Contact( "Unit1.Em4.ControlNodes".sideTapeAttachment.sequence.status.seqActive )
      wire#w1
      I_Contact( "Unit1.Em4.ControlNodes".cm.softcam.sideTapeAttachmentAxisX.pos00_wait.inPos )
      Move(in := 0, out1 => "Unit1.Em4.ControlNodes".cmSideTapeAttachmentAxisX.commands.selectSetPosition)
      Coil( "Unit1.Em4.ControlNodes".sideTapeAttachment."step".action1[680] )
   END_RUNG
   RUNG wire#w1
      Contact( "Unit1.Em4.ControlNodes".cm.softcam.sideTapeAttachmentAxisX.pos00_wait.inPos )
      Contact( "Unit1.Em4.ControlNodes".cmSideTapeAttachmentBtmBwdFwd.monitoring.inWorkPos )
      Coil( "Unit1.Em4.ControlNodes".sideTapeAttachment."step".transition1[680] )
   END_RUNG
   RUNG wire#w1
      Contact( "Unit1.Em4.ControlNodes".sideTapeAttachment."step".transition1[680] )
      { S7_Templates := "time_type := Time" } #statTonTime[680].TON(pt := T#100ms, et =>)
      Move(in := #JOB_6_STEP_90, out1 => "Unit1.Em4.ControlNodes".sideTapeAttachment.sequence.status.nextStep)
   END_RUNG
   // the same network as SCL:
   #_w1 := ("Unit1.Em4.ControlNodes".sideTapeAttachment.sequence.status.currentStep = #JOB_6_STEP_80) AND "Unit1.Em4.ControlNodes".sideTapeAttachment.sequence.status.seqActive;
   #_w2 := #_w1 AND NOT "Unit1.Em4.ControlNodes".cm.softcam.sideTapeAttachmentAxisX.pos00_wait.inPos;
   IF #_w2 THEN "Unit1.Em4.ControlNodes".cmSideTapeAttachmentAxisX.commands.selectSetPosition := 0; END_IF;
   "Unit1.Em4.ControlNodes".sideTapeAttachment."step".action1[680] := #_w2;
   "Unit1.Em4.ControlNodes".sideTapeAttachment."step".transition1[680] := #_w1 AND "Unit1.Em4.ControlNodes".cm.softcam.sideTapeAttachmentAxisX.pos00_wait.inPos AND "Unit1.Em4.ControlNodes".cmSideTapeAttachmentBtmBwdFwd.monitoring.inWorkPos;
   #statTonTime[680].TON(IN := #_w1 AND "Unit1.Em4.ControlNodes".sideTapeAttachment."step".transition1[680],
                         PT := T#100ms);
   IF #statTonTime[680].Q THEN
       "Unit1.Em4.ControlNodes".sideTapeAttachment.sequence.status.nextStep := #JOB_6_STEP_90;
   END_IF;
END_REGION

REGION Network 78: Step[690] : Job[6] Step End
   RUNG wire#powerrail
      { S7_Templates := "SrcType := DInt" } EQ_Contact(in1 := "Unit1.Em4.ControlNodes".sideTapeAttachment.sequence.status.currentStep, in2 := #JOB_6_STEP_90)
      Contact( "Unit1.Em4.ControlNodes".sideTapeAttachment.sequence.status.seqActive )
      wire#w1
      Coil( "Unit1.Em4.ControlNodes".sideTapeAttachment."step".action1[690] )
   END_RUNG
   RUNG wire#w1
      Coil( "Unit1.Em4.ControlNodes".sideTapeAttachment."step".transition1[690] )
   END_RUNG
   RUNG wire#w1
      Contact( "Unit1.Em4.ControlNodes".sideTapeAttachment."step".transition1[690] )
      { S7_Templates := "time_type := Time" } #statTonTime[690].TON(pt := T#100ms, et =>)
      Move(in := #STEP_IDLE, out1 => "Unit1.Em4.ControlNodes".sideTapeAttachment.sequence.status.nextStep)
   END_RUNG
   // the same network as SCL:
   "Unit1.Em4.ControlNodes".sideTapeAttachment."step".action1[690] := ("Unit1.Em4.ControlNodes".sideTapeAttachment.sequence.status.currentStep = #JOB_6_STEP_90) AND "Unit1.Em4.ControlNodes".sideTapeAttachment.sequence.status.seqActive;
   "Unit1.Em4.ControlNodes".sideTapeAttachment."step".transition1[690] := ("Unit1.Em4.ControlNodes".sideTapeAttachment.sequence.status.currentStep = #JOB_6_STEP_90) AND "Unit1.Em4.ControlNodes".sideTapeAttachment.sequence.status.seqActive;
   #statTonTime[690].TON(IN := ("Unit1.Em4.ControlNodes".sideTapeAttachment.sequence.status.currentStep = #JOB_6_STEP_90) AND "Unit1.Em4.ControlNodes".sideTapeAttachment.sequence.status.seqActive AND "Unit1.Em4.ControlNodes".sideTapeAttachment."step".transition1[690],
                         PT := T#100ms);
   IF #statTonTime[690].Q THEN
       "Unit1.Em4.ControlNodes".sideTapeAttachment.sequence.status.nextStep := #STEP_IDLE;
   END_IF;
END_REGION

REGION Network 79: *************** JOB[7] SIDE TAPE PUT-4=AUTO *************************
END_REGION

REGION Network 80: Step[701] : Job[7] Condition
   RUNG wire#powerrail
      { S7_Templates := "SrcType := DInt" } EQ_Contact(in1 := "Unit1.Em4.ControlNodes".sideTapeAttachment.sequence.status.currentStep, in2 := #JOB_7_STEP_1)
      Contact( "Unit1.Em4.ControlNodes".sideTapeAttachment.sequence.status.seqActive )
      wire#w1
      Coil( "Unit1.Em4.ControlNodes".sideTapeAttachment."step".action1[701] )
   END_RUNG
   RUNG wire#w1
      Coil( "Unit1.Em4.ControlNodes".sideTapeAttachment."step".transition1[701] )
   END_RUNG
   RUNG wire#w1
      Contact( "Unit1.Em4.ControlNodes".sideTapeAttachment."step".transition1[701] )
      { S7_Templates := "time_type := Time" } #statTonTime[701].TON(pt := T#100ms, et =>)
      wire#w2
      Contact( "Unit1.Em4.ControlNodes".sideTapeAttachment.homeCheck.waitPosTapeRightGet )
      Move(in := #JOB_7_STEP_10, out1 => "Unit1.Em4.ControlNodes".sideTapeAttachment.sequence.status.nextStep)
   END_RUNG
   RUNG wire#w2
      Contact( #unitStatus.specialFunctions."sideTapeRight4 Unuse" )
      Move(in := #JOB_7_STEP_90, out1 => "Unit1.Em4.ControlNodes".sideTapeAttachment.sequence.status.nextStep)
   END_RUNG
   // the same network as SCL:
   "Unit1.Em4.ControlNodes".sideTapeAttachment."step".action1[701] := ("Unit1.Em4.ControlNodes".sideTapeAttachment.sequence.status.currentStep = #JOB_7_STEP_1) AND "Unit1.Em4.ControlNodes".sideTapeAttachment.sequence.status.seqActive;
   "Unit1.Em4.ControlNodes".sideTapeAttachment."step".transition1[701] := ("Unit1.Em4.ControlNodes".sideTapeAttachment.sequence.status.currentStep = #JOB_7_STEP_1) AND "Unit1.Em4.ControlNodes".sideTapeAttachment.sequence.status.seqActive;
   #statTonTime[701].TON(IN := ("Unit1.Em4.ControlNodes".sideTapeAttachment.sequence.status.currentStep = #JOB_7_STEP_1) AND "Unit1.Em4.ControlNodes".sideTapeAttachment.sequence.status.seqActive AND "Unit1.Em4.ControlNodes".sideTapeAttachment."step".transition1[701],
                         PT := T#100ms);
   IF #statTonTime[701].Q AND "Unit1.Em4.ControlNodes".sideTapeAttachment.homeCheck.waitPosTapeRightGet THEN
       "Unit1.Em4.ControlNodes".sideTapeAttachment.sequence.status.nextStep := #JOB_7_STEP_10;
   END_IF;
   IF #statTonTime[701].Q AND #unitStatus.specialFunctions."sideTapeRight4 Unuse" THEN
       "Unit1.Em4.ControlNodes".sideTapeAttachment.sequence.status.nextStep := #JOB_7_STEP_90;
   END_IF;
END_REGION

REGION Network 81: Step[710] : Side Tape Attachment X-Axis Tape-4 Put Pos
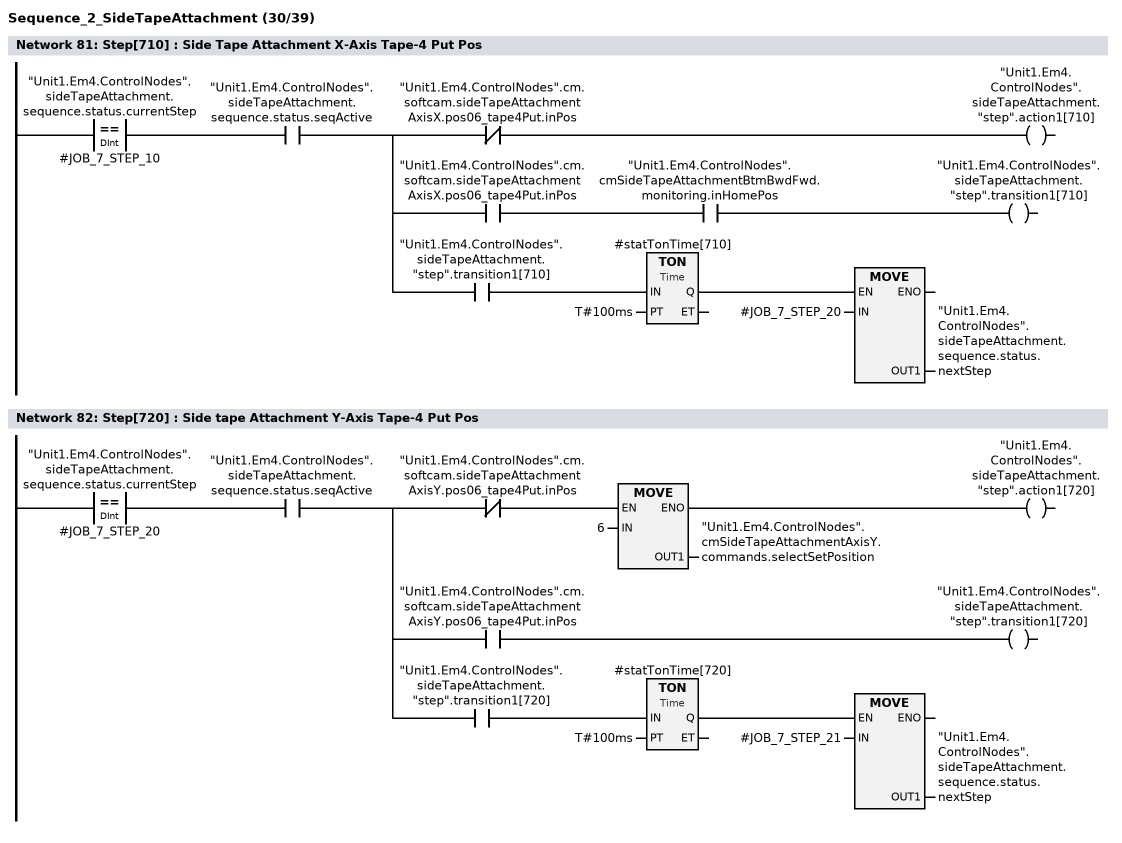
   RUNG wire#powerrail
      { S7_Templates := "SrcType := DInt" } EQ_Contact(in1 := "Unit1.Em4.ControlNodes".sideTapeAttachment.sequence.status.currentStep, in2 := #JOB_7_STEP_10)
      Contact( "Unit1.Em4.ControlNodes".sideTapeAttachment.sequence.status.seqActive )
      wire#w1
      I_Contact( "Unit1.Em4.ControlNodes".cm.softcam.sideTapeAttachmentAxisX.pos06_tape4Put.inPos )
      Coil( "Unit1.Em4.ControlNodes".sideTapeAttachment."step".action1[710] )
   END_RUNG
   RUNG wire#w1
      Contact( "Unit1.Em4.ControlNodes".cm.softcam.sideTapeAttachmentAxisX.pos06_tape4Put.inPos )
      Contact( "Unit1.Em4.ControlNodes".cmSideTapeAttachmentBtmBwdFwd.monitoring.inHomePos )
      Coil( "Unit1.Em4.ControlNodes".sideTapeAttachment."step".transition1[710] )
   END_RUNG
   RUNG wire#w1
      Contact( "Unit1.Em4.ControlNodes".sideTapeAttachment."step".transition1[710] )
      { S7_Templates := "time_type := Time" } #statTonTime[710].TON(pt := T#100ms, et =>)
      Move(in := #JOB_7_STEP_20, out1 => "Unit1.Em4.ControlNodes".sideTapeAttachment.sequence.status.nextStep)
   END_RUNG
   // the same network as SCL:
   #_w1 := ("Unit1.Em4.ControlNodes".sideTapeAttachment.sequence.status.currentStep = #JOB_7_STEP_10) AND "Unit1.Em4.ControlNodes".sideTapeAttachment.sequence.status.seqActive;
   "Unit1.Em4.ControlNodes".sideTapeAttachment."step".action1[710] := #_w1 AND NOT "Unit1.Em4.ControlNodes".cm.softcam.sideTapeAttachmentAxisX.pos06_tape4Put.inPos;
   "Unit1.Em4.ControlNodes".sideTapeAttachment."step".transition1[710] := #_w1 AND "Unit1.Em4.ControlNodes".cm.softcam.sideTapeAttachmentAxisX.pos06_tape4Put.inPos AND "Unit1.Em4.ControlNodes".cmSideTapeAttachmentBtmBwdFwd.monitoring.inHomePos;
   #statTonTime[710].TON(IN := #_w1 AND "Unit1.Em4.ControlNodes".sideTapeAttachment."step".transition1[710],
                         PT := T#100ms);
   IF #statTonTime[710].Q THEN
       "Unit1.Em4.ControlNodes".sideTapeAttachment.sequence.status.nextStep := #JOB_7_STEP_20;
   END_IF;
END_REGION

REGION Network 82: Step[720] : Side tape Attachment Y-Axis Tape-4 Put Pos
   RUNG wire#powerrail
      { S7_Templates := "SrcType := DInt" } EQ_Contact(in1 := "Unit1.Em4.ControlNodes".sideTapeAttachment.sequence.status.currentStep, in2 := #JOB_7_STEP_20)
      Contact( "Unit1.Em4.ControlNodes".sideTapeAttachment.sequence.status.seqActive )
      wire#w1
      I_Contact( "Unit1.Em4.ControlNodes".cm.softcam.sideTapeAttachmentAxisY.pos06_tape4Put.inPos )
      Move(in := 6, out1 => "Unit1.Em4.ControlNodes".cmSideTapeAttachmentAxisY.commands.selectSetPosition)
      Coil( "Unit1.Em4.ControlNodes".sideTapeAttachment."step".action1[720] )
   END_RUNG
   RUNG wire#w1
      Contact( "Unit1.Em4.ControlNodes".cm.softcam.sideTapeAttachmentAxisY.pos06_tape4Put.inPos )
      Coil( "Unit1.Em4.ControlNodes".sideTapeAttachment."step".transition1[720] )
   END_RUNG
   RUNG wire#w1
      Contact( "Unit1.Em4.ControlNodes".sideTapeAttachment."step".transition1[720] )
      { S7_Templates := "time_type := Time" } #statTonTime[720].TON(pt := T#100ms, et =>)
      Move(in := #JOB_7_STEP_21, out1 => "Unit1.Em4.ControlNodes".sideTapeAttachment.sequence.status.nextStep)
   END_RUNG
   // the same network as SCL:
   #_w1 := ("Unit1.Em4.ControlNodes".sideTapeAttachment.sequence.status.currentStep = #JOB_7_STEP_20) AND "Unit1.Em4.ControlNodes".sideTapeAttachment.sequence.status.seqActive;
   #_w2 := #_w1 AND NOT "Unit1.Em4.ControlNodes".cm.softcam.sideTapeAttachmentAxisY.pos06_tape4Put.inPos;
   IF #_w2 THEN "Unit1.Em4.ControlNodes".cmSideTapeAttachmentAxisY.commands.selectSetPosition := 6; END_IF;
   "Unit1.Em4.ControlNodes".sideTapeAttachment."step".action1[720] := #_w2;
   "Unit1.Em4.ControlNodes".sideTapeAttachment."step".transition1[720] := #_w1 AND "Unit1.Em4.ControlNodes".cm.softcam.sideTapeAttachmentAxisY.pos06_tape4Put.inPos;
   #statTonTime[720].TON(IN := #_w1 AND "Unit1.Em4.ControlNodes".sideTapeAttachment."step".transition1[720],
                         PT := T#100ms);
   IF #statTonTime[720].Q THEN
       "Unit1.Em4.ControlNodes".sideTapeAttachment.sequence.status.nextStep := #JOB_7_STEP_21;
   END_IF;
END_REGION

REGION Network 83: Step[721] : Side Tape Attachment Right Forward, Vaccum Off
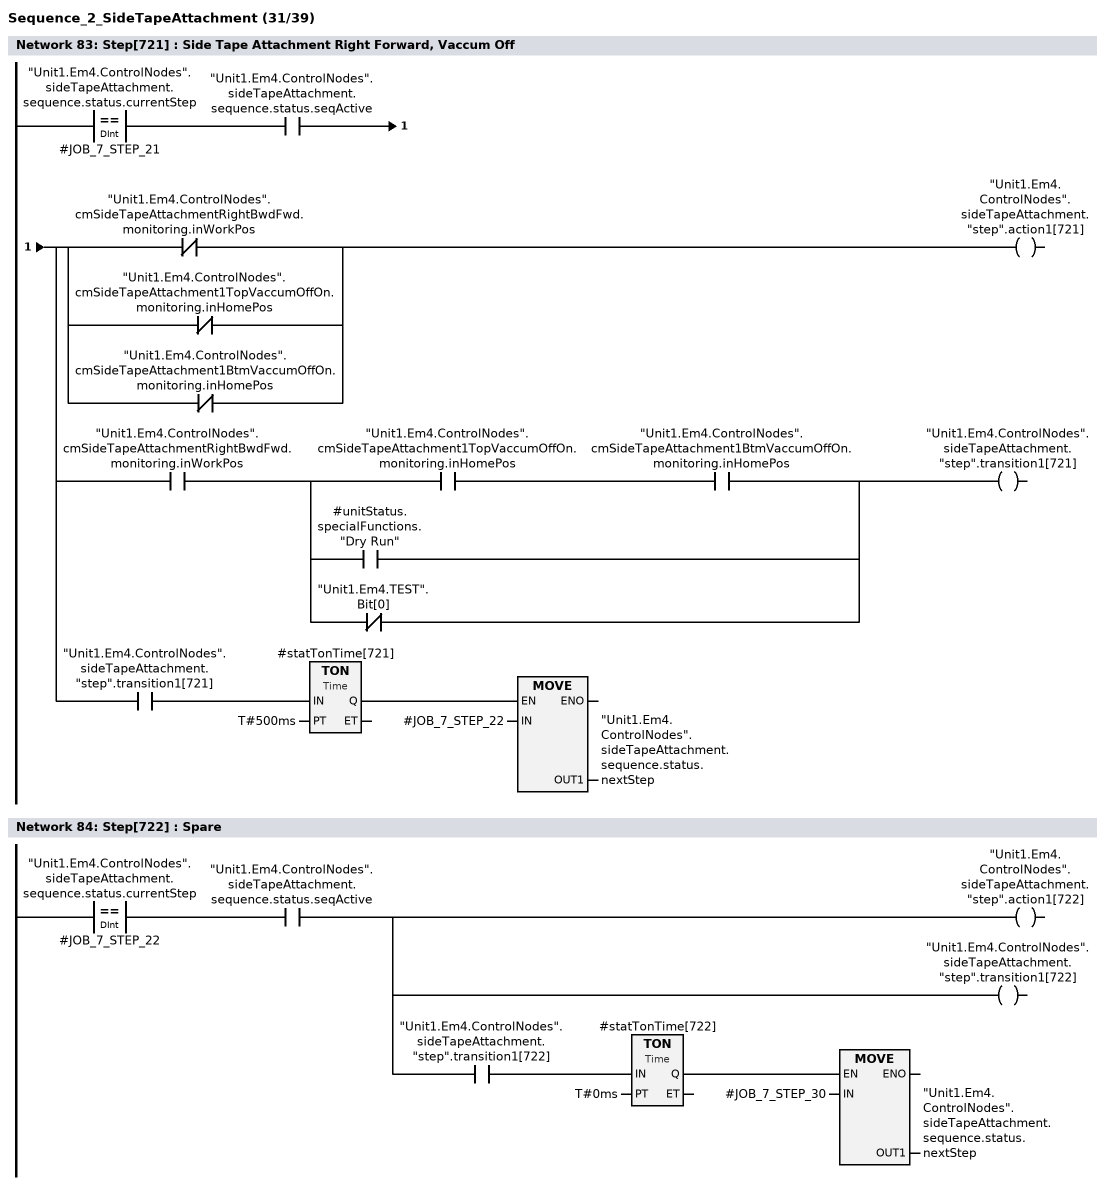
   RUNG wire#powerrail
      { S7_Templates := "SrcType := DInt" } EQ_Contact(in1 := "Unit1.Em4.ControlNodes".sideTapeAttachment.sequence.status.currentStep, in2 := #JOB_7_STEP_21)
      Contact( "Unit1.Em4.ControlNodes".sideTapeAttachment.sequence.status.seqActive )
      wire#w1
      I_Contact( "Unit1.Em4.ControlNodes".cmSideTapeAttachmentRightBwdFwd.monitoring.inWorkPos )
      wire#w2
      Coil( "Unit1.Em4.ControlNodes".sideTapeAttachment."step".action1[721] )
   END_RUNG
   RUNG wire#w1
      I_Contact( "Unit1.Em4.ControlNodes".cmSideTapeAttachment1TopVaccumOffOn.monitoring.inHomePos )
   END_RUNG wire#w2
   RUNG wire#w1
      I_Contact( "Unit1.Em4.ControlNodes".cmSideTapeAttachment1BtmVaccumOffOn.monitoring.inHomePos )
   END_RUNG wire#w2
   RUNG wire#w1
      Contact( "Unit1.Em4.ControlNodes".cmSideTapeAttachmentRightBwdFwd.monitoring.inWorkPos )
      wire#w3
      Contact( "Unit1.Em4.ControlNodes".cmSideTapeAttachment1TopVaccumOffOn.monitoring.inHomePos )
      Contact( "Unit1.Em4.ControlNodes".cmSideTapeAttachment1BtmVaccumOffOn.monitoring.inHomePos )
      wire#w4
      Coil( "Unit1.Em4.ControlNodes".sideTapeAttachment."step".transition1[721] )
   END_RUNG
   RUNG wire#w3
      Contact( #unitStatus.specialFunctions."Dry Run" )
   END_RUNG wire#w4
   RUNG wire#w3
      I_Contact( "Unit1.Em4.TEST".Bit[0] )
   END_RUNG wire#w4
   RUNG wire#w1
      Contact( "Unit1.Em4.ControlNodes".sideTapeAttachment."step".transition1[721] )
      { S7_Templates := "time_type := Time" } #statTonTime[721].TON(pt := T#500ms, et =>)
      Move(in := #JOB_7_STEP_22, out1 => "Unit1.Em4.ControlNodes".sideTapeAttachment.sequence.status.nextStep)
   END_RUNG
   // the same network as SCL:
   #_w1 := ("Unit1.Em4.ControlNodes".sideTapeAttachment.sequence.status.currentStep = #JOB_7_STEP_21) AND "Unit1.Em4.ControlNodes".sideTapeAttachment.sequence.status.seqActive;
   "Unit1.Em4.ControlNodes".sideTapeAttachment."step".action1[721] := #_w1 AND (NOT "Unit1.Em4.ControlNodes".cmSideTapeAttachmentRightBwdFwd.monitoring.inWorkPos OR NOT "Unit1.Em4.ControlNodes".cmSideTapeAttachment1TopVaccumOffOn.monitoring.inHomePos OR NOT "Unit1.Em4.ControlNodes".cmSideTapeAttachment1BtmVaccumOffOn.monitoring.inHomePos);
   "Unit1.Em4.ControlNodes".sideTapeAttachment."step".transition1[721] := #_w1 AND "Unit1.Em4.ControlNodes".cmSideTapeAttachmentRightBwdFwd.monitoring.inWorkPos AND (("Unit1.Em4.ControlNodes".cmSideTapeAttachment1TopVaccumOffOn.monitoring.inHomePos AND "Unit1.Em4.ControlNodes".cmSideTapeAttachment1BtmVaccumOffOn.monitoring.inHomePos) OR #unitStatus.specialFunctions."Dry Run" OR NOT "Unit1.Em4.TEST".Bit[0]);
   #statTonTime[721].TON(IN := #_w1 AND "Unit1.Em4.ControlNodes".sideTapeAttachment."step".transition1[721],
                         PT := T#500ms);
   IF #statTonTime[721].Q THEN
       "Unit1.Em4.ControlNodes".sideTapeAttachment.sequence.status.nextStep := #JOB_7_STEP_22;
   END_IF;
END_REGION

REGION Network 84: Step[722] : Spare
   RUNG wire#powerrail
      { S7_Templates := "SrcType := DInt" } EQ_Contact(in1 := "Unit1.Em4.ControlNodes".sideTapeAttachment.sequence.status.currentStep, in2 := #JOB_7_STEP_22)
      Contact( "Unit1.Em4.ControlNodes".sideTapeAttachment.sequence.status.seqActive )
      wire#w1
      Coil( "Unit1.Em4.ControlNodes".sideTapeAttachment."step".action1[722] )
   END_RUNG
   RUNG wire#w1
      Coil( "Unit1.Em4.ControlNodes".sideTapeAttachment."step".transition1[722] )
   END_RUNG
   RUNG wire#w1
      Contact( "Unit1.Em4.ControlNodes".sideTapeAttachment."step".transition1[722] )
      { S7_Templates := "time_type := Time" } #statTonTime[722].TON(pt := T#0ms, et =>)
      Move(in := #JOB_7_STEP_30, out1 => "Unit1.Em4.ControlNodes".sideTapeAttachment.sequence.status.nextStep)
   END_RUNG
   // the same network as SCL:
   "Unit1.Em4.ControlNodes".sideTapeAttachment."step".action1[722] := ("Unit1.Em4.ControlNodes".sideTapeAttachment.sequence.status.currentStep = #JOB_7_STEP_22) AND "Unit1.Em4.ControlNodes".sideTapeAttachment.sequence.status.seqActive;
   "Unit1.Em4.ControlNodes".sideTapeAttachment."step".transition1[722] := ("Unit1.Em4.ControlNodes".sideTapeAttachment.sequence.status.currentStep = #JOB_7_STEP_22) AND "Unit1.Em4.ControlNodes".sideTapeAttachment.sequence.status.seqActive;
   #statTonTime[722].TON(IN := ("Unit1.Em4.ControlNodes".sideTapeAttachment.sequence.status.currentStep = #JOB_7_STEP_22) AND "Unit1.Em4.ControlNodes".sideTapeAttachment.sequence.status.seqActive AND "Unit1.Em4.ControlNodes".sideTapeAttachment."step".transition1[722],
                         PT := T#0ms);
   IF #statTonTime[722].Q THEN
       "Unit1.Em4.ControlNodes".sideTapeAttachment.sequence.status.nextStep := #JOB_7_STEP_30;
   END_IF;
END_REGION

REGION Network 85: Step[730] : Side Tape Attachment Right Backward
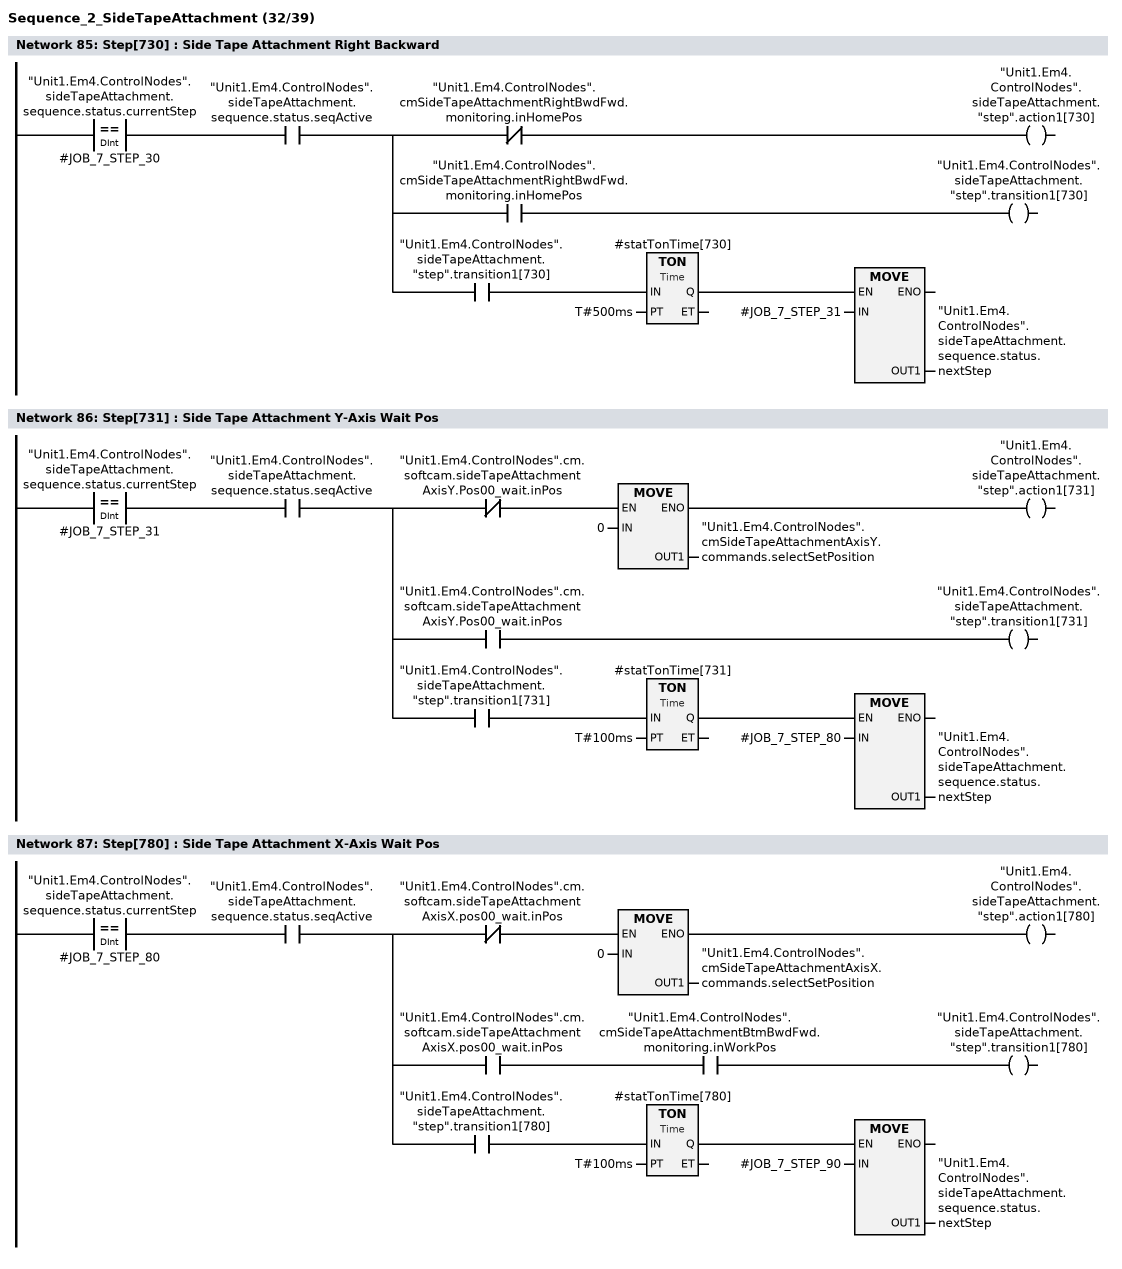
   RUNG wire#powerrail
      { S7_Templates := "SrcType := DInt" } EQ_Contact(in1 := "Unit1.Em4.ControlNodes".sideTapeAttachment.sequence.status.currentStep, in2 := #JOB_7_STEP_30)
      Contact( "Unit1.Em4.ControlNodes".sideTapeAttachment.sequence.status.seqActive )
      wire#w1
      I_Contact( "Unit1.Em4.ControlNodes".cmSideTapeAttachmentRightBwdFwd.monitoring.inHomePos )
      Coil( "Unit1.Em4.ControlNodes".sideTapeAttachment."step".action1[730] )
   END_RUNG
   RUNG wire#w1
      Contact( "Unit1.Em4.ControlNodes".cmSideTapeAttachmentRightBwdFwd.monitoring.inHomePos )
      Coil( "Unit1.Em4.ControlNodes".sideTapeAttachment."step".transition1[730] )
   END_RUNG
   RUNG wire#w1
      Contact( "Unit1.Em4.ControlNodes".sideTapeAttachment."step".transition1[730] )
      { S7_Templates := "time_type := Time" } #statTonTime[730].TON(pt := T#500ms, et =>)
      Move(in := #JOB_7_STEP_31, out1 => "Unit1.Em4.ControlNodes".sideTapeAttachment.sequence.status.nextStep)
   END_RUNG
   // the same network as SCL:
   #_w1 := ("Unit1.Em4.ControlNodes".sideTapeAttachment.sequence.status.currentStep = #JOB_7_STEP_30) AND "Unit1.Em4.ControlNodes".sideTapeAttachment.sequence.status.seqActive;
   "Unit1.Em4.ControlNodes".sideTapeAttachment."step".action1[730] := #_w1 AND NOT "Unit1.Em4.ControlNodes".cmSideTapeAttachmentRightBwdFwd.monitoring.inHomePos;
   "Unit1.Em4.ControlNodes".sideTapeAttachment."step".transition1[730] := #_w1 AND "Unit1.Em4.ControlNodes".cmSideTapeAttachmentRightBwdFwd.monitoring.inHomePos;
   #statTonTime[730].TON(IN := #_w1 AND "Unit1.Em4.ControlNodes".sideTapeAttachment."step".transition1[730],
                         PT := T#500ms);
   IF #statTonTime[730].Q THEN
       "Unit1.Em4.ControlNodes".sideTapeAttachment.sequence.status.nextStep := #JOB_7_STEP_31;
   END_IF;
END_REGION

REGION Network 86: Step[731] : Side Tape Attachment Y-Axis Wait Pos
   RUNG wire#powerrail
      { S7_Templates := "SrcType := DInt" } EQ_Contact(in1 := "Unit1.Em4.ControlNodes".sideTapeAttachment.sequence.status.currentStep, in2 := #JOB_7_STEP_31)
      Contact( "Unit1.Em4.ControlNodes".sideTapeAttachment.sequence.status.seqActive )
      wire#w1
      I_Contact( "Unit1.Em4.ControlNodes".cm.softcam.sideTapeAttachmentAxisY.Pos00_wait.inPos )
      Move(in := 0, out1 => "Unit1.Em4.ControlNodes".cmSideTapeAttachmentAxisY.commands.selectSetPosition)
      Coil( "Unit1.Em4.ControlNodes".sideTapeAttachment."step".action1[731] )
   END_RUNG
   RUNG wire#w1
      Contact( "Unit1.Em4.ControlNodes".cm.softcam.sideTapeAttachmentAxisY.Pos00_wait.inPos )
      Coil( "Unit1.Em4.ControlNodes".sideTapeAttachment."step".transition1[731] )
   END_RUNG
   RUNG wire#w1
      Contact( "Unit1.Em4.ControlNodes".sideTapeAttachment."step".transition1[731] )
      { S7_Templates := "time_type := Time" } #statTonTime[731].TON(pt := T#100ms, et =>)
      Move(in := #JOB_7_STEP_80, out1 => "Unit1.Em4.ControlNodes".sideTapeAttachment.sequence.status.nextStep)
   END_RUNG
   // the same network as SCL:
   #_w1 := ("Unit1.Em4.ControlNodes".sideTapeAttachment.sequence.status.currentStep = #JOB_7_STEP_31) AND "Unit1.Em4.ControlNodes".sideTapeAttachment.sequence.status.seqActive;
   #_w2 := #_w1 AND NOT "Unit1.Em4.ControlNodes".cm.softcam.sideTapeAttachmentAxisY.Pos00_wait.inPos;
   IF #_w2 THEN "Unit1.Em4.ControlNodes".cmSideTapeAttachmentAxisY.commands.selectSetPosition := 0; END_IF;
   "Unit1.Em4.ControlNodes".sideTapeAttachment."step".action1[731] := #_w2;
   "Unit1.Em4.ControlNodes".sideTapeAttachment."step".transition1[731] := #_w1 AND "Unit1.Em4.ControlNodes".cm.softcam.sideTapeAttachmentAxisY.Pos00_wait.inPos;
   #statTonTime[731].TON(IN := #_w1 AND "Unit1.Em4.ControlNodes".sideTapeAttachment."step".transition1[731],
                         PT := T#100ms);
   IF #statTonTime[731].Q THEN
       "Unit1.Em4.ControlNodes".sideTapeAttachment.sequence.status.nextStep := #JOB_7_STEP_80;
   END_IF;
END_REGION

REGION Network 87: Step[780] : Side Tape Attachment X-Axis Wait Pos
   RUNG wire#powerrail
      { S7_Templates := "SrcType := DInt" } EQ_Contact(in1 := "Unit1.Em4.ControlNodes".sideTapeAttachment.sequence.status.currentStep, in2 := #JOB_7_STEP_80)
      Contact( "Unit1.Em4.ControlNodes".sideTapeAttachment.sequence.status.seqActive )
      wire#w1
      I_Contact( "Unit1.Em4.ControlNodes".cm.softcam.sideTapeAttachmentAxisX.pos00_wait.inPos )
      Move(in := 0, out1 => "Unit1.Em4.ControlNodes".cmSideTapeAttachmentAxisX.commands.selectSetPosition)
      Coil( "Unit1.Em4.ControlNodes".sideTapeAttachment."step".action1[780] )
   END_RUNG
   RUNG wire#w1
      Contact( "Unit1.Em4.ControlNodes".cm.softcam.sideTapeAttachmentAxisX.pos00_wait.inPos )
      Contact( "Unit1.Em4.ControlNodes".cmSideTapeAttachmentBtmBwdFwd.monitoring.inWorkPos )
      Coil( "Unit1.Em4.ControlNodes".sideTapeAttachment."step".transition1[780] )
   END_RUNG
   RUNG wire#w1
      Contact( "Unit1.Em4.ControlNodes".sideTapeAttachment."step".transition1[780] )
      { S7_Templates := "time_type := Time" } #statTonTime[780].TON(pt := T#100ms, et =>)
      Move(in := #JOB_7_STEP_90, out1 => "Unit1.Em4.ControlNodes".sideTapeAttachment.sequence.status.nextStep)
   END_RUNG
   // the same network as SCL:
   #_w1 := ("Unit1.Em4.ControlNodes".sideTapeAttachment.sequence.status.currentStep = #JOB_7_STEP_80) AND "Unit1.Em4.ControlNodes".sideTapeAttachment.sequence.status.seqActive;
   #_w2 := #_w1 AND NOT "Unit1.Em4.ControlNodes".cm.softcam.sideTapeAttachmentAxisX.pos00_wait.inPos;
   IF #_w2 THEN "Unit1.Em4.ControlNodes".cmSideTapeAttachmentAxisX.commands.selectSetPosition := 0; END_IF;
   "Unit1.Em4.ControlNodes".sideTapeAttachment."step".action1[780] := #_w2;
   "Unit1.Em4.ControlNodes".sideTapeAttachment."step".transition1[780] := #_w1 AND "Unit1.Em4.ControlNodes".cm.softcam.sideTapeAttachmentAxisX.pos00_wait.inPos AND "Unit1.Em4.ControlNodes".cmSideTapeAttachmentBtmBwdFwd.monitoring.inWorkPos;
   #statTonTime[780].TON(IN := #_w1 AND "Unit1.Em4.ControlNodes".sideTapeAttachment."step".transition1[780],
                         PT := T#100ms);
   IF #statTonTime[780].Q THEN
       "Unit1.Em4.ControlNodes".sideTapeAttachment.sequence.status.nextStep := #JOB_7_STEP_90;
   END_IF;
END_REGION

REGION Network 88: Step[790] : Job[7] Step End
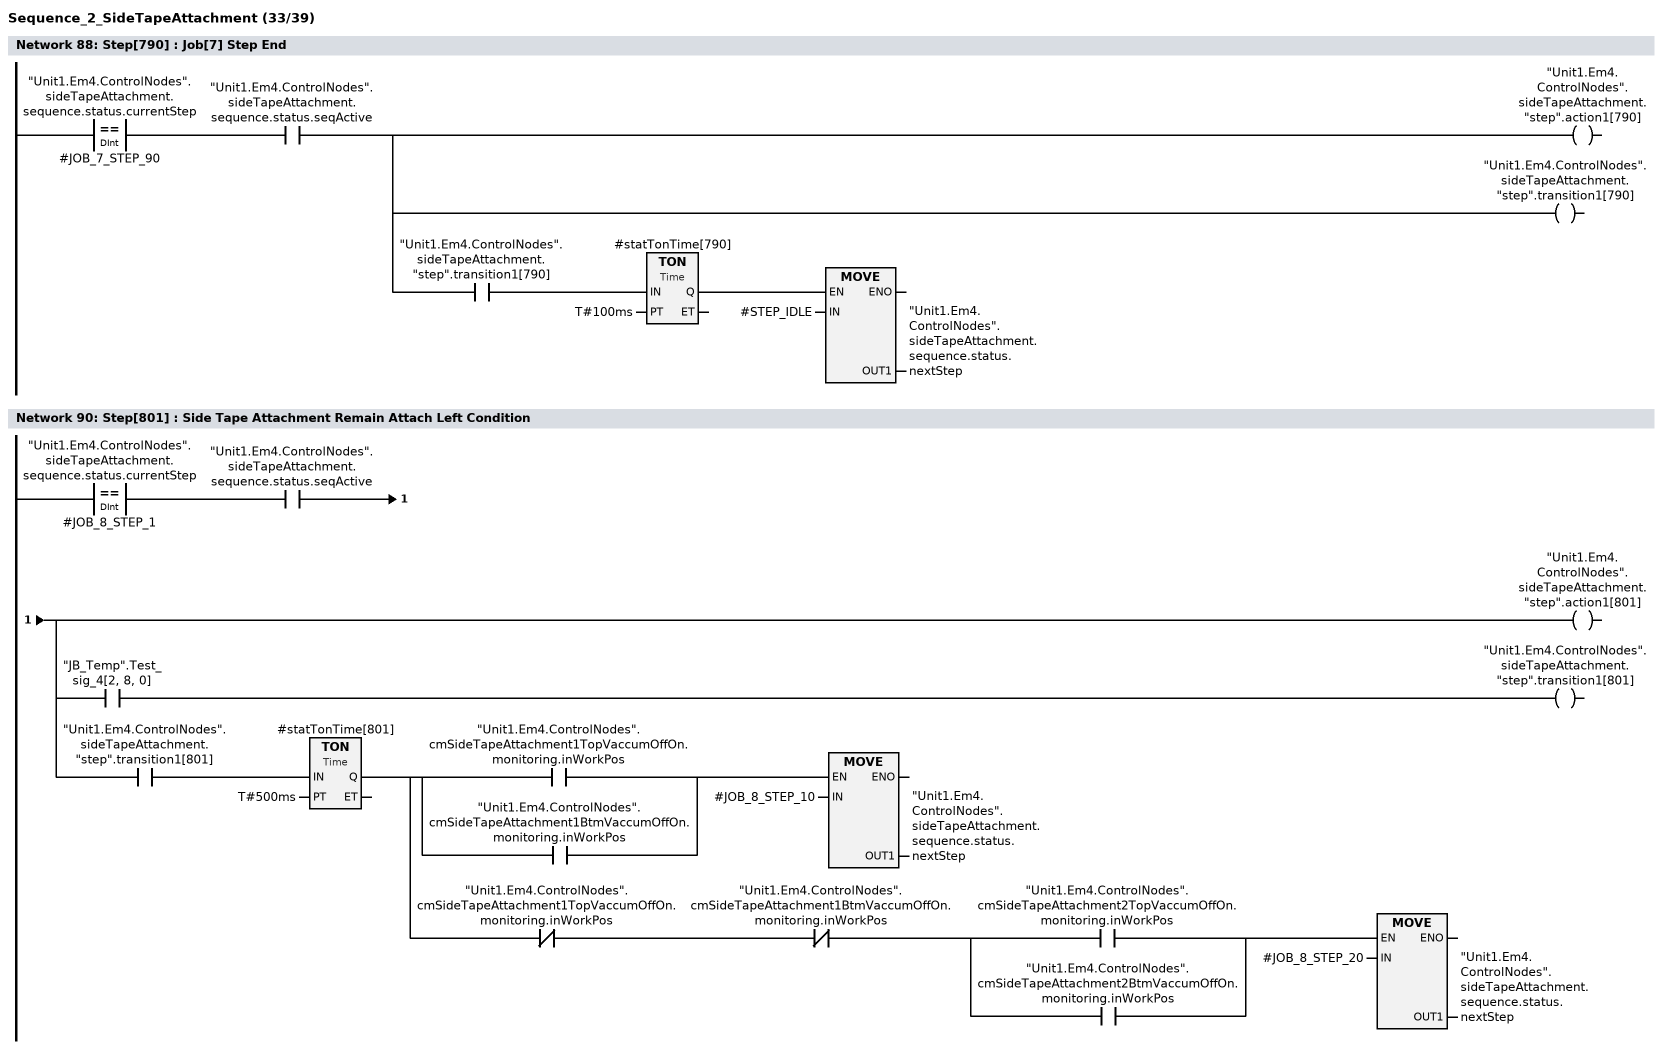
   RUNG wire#powerrail
      { S7_Templates := "SrcType := DInt" } EQ_Contact(in1 := "Unit1.Em4.ControlNodes".sideTapeAttachment.sequence.status.currentStep, in2 := #JOB_7_STEP_90)
      Contact( "Unit1.Em4.ControlNodes".sideTapeAttachment.sequence.status.seqActive )
      wire#w1
      Coil( "Unit1.Em4.ControlNodes".sideTapeAttachment."step".action1[790] )
   END_RUNG
   RUNG wire#w1
      Coil( "Unit1.Em4.ControlNodes".sideTapeAttachment."step".transition1[790] )
   END_RUNG
   RUNG wire#w1
      Contact( "Unit1.Em4.ControlNodes".sideTapeAttachment."step".transition1[790] )
      { S7_Templates := "time_type := Time" } #statTonTime[790].TON(pt := T#100ms, et =>)
      Move(in := #STEP_IDLE, out1 => "Unit1.Em4.ControlNodes".sideTapeAttachment.sequence.status.nextStep)
   END_RUNG
   // the same network as SCL:
   "Unit1.Em4.ControlNodes".sideTapeAttachment."step".action1[790] := ("Unit1.Em4.ControlNodes".sideTapeAttachment.sequence.status.currentStep = #JOB_7_STEP_90) AND "Unit1.Em4.ControlNodes".sideTapeAttachment.sequence.status.seqActive;
   "Unit1.Em4.ControlNodes".sideTapeAttachment."step".transition1[790] := ("Unit1.Em4.ControlNodes".sideTapeAttachment.sequence.status.currentStep = #JOB_7_STEP_90) AND "Unit1.Em4.ControlNodes".sideTapeAttachment.sequence.status.seqActive;
   #statTonTime[790].TON(IN := ("Unit1.Em4.ControlNodes".sideTapeAttachment.sequence.status.currentStep = #JOB_7_STEP_90) AND "Unit1.Em4.ControlNodes".sideTapeAttachment.sequence.status.seqActive AND "Unit1.Em4.ControlNodes".sideTapeAttachment."step".transition1[790],
                         PT := T#100ms);
   IF #statTonTime[790].Q THEN
       "Unit1.Em4.ControlNodes".sideTapeAttachment.sequence.status.nextStep := #STEP_IDLE;
   END_IF;
END_REGION

REGION Network 89: ******************** Job[8] SIDE TAPE ATTACHMENT LEFT REMAIN ATTACH ********************
END_REGION

REGION Network 90: Step[801] : Side Tape Attachment Remain Attach Left Condition
   RUNG wire#powerrail
      { S7_Templates := "SrcType := DInt" } EQ_Contact(in1 := "Unit1.Em4.ControlNodes".sideTapeAttachment.sequence.status.currentStep, in2 := #JOB_8_STEP_1)
      Contact( "Unit1.Em4.ControlNodes".sideTapeAttachment.sequence.status.seqActive )
      wire#w1
      Coil( "Unit1.Em4.ControlNodes".sideTapeAttachment."step".action1[801] )
   END_RUNG
   RUNG wire#w1
      Contact( "JB_Temp".Test_sig_4[2, 8, 0] )
      Coil( "Unit1.Em4.ControlNodes".sideTapeAttachment."step".transition1[801] )
   END_RUNG
   RUNG wire#w1
      Contact( "Unit1.Em4.ControlNodes".sideTapeAttachment."step".transition1[801] )
      { S7_Templates := "time_type := Time" } #statTonTime[801].TON(pt := T#500ms, et =>)
      wire#w2
      Contact( "Unit1.Em4.ControlNodes".cmSideTapeAttachment1TopVaccumOffOn.monitoring.inWorkPos )
      wire#w3
      Move(in := #JOB_8_STEP_10, out1 => "Unit1.Em4.ControlNodes".sideTapeAttachment.sequence.status.nextStep)
   END_RUNG
   RUNG wire#w2
      Contact( "Unit1.Em4.ControlNodes".cmSideTapeAttachment1BtmVaccumOffOn.monitoring.inWorkPos )
   END_RUNG wire#w3
   RUNG wire#w2
      I_Contact( "Unit1.Em4.ControlNodes".cmSideTapeAttachment1TopVaccumOffOn.monitoring.inWorkPos )
      I_Contact( "Unit1.Em4.ControlNodes".cmSideTapeAttachment1BtmVaccumOffOn.monitoring.inWorkPos )
      wire#w4
      Contact( "Unit1.Em4.ControlNodes".cmSideTapeAttachment2TopVaccumOffOn.monitoring.inWorkPos )
      wire#w5
      Move(in := #JOB_8_STEP_20, out1 => "Unit1.Em4.ControlNodes".sideTapeAttachment.sequence.status.nextStep)
   END_RUNG
   RUNG wire#w4
      Contact( "Unit1.Em4.ControlNodes".cmSideTapeAttachment2BtmVaccumOffOn.monitoring.inWorkPos )
   END_RUNG wire#w5
   // the same network as SCL:
   "Unit1.Em4.ControlNodes".sideTapeAttachment."step".action1[801] := ("Unit1.Em4.ControlNodes".sideTapeAttachment.sequence.status.currentStep = #JOB_8_STEP_1) AND "Unit1.Em4.ControlNodes".sideTapeAttachment.sequence.status.seqActive;
   "Unit1.Em4.ControlNodes".sideTapeAttachment."step".transition1[801] := ("Unit1.Em4.ControlNodes".sideTapeAttachment.sequence.status.currentStep = #JOB_8_STEP_1) AND "Unit1.Em4.ControlNodes".sideTapeAttachment.sequence.status.seqActive AND "JB_Temp".Test_sig_4[2, 8, 0];
   #statTonTime[801].TON(IN := ("Unit1.Em4.ControlNodes".sideTapeAttachment.sequence.status.currentStep = #JOB_8_STEP_1) AND "Unit1.Em4.ControlNodes".sideTapeAttachment.sequence.status.seqActive AND "Unit1.Em4.ControlNodes".sideTapeAttachment."step".transition1[801],
                         PT := T#500ms);
   IF #statTonTime[801].Q AND ("Unit1.Em4.ControlNodes".cmSideTapeAttachment1TopVaccumOffOn.monitoring.inWorkPos OR "Unit1.Em4.ControlNodes".cmSideTapeAttachment1BtmVaccumOffOn.monitoring.inWorkPos) THEN
       "Unit1.Em4.ControlNodes".sideTapeAttachment.sequence.status.nextStep := #JOB_8_STEP_10;
   END_IF;
   IF #statTonTime[801].Q AND NOT "Unit1.Em4.ControlNodes".cmSideTapeAttachment1TopVaccumOffOn.monitoring.inWorkPos AND NOT "Unit1.Em4.ControlNodes".cmSideTapeAttachment1BtmVaccumOffOn.monitoring.inWorkPos AND ("Unit1.Em4.ControlNodes".cmSideTapeAttachment2TopVaccumOffOn.monitoring.inWorkPos OR "Unit1.Em4.ControlNodes".cmSideTapeAttachment2BtmVaccumOffOn.monitoring.inWorkPos) THEN
       "Unit1.Em4.ControlNodes".sideTapeAttachment.sequence.status.nextStep := #JOB_8_STEP_20;
   END_IF;
END_REGION

REGION Network 91: Step[810] : Side Tape Attachment X-Axis Remain Attach Left Position
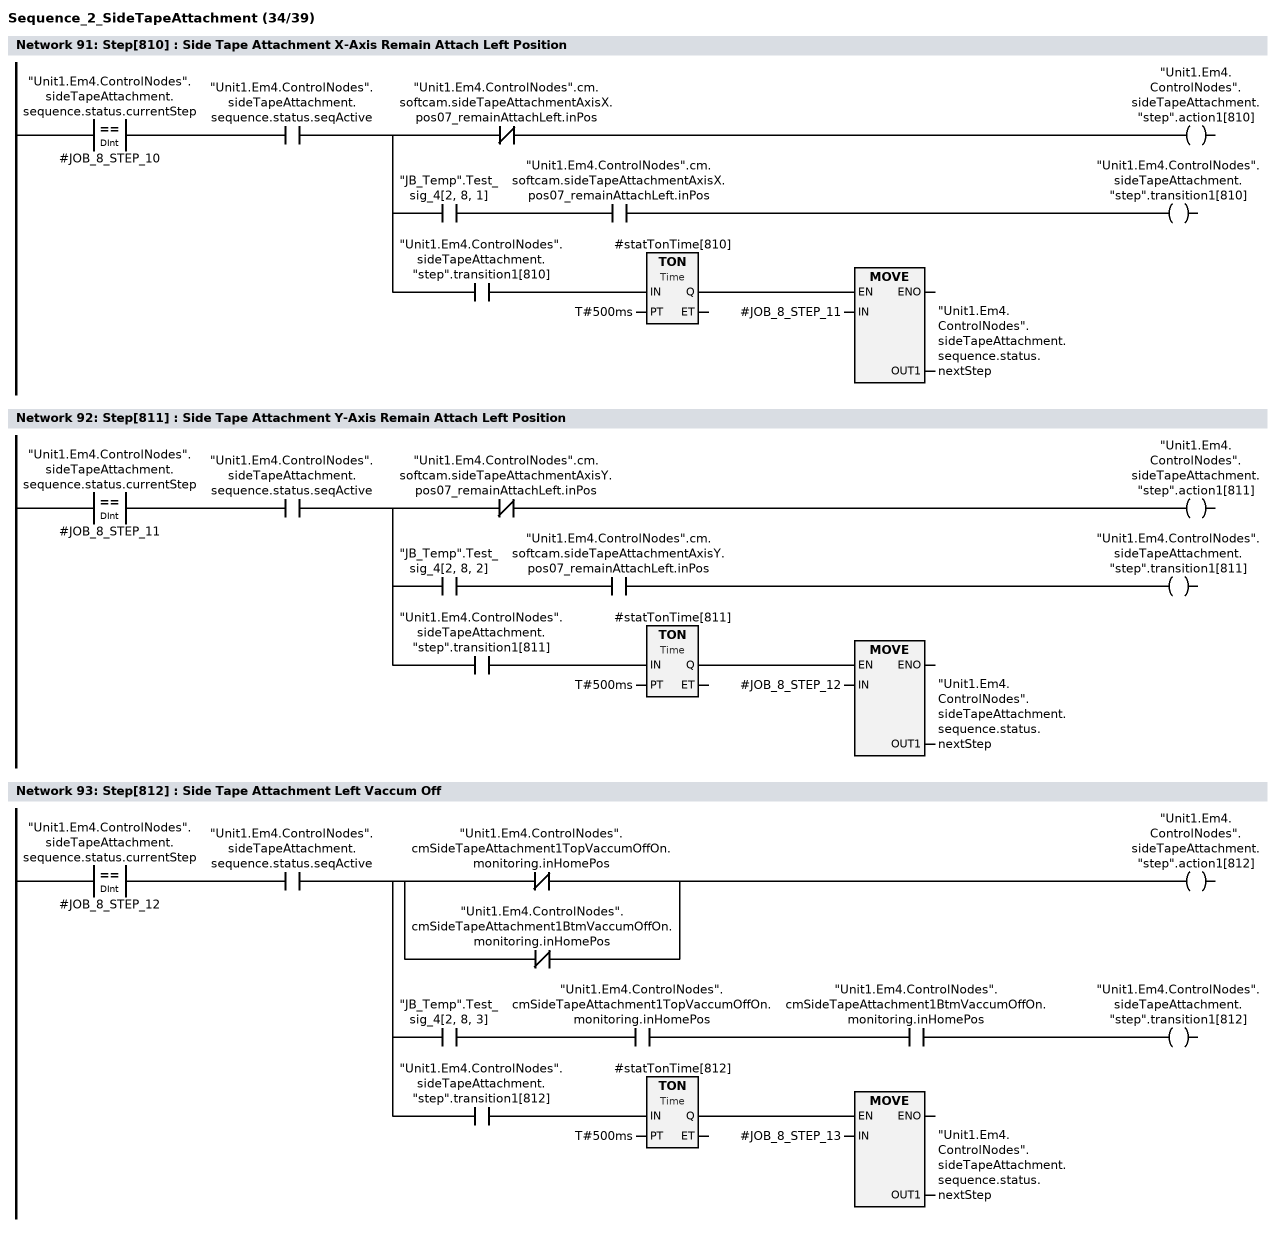
   RUNG wire#powerrail
      { S7_Templates := "SrcType := DInt" } EQ_Contact(in1 := "Unit1.Em4.ControlNodes".sideTapeAttachment.sequence.status.currentStep, in2 := #JOB_8_STEP_10)
      Contact( "Unit1.Em4.ControlNodes".sideTapeAttachment.sequence.status.seqActive )
      wire#w1
      I_Contact( "Unit1.Em4.ControlNodes".cm.softcam.sideTapeAttachmentAxisX.pos07_remainAttachLeft.inPos )
      Coil( "Unit1.Em4.ControlNodes".sideTapeAttachment."step".action1[810] )
   END_RUNG
   RUNG wire#w1
      Contact( "JB_Temp".Test_sig_4[2, 8, 1] )
      Contact( "Unit1.Em4.ControlNodes".cm.softcam.sideTapeAttachmentAxisX.pos07_remainAttachLeft.inPos )
      Coil( "Unit1.Em4.ControlNodes".sideTapeAttachment."step".transition1[810] )
   END_RUNG
   RUNG wire#w1
      Contact( "Unit1.Em4.ControlNodes".sideTapeAttachment."step".transition1[810] )
      { S7_Templates := "time_type := Time" } #statTonTime[810].TON(pt := T#500ms, et =>)
      Move(in := #JOB_8_STEP_11, out1 => "Unit1.Em4.ControlNodes".sideTapeAttachment.sequence.status.nextStep)
   END_RUNG
   // the same network as SCL:
   #_w1 := ("Unit1.Em4.ControlNodes".sideTapeAttachment.sequence.status.currentStep = #JOB_8_STEP_10) AND "Unit1.Em4.ControlNodes".sideTapeAttachment.sequence.status.seqActive;
   "Unit1.Em4.ControlNodes".sideTapeAttachment."step".action1[810] := #_w1 AND NOT "Unit1.Em4.ControlNodes".cm.softcam.sideTapeAttachmentAxisX.pos07_remainAttachLeft.inPos;
   "Unit1.Em4.ControlNodes".sideTapeAttachment."step".transition1[810] := #_w1 AND "JB_Temp".Test_sig_4[2, 8, 1] AND "Unit1.Em4.ControlNodes".cm.softcam.sideTapeAttachmentAxisX.pos07_remainAttachLeft.inPos;
   #statTonTime[810].TON(IN := #_w1 AND "Unit1.Em4.ControlNodes".sideTapeAttachment."step".transition1[810],
                         PT := T#500ms);
   IF #statTonTime[810].Q THEN
       "Unit1.Em4.ControlNodes".sideTapeAttachment.sequence.status.nextStep := #JOB_8_STEP_11;
   END_IF;
END_REGION

REGION Network 92: Step[811] : Side Tape Attachment Y-Axis Remain Attach Left Position
   RUNG wire#powerrail
      { S7_Templates := "SrcType := DInt" } EQ_Contact(in1 := "Unit1.Em4.ControlNodes".sideTapeAttachment.sequence.status.currentStep, in2 := #JOB_8_STEP_11)
      Contact( "Unit1.Em4.ControlNodes".sideTapeAttachment.sequence.status.seqActive )
      wire#w1
      I_Contact( "Unit1.Em4.ControlNodes".cm.softcam.sideTapeAttachmentAxisY.pos07_remainAttachLeft.inPos )
      Coil( "Unit1.Em4.ControlNodes".sideTapeAttachment."step".action1[811] )
   END_RUNG
   RUNG wire#w1
      Contact( "JB_Temp".Test_sig_4[2, 8, 2] )
      Contact( "Unit1.Em4.ControlNodes".cm.softcam.sideTapeAttachmentAxisY.pos07_remainAttachLeft.inPos )
      Coil( "Unit1.Em4.ControlNodes".sideTapeAttachment."step".transition1[811] )
   END_RUNG
   RUNG wire#w1
      Contact( "Unit1.Em4.ControlNodes".sideTapeAttachment."step".transition1[811] )
      { S7_Templates := "time_type := Time" } #statTonTime[811].TON(pt := T#500ms, et =>)
      Move(in := #JOB_8_STEP_12, out1 => "Unit1.Em4.ControlNodes".sideTapeAttachment.sequence.status.nextStep)
   END_RUNG
   // the same network as SCL:
   #_w1 := ("Unit1.Em4.ControlNodes".sideTapeAttachment.sequence.status.currentStep = #JOB_8_STEP_11) AND "Unit1.Em4.ControlNodes".sideTapeAttachment.sequence.status.seqActive;
   "Unit1.Em4.ControlNodes".sideTapeAttachment."step".action1[811] := #_w1 AND NOT "Unit1.Em4.ControlNodes".cm.softcam.sideTapeAttachmentAxisY.pos07_remainAttachLeft.inPos;
   "Unit1.Em4.ControlNodes".sideTapeAttachment."step".transition1[811] := #_w1 AND "JB_Temp".Test_sig_4[2, 8, 2] AND "Unit1.Em4.ControlNodes".cm.softcam.sideTapeAttachmentAxisY.pos07_remainAttachLeft.inPos;
   #statTonTime[811].TON(IN := #_w1 AND "Unit1.Em4.ControlNodes".sideTapeAttachment."step".transition1[811],
                         PT := T#500ms);
   IF #statTonTime[811].Q THEN
       "Unit1.Em4.ControlNodes".sideTapeAttachment.sequence.status.nextStep := #JOB_8_STEP_12;
   END_IF;
END_REGION

REGION Network 93: Step[812] : Side Tape Attachment Left Vaccum Off
   RUNG wire#powerrail
      { S7_Templates := "SrcType := DInt" } EQ_Contact(in1 := "Unit1.Em4.ControlNodes".sideTapeAttachment.sequence.status.currentStep, in2 := #JOB_8_STEP_12)
      Contact( "Unit1.Em4.ControlNodes".sideTapeAttachment.sequence.status.seqActive )
      wire#w1
      I_Contact( "Unit1.Em4.ControlNodes".cmSideTapeAttachment1TopVaccumOffOn.monitoring.inHomePos )
      wire#w2
      Coil( "Unit1.Em4.ControlNodes".sideTapeAttachment."step".action1[812] )
   END_RUNG
   RUNG wire#w1
      I_Contact( "Unit1.Em4.ControlNodes".cmSideTapeAttachment1BtmVaccumOffOn.monitoring.inHomePos )
   END_RUNG wire#w2
   RUNG wire#w1
      Contact( "JB_Temp".Test_sig_4[2, 8, 3] )
      Contact( "Unit1.Em4.ControlNodes".cmSideTapeAttachment1TopVaccumOffOn.monitoring.inHomePos )
      Contact( "Unit1.Em4.ControlNodes".cmSideTapeAttachment1BtmVaccumOffOn.monitoring.inHomePos )
      Coil( "Unit1.Em4.ControlNodes".sideTapeAttachment."step".transition1[812] )
   END_RUNG
   RUNG wire#w1
      Contact( "Unit1.Em4.ControlNodes".sideTapeAttachment."step".transition1[812] )
      { S7_Templates := "time_type := Time" } #statTonTime[812].TON(pt := T#500ms, et =>)
      Move(in := #JOB_8_STEP_13, out1 => "Unit1.Em4.ControlNodes".sideTapeAttachment.sequence.status.nextStep)
   END_RUNG
   // the same network as SCL:
   #_w1 := ("Unit1.Em4.ControlNodes".sideTapeAttachment.sequence.status.currentStep = #JOB_8_STEP_12) AND "Unit1.Em4.ControlNodes".sideTapeAttachment.sequence.status.seqActive;
   "Unit1.Em4.ControlNodes".sideTapeAttachment."step".action1[812] := #_w1 AND (NOT "Unit1.Em4.ControlNodes".cmSideTapeAttachment1TopVaccumOffOn.monitoring.inHomePos OR NOT "Unit1.Em4.ControlNodes".cmSideTapeAttachment1BtmVaccumOffOn.monitoring.inHomePos);
   "Unit1.Em4.ControlNodes".sideTapeAttachment."step".transition1[812] := #_w1 AND "JB_Temp".Test_sig_4[2, 8, 3] AND "Unit1.Em4.ControlNodes".cmSideTapeAttachment1TopVaccumOffOn.monitoring.inHomePos AND "Unit1.Em4.ControlNodes".cmSideTapeAttachment1BtmVaccumOffOn.monitoring.inHomePos;
   #statTonTime[812].TON(IN := #_w1 AND "Unit1.Em4.ControlNodes".sideTapeAttachment."step".transition1[812],
                         PT := T#500ms);
   IF #statTonTime[812].Q THEN
       "Unit1.Em4.ControlNodes".sideTapeAttachment.sequence.status.nextStep := #JOB_8_STEP_13;
   END_IF;
END_REGION

REGION Network 94: Step[813] : Side Tape Attachment Y-Axis Wait Pos
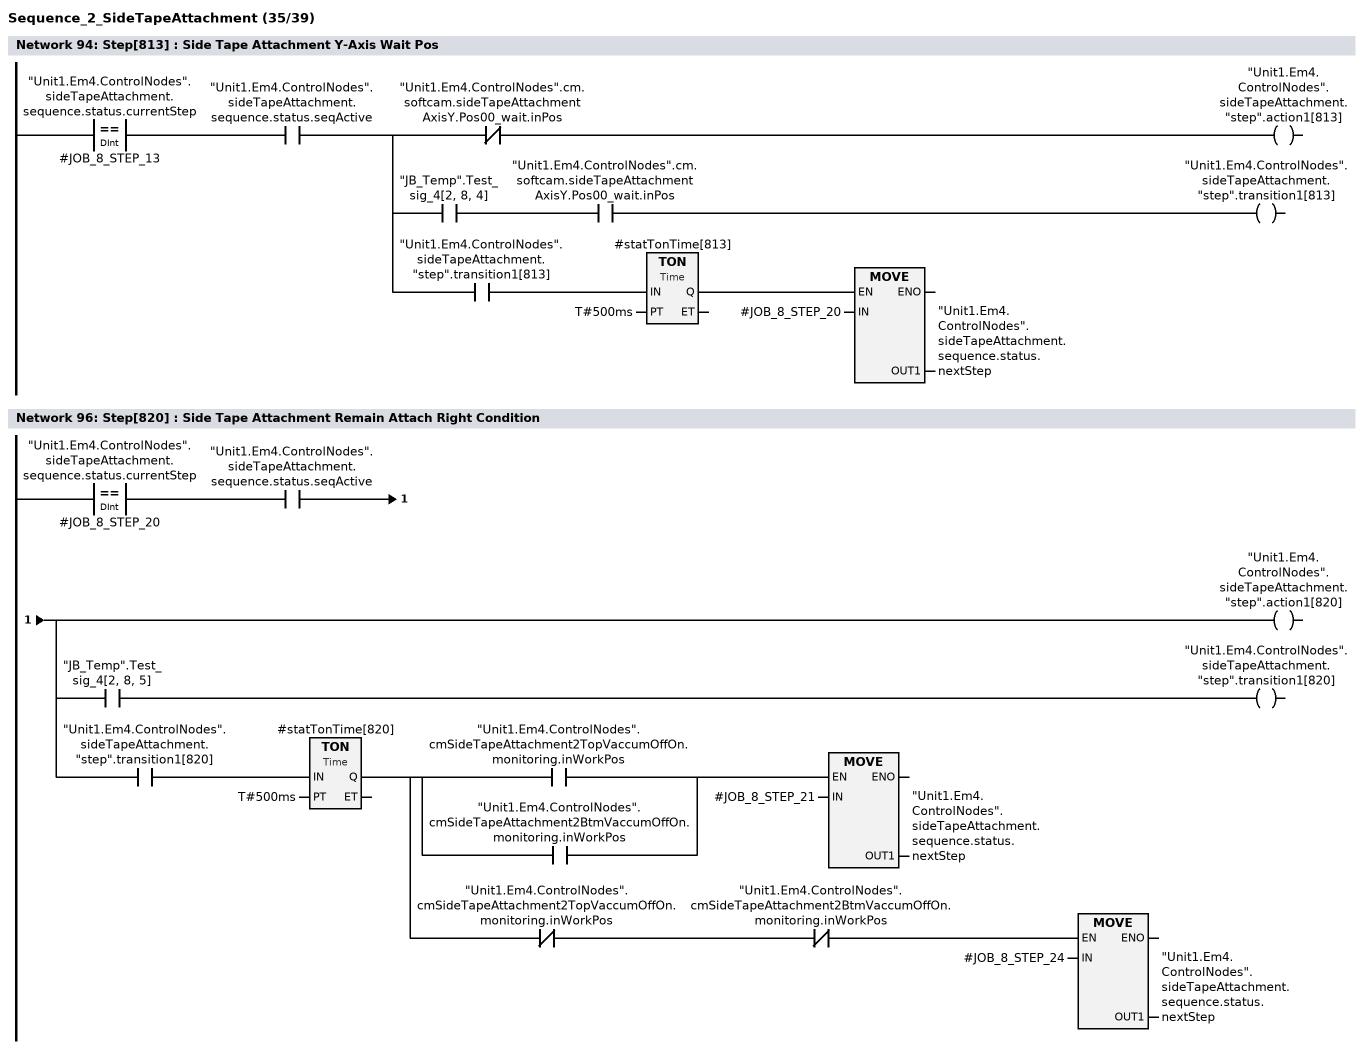
   RUNG wire#powerrail
      { S7_Templates := "SrcType := DInt" } EQ_Contact(in1 := "Unit1.Em4.ControlNodes".sideTapeAttachment.sequence.status.currentStep, in2 := #JOB_8_STEP_13)
      Contact( "Unit1.Em4.ControlNodes".sideTapeAttachment.sequence.status.seqActive )
      wire#w1
      I_Contact( "Unit1.Em4.ControlNodes".cm.softcam.sideTapeAttachmentAxisY.Pos00_wait.inPos )
      Coil( "Unit1.Em4.ControlNodes".sideTapeAttachment."step".action1[813] )
   END_RUNG
   RUNG wire#w1
      Contact( "JB_Temp".Test_sig_4[2, 8, 4] )
      Contact( "Unit1.Em4.ControlNodes".cm.softcam.sideTapeAttachmentAxisY.Pos00_wait.inPos )
      Coil( "Unit1.Em4.ControlNodes".sideTapeAttachment."step".transition1[813] )
   END_RUNG
   RUNG wire#w1
      Contact( "Unit1.Em4.ControlNodes".sideTapeAttachment."step".transition1[813] )
      { S7_Templates := "time_type := Time" } #statTonTime[813].TON(pt := T#500ms, et =>)
      Move(in := #JOB_8_STEP_20, out1 => "Unit1.Em4.ControlNodes".sideTapeAttachment.sequence.status.nextStep)
   END_RUNG
   // the same network as SCL:
   #_w1 := ("Unit1.Em4.ControlNodes".sideTapeAttachment.sequence.status.currentStep = #JOB_8_STEP_13) AND "Unit1.Em4.ControlNodes".sideTapeAttachment.sequence.status.seqActive;
   "Unit1.Em4.ControlNodes".sideTapeAttachment."step".action1[813] := #_w1 AND NOT "Unit1.Em4.ControlNodes".cm.softcam.sideTapeAttachmentAxisY.Pos00_wait.inPos;
   "Unit1.Em4.ControlNodes".sideTapeAttachment."step".transition1[813] := #_w1 AND "JB_Temp".Test_sig_4[2, 8, 4] AND "Unit1.Em4.ControlNodes".cm.softcam.sideTapeAttachmentAxisY.Pos00_wait.inPos;
   #statTonTime[813].TON(IN := #_w1 AND "Unit1.Em4.ControlNodes".sideTapeAttachment."step".transition1[813],
                         PT := T#500ms);
   IF #statTonTime[813].Q THEN
       "Unit1.Em4.ControlNodes".sideTapeAttachment.sequence.status.nextStep := #JOB_8_STEP_20;
   END_IF;
END_REGION

REGION Network 95: ******************** STEP[140~144] SIDE TAPE ATTACHMENT RIGHT REMAIN ATTACH ********************
END_REGION

REGION Network 96: Step[820] : Side Tape Attachment Remain Attach Right Condition
   RUNG wire#powerrail
      { S7_Templates := "SrcType := DInt" } EQ_Contact(in1 := "Unit1.Em4.ControlNodes".sideTapeAttachment.sequence.status.currentStep, in2 := #JOB_8_STEP_20)
      Contact( "Unit1.Em4.ControlNodes".sideTapeAttachment.sequence.status.seqActive )
      wire#w1
      Coil( "Unit1.Em4.ControlNodes".sideTapeAttachment."step".action1[820] )
   END_RUNG
   RUNG wire#w1
      Contact( "JB_Temp".Test_sig_4[2, 8, 5] )
      Coil( "Unit1.Em4.ControlNodes".sideTapeAttachment."step".transition1[820] )
   END_RUNG
   RUNG wire#w1
      Contact( "Unit1.Em4.ControlNodes".sideTapeAttachment."step".transition1[820] )
      { S7_Templates := "time_type := Time" } #statTonTime[820].TON(pt := T#500ms, et =>)
      wire#w2
      Contact( "Unit1.Em4.ControlNodes".cmSideTapeAttachment2TopVaccumOffOn.monitoring.inWorkPos )
      wire#w3
      Move(in := #JOB_8_STEP_21, out1 => "Unit1.Em4.ControlNodes".sideTapeAttachment.sequence.status.nextStep)
   END_RUNG
   RUNG wire#w2
      Contact( "Unit1.Em4.ControlNodes".cmSideTapeAttachment2BtmVaccumOffOn.monitoring.inWorkPos )
   END_RUNG wire#w3
   RUNG wire#w2
      I_Contact( "Unit1.Em4.ControlNodes".cmSideTapeAttachment2TopVaccumOffOn.monitoring.inWorkPos )
      I_Contact( "Unit1.Em4.ControlNodes".cmSideTapeAttachment2BtmVaccumOffOn.monitoring.inWorkPos )
      Move(in := #JOB_8_STEP_24, out1 => "Unit1.Em4.ControlNodes".sideTapeAttachment.sequence.status.nextStep)
   END_RUNG
   // the same network as SCL:
   "Unit1.Em4.ControlNodes".sideTapeAttachment."step".action1[820] := ("Unit1.Em4.ControlNodes".sideTapeAttachment.sequence.status.currentStep = #JOB_8_STEP_20) AND "Unit1.Em4.ControlNodes".sideTapeAttachment.sequence.status.seqActive;
   "Unit1.Em4.ControlNodes".sideTapeAttachment."step".transition1[820] := ("Unit1.Em4.ControlNodes".sideTapeAttachment.sequence.status.currentStep = #JOB_8_STEP_20) AND "Unit1.Em4.ControlNodes".sideTapeAttachment.sequence.status.seqActive AND "JB_Temp".Test_sig_4[2, 8, 5];
   #statTonTime[820].TON(IN := ("Unit1.Em4.ControlNodes".sideTapeAttachment.sequence.status.currentStep = #JOB_8_STEP_20) AND "Unit1.Em4.ControlNodes".sideTapeAttachment.sequence.status.seqActive AND "Unit1.Em4.ControlNodes".sideTapeAttachment."step".transition1[820],
                         PT := T#500ms);
   IF #statTonTime[820].Q AND ("Unit1.Em4.ControlNodes".cmSideTapeAttachment2TopVaccumOffOn.monitoring.inWorkPos OR "Unit1.Em4.ControlNodes".cmSideTapeAttachment2BtmVaccumOffOn.monitoring.inWorkPos) THEN
       "Unit1.Em4.ControlNodes".sideTapeAttachment.sequence.status.nextStep := #JOB_8_STEP_21;
   END_IF;
   IF #statTonTime[820].Q AND NOT "Unit1.Em4.ControlNodes".cmSideTapeAttachment2TopVaccumOffOn.monitoring.inWorkPos AND NOT "Unit1.Em4.ControlNodes".cmSideTapeAttachment2BtmVaccumOffOn.monitoring.inWorkPos THEN
       "Unit1.Em4.ControlNodes".sideTapeAttachment.sequence.status.nextStep := #JOB_8_STEP_24;
   END_IF;
END_REGION

REGION Network 97: Step[821] : Side Tape Attachment X-Axis Remain Attach Right Position
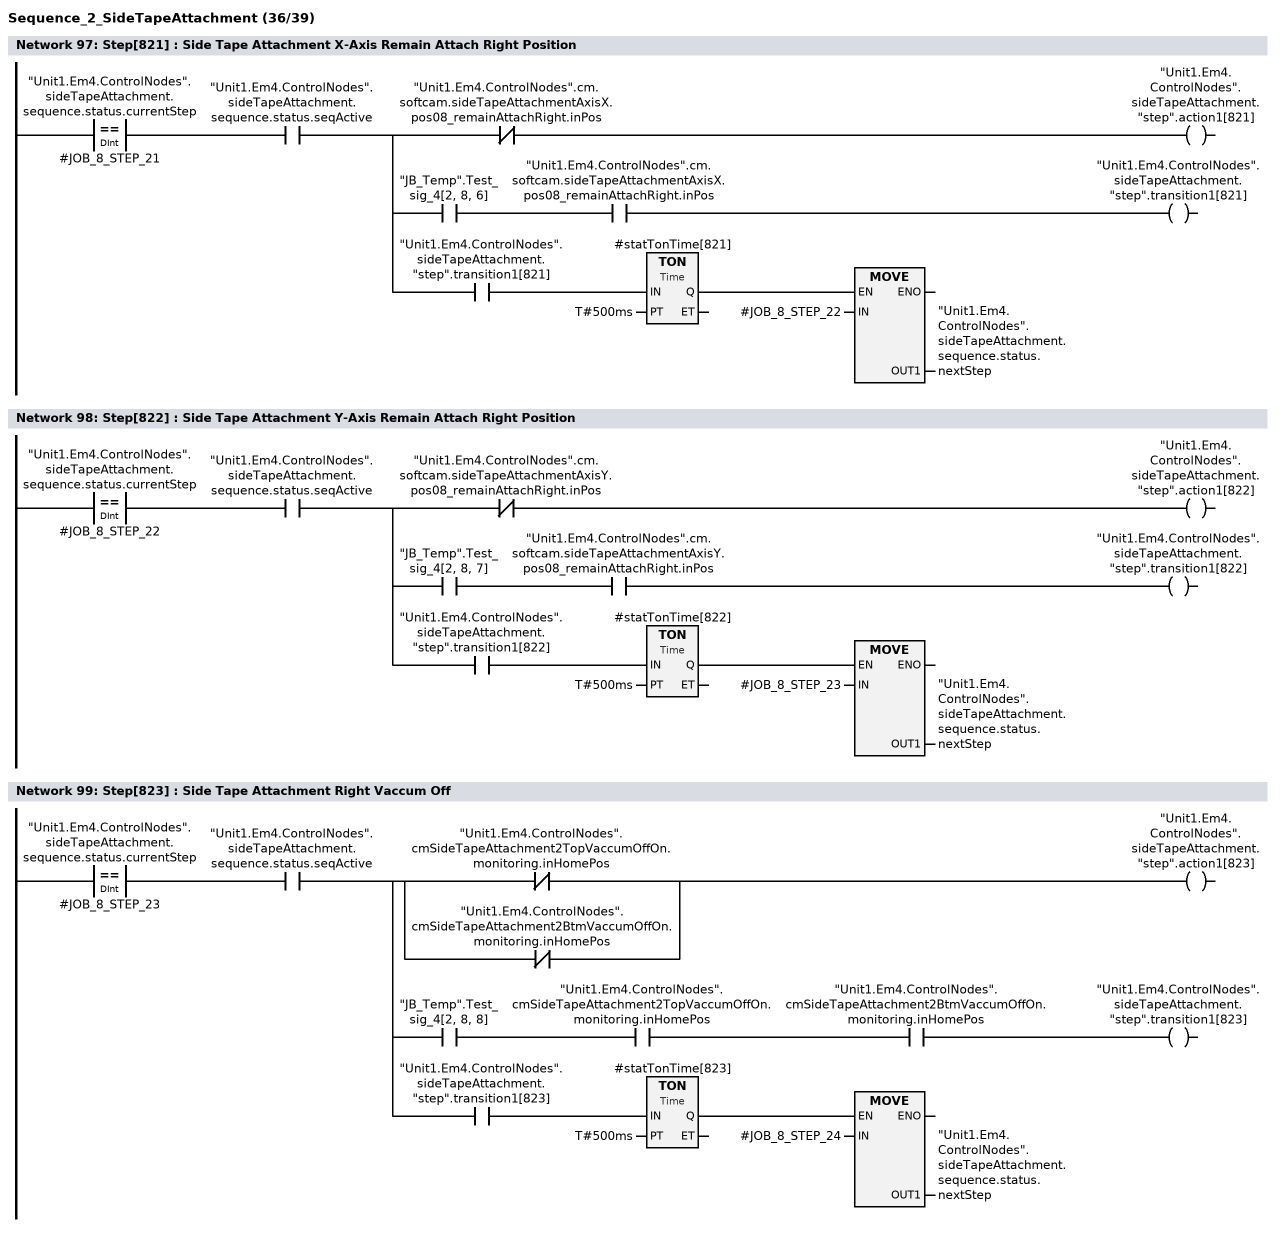
   RUNG wire#powerrail
      { S7_Templates := "SrcType := DInt" } EQ_Contact(in1 := "Unit1.Em4.ControlNodes".sideTapeAttachment.sequence.status.currentStep, in2 := #JOB_8_STEP_21)
      Contact( "Unit1.Em4.ControlNodes".sideTapeAttachment.sequence.status.seqActive )
      wire#w1
      I_Contact( "Unit1.Em4.ControlNodes".cm.softcam.sideTapeAttachmentAxisX.pos08_remainAttachRight.inPos )
      Coil( "Unit1.Em4.ControlNodes".sideTapeAttachment."step".action1[821] )
   END_RUNG
   RUNG wire#w1
      Contact( "JB_Temp".Test_sig_4[2, 8, 6] )
      Contact( "Unit1.Em4.ControlNodes".cm.softcam.sideTapeAttachmentAxisX.pos08_remainAttachRight.inPos )
      Coil( "Unit1.Em4.ControlNodes".sideTapeAttachment."step".transition1[821] )
   END_RUNG
   RUNG wire#w1
      Contact( "Unit1.Em4.ControlNodes".sideTapeAttachment."step".transition1[821] )
      { S7_Templates := "time_type := Time" } #statTonTime[821].TON(pt := T#500ms, et =>)
      Move(in := #JOB_8_STEP_22, out1 => "Unit1.Em4.ControlNodes".sideTapeAttachment.sequence.status.nextStep)
   END_RUNG
   // the same network as SCL:
   #_w1 := ("Unit1.Em4.ControlNodes".sideTapeAttachment.sequence.status.currentStep = #JOB_8_STEP_21) AND "Unit1.Em4.ControlNodes".sideTapeAttachment.sequence.status.seqActive;
   "Unit1.Em4.ControlNodes".sideTapeAttachment."step".action1[821] := #_w1 AND NOT "Unit1.Em4.ControlNodes".cm.softcam.sideTapeAttachmentAxisX.pos08_remainAttachRight.inPos;
   "Unit1.Em4.ControlNodes".sideTapeAttachment."step".transition1[821] := #_w1 AND "JB_Temp".Test_sig_4[2, 8, 6] AND "Unit1.Em4.ControlNodes".cm.softcam.sideTapeAttachmentAxisX.pos08_remainAttachRight.inPos;
   #statTonTime[821].TON(IN := #_w1 AND "Unit1.Em4.ControlNodes".sideTapeAttachment."step".transition1[821],
                         PT := T#500ms);
   IF #statTonTime[821].Q THEN
       "Unit1.Em4.ControlNodes".sideTapeAttachment.sequence.status.nextStep := #JOB_8_STEP_22;
   END_IF;
END_REGION

